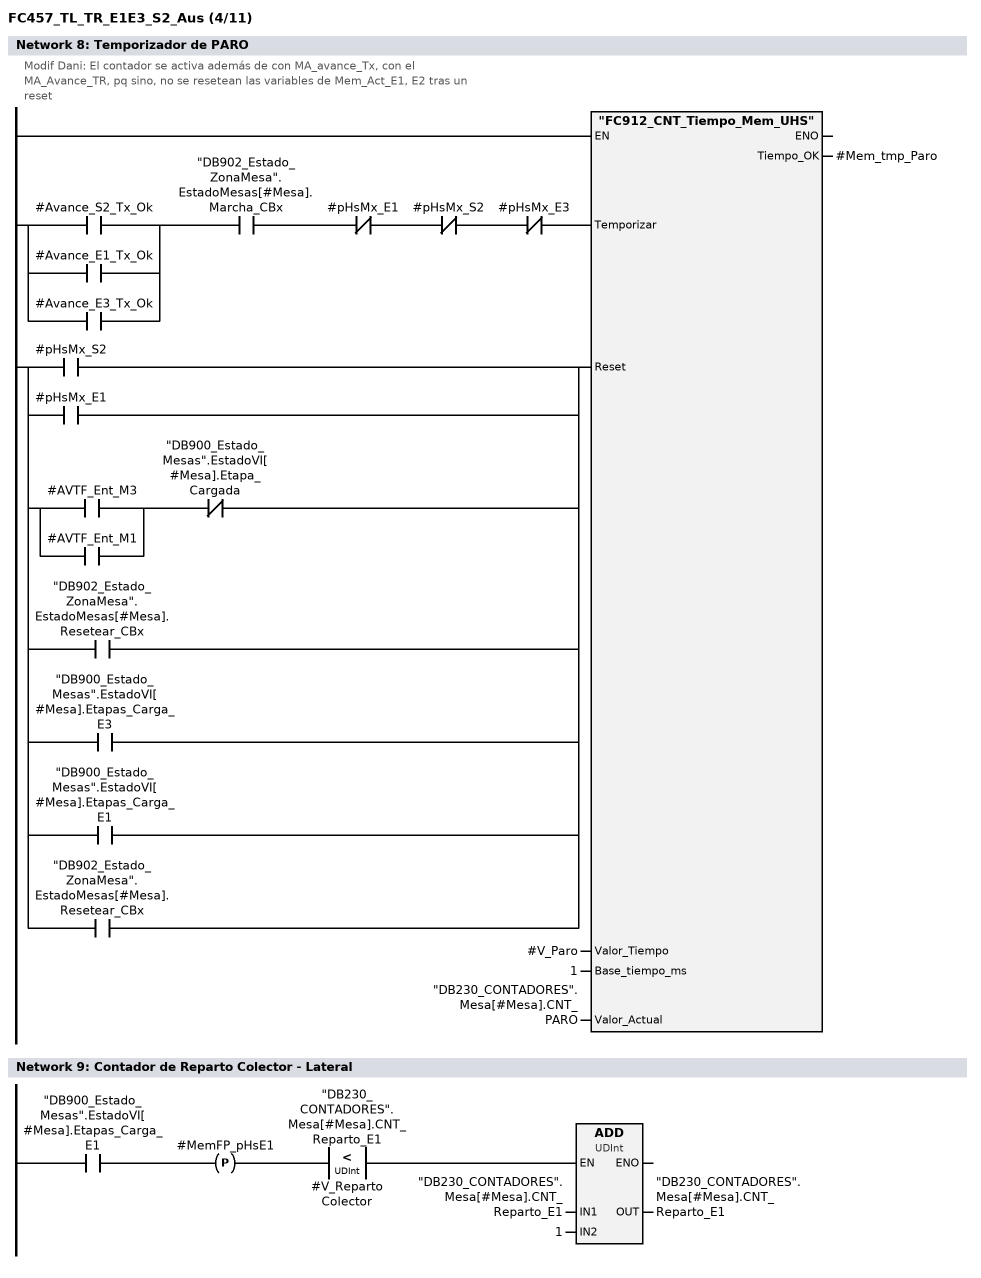
   RUNG wire#powerrail
      "FC912_CNT_Tiempo_Mem_UHS"(Temporizar := wire#w2, Reset := wire#w4, Valor_Tiempo := #V_Paro, Base_tiempo_ms := 1, Valor_Actual := "DB230_CONTADORES".Mesa[#Mesa].CNT_PARO, Tiempo_OK => #Mem_tmp_Paro)
   END_RUNG
   RUNG wire#powerrail
      Contact( #Avance_S2_Tx_Ok )
      wire#w1
      Contact( "DB902_Estado_ZonaMesa".EstadoMesas[#Mesa].Marcha_CBx )
      I_Contact( #pHsMx_E1 )
      I_Contact( #pHsMx_S2 )
      I_Contact( #pHsMx_E3 )
   END_RUNG wire#w2
   RUNG wire#powerrail
      Contact( #Avance_E1_Tx_Ok )
   END_RUNG wire#w1
   RUNG wire#powerrail
      Contact( #Avance_E3_Tx_Ok )
   END_RUNG wire#w1
   RUNG wire#powerrail
      Contact( #pHsMx_S2 )
   END_RUNG wire#w4
   RUNG wire#powerrail
      Contact( #pHsMx_E1 )
   END_RUNG wire#w4
   RUNG wire#powerrail
      Contact( #AVTF_Ent_M3 )
      wire#w3
      I_Contact( "DB900_Estado_Mesas".EstadoVI[#Mesa].Etapa_Cargada )
   END_RUNG wire#w4
   RUNG wire#powerrail
      Contact( #AVTF_Ent_M1 )
   END_RUNG wire#w3
   RUNG wire#powerrail
      Contact( "DB902_Estado_ZonaMesa".EstadoMesas[#Mesa].Resetear_CBx )
   END_RUNG wire#w4
   RUNG wire#powerrail
      Contact( "DB900_Estado_Mesas".EstadoVI[#Mesa].Etapas_Carga_E3 )
   END_RUNG wire#w4
   RUNG wire#powerrail
      Contact( "DB900_Estado_Mesas".EstadoVI[#Mesa].Etapas_Carga_E1 )
   END_RUNG wire#w4
   RUNG wire#powerrail
      Contact( "DB902_Estado_ZonaMesa".EstadoMesas[#Mesa].Resetear_CBx )
   END_RUNG wire#w4
   // the same network as SCL:
   "FC912_CNT_Tiempo_Mem_UHS"(Temporizar := (#Avance_S2_Tx_Ok OR #Avance_E1_Tx_Ok OR #Avance_E3_Tx_Ok) AND "DB902_Estado_ZonaMesa".EstadoMesas[#Mesa].Marcha_CBx AND NOT #pHsMx_E1 AND NOT #pHsMx_S2 AND NOT #pHsMx_E3,
                           Reset := #pHsMx_S2 OR #pHsMx_E1 OR ((#AVTF_Ent_M3 OR #AVTF_Ent_M1) AND NOT "DB900_Estado_Mesas".EstadoVI[#Mesa].Etapa_Cargada) OR "DB902_Estado_ZonaMesa".EstadoMesas[#Mesa].Resetear_CBx OR "DB900_Estado_Mesas".EstadoVI[#Mesa].Etapas_Carga_E3 OR "DB900_Estado_Mesas".EstadoVI[#Mesa].Etapas_Carga_E1 OR "DB902_Estado_ZonaMesa".EstadoMesas[#Mesa].Resetear_CBx,
                           Valor_Tiempo := #V_Paro,
                           Base_tiempo_ms := 1,
                           Valor_Actual := "DB230_CONTADORES".Mesa[#Mesa].CNT_PARO,
                           Tiempo_OK => #Mem_tmp_Paro);
END_REGION

REGION Network 9: Contador de Reparto Colector - Lateral
   RUNG wire#powerrail
      Contact( "DB900_Estado_Mesas".EstadoVI[#Mesa].Etapas_Carga_E1 )
      P_Trig( #MemFP_pHsE1 )
      { S7_Templates := "SrcType := UDInt" } LT_Contact(in1 := "DB230_CONTADORES".Mesa[#Mesa].CNT_Reparto_E1, in2 := #V_RepartoColector)
      { S7_Templates := "SrcType := UDInt"; S7_GenerateENO := "TRUE" } Add(in1 := "DB230_CONTADORES".Mesa[#Mesa].CNT_Reparto_E1, in2 := 1, out => "DB230_CONTADORES".Mesa[#Mesa].CNT_Reparto_E1)
   END_RUNG
   // the same network as SCL:
   #_w1 := "DB900_Estado_Mesas".EstadoVI[#Mesa].Etapas_Carga_E1 AND NOT #MemFP_pHsE1;   // rising edge
   #MemFP_pHsE1 := "DB900_Estado_Mesas".EstadoVI[#Mesa].Etapas_Carga_E1;
   IF #_w1 AND ("DB230_CONTADORES".Mesa[#Mesa].CNT_Reparto_E1 < #V_RepartoColector) THEN
       "DB230_CONTADORES".Mesa[#Mesa].CNT_Reparto_E1 := "DB230_CONTADORES".Mesa[#Mesa].CNT_Reparto_E1 + 1;
   END_IF;
END_REGION

REGION Network 10
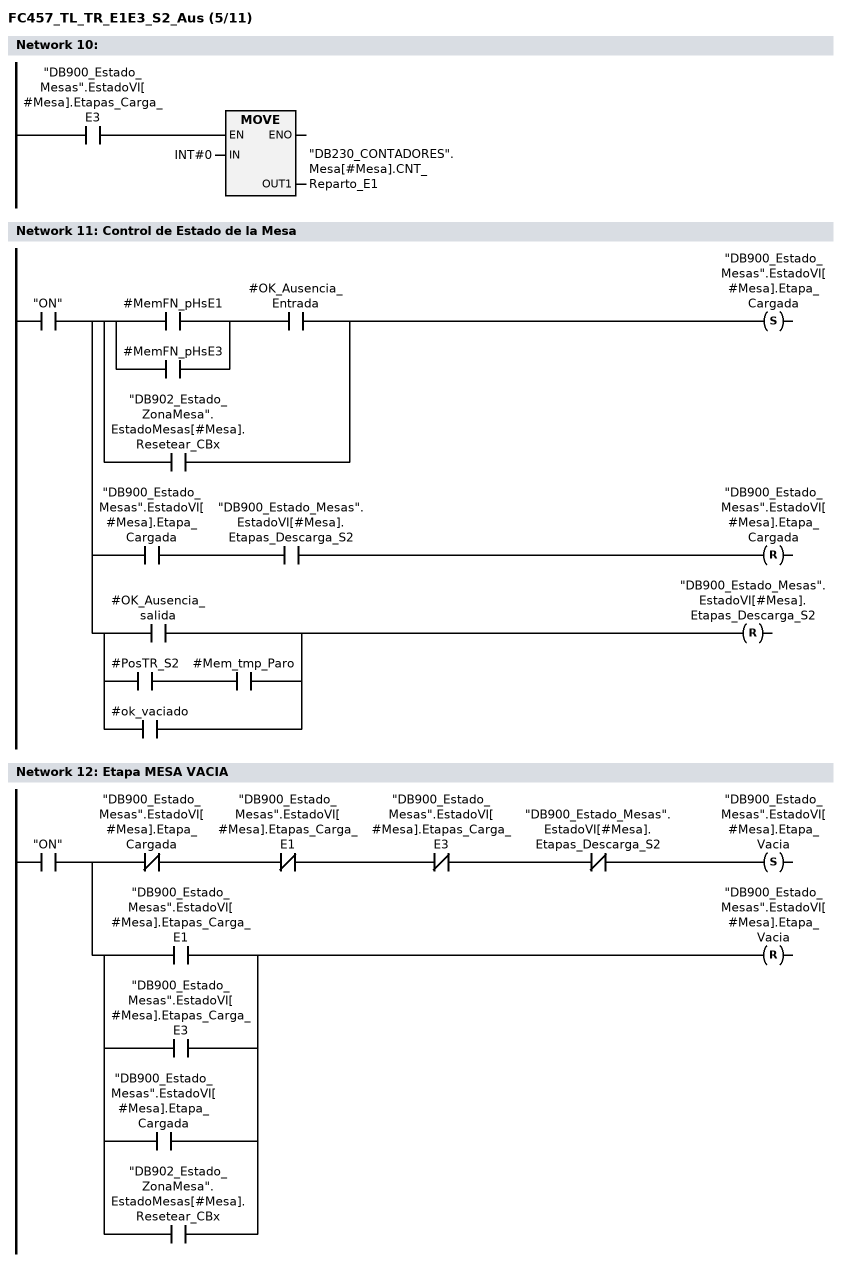
   RUNG wire#powerrail
      Contact( "DB900_Estado_Mesas".EstadoVI[#Mesa].Etapas_Carga_E3 )
      { S7_GenerateENO := "TRUE" } Move(in := INT#0, out1 => "DB230_CONTADORES".Mesa[#Mesa].CNT_Reparto_E1)
   END_RUNG
   // the same network as SCL:
   IF "DB900_Estado_Mesas".EstadoVI[#Mesa].Etapas_Carga_E3 THEN
       "DB230_CONTADORES".Mesa[#Mesa].CNT_Reparto_E1 := INT#0;
   END_IF;
END_REGION

REGION Network 11: Control de Estado de la Mesa
   RUNG wire#powerrail
      Contact( "ON" )
      wire#w1
      Contact( #MemFN_pHsE1 )
      wire#w2
      Contact( #OK_Ausencia_Entrada )
      wire#w3
      S_Coil( "DB900_Estado_Mesas".EstadoVI[#Mesa].Etapa_Cargada )
   END_RUNG
   RUNG wire#w1
      Contact( #MemFN_pHsE3 )
   END_RUNG wire#w2
   RUNG wire#w1
      Contact( "DB902_Estado_ZonaMesa".EstadoMesas[#Mesa].Resetear_CBx )
   END_RUNG wire#w3
   RUNG wire#w1
      Contact( "DB900_Estado_Mesas".EstadoVI[#Mesa].Etapa_Cargada )
      Contact( "DB900_Estado_Mesas".EstadoVI[#Mesa].Etapas_Descarga_S2 )
      R_Coil( "DB900_Estado_Mesas".EstadoVI[#Mesa].Etapa_Cargada )
   END_RUNG
   RUNG wire#w1
      Contact( #OK_Ausencia_salida )
      wire#w4
      R_Coil( "DB900_Estado_Mesas".EstadoVI[#Mesa].Etapas_Descarga_S2 )
   END_RUNG
   RUNG wire#w1
      Contact( #PosTR_S2 )
      Contact( #Mem_tmp_Paro )
   END_RUNG wire#w4
   RUNG wire#w1
      Contact( #ok_vaciado )
   END_RUNG wire#w4
   // the same network as SCL:
   IF "ON" AND (((#MemFN_pHsE1 OR #MemFN_pHsE3) AND #OK_Ausencia_Entrada) OR "DB902_Estado_ZonaMesa".EstadoMesas[#Mesa].Resetear_CBx) THEN
       "DB900_Estado_Mesas".EstadoVI[#Mesa].Etapa_Cargada := TRUE;
   END_IF;
   IF "ON" AND "DB900_Estado_Mesas".EstadoVI[#Mesa].Etapa_Cargada AND "DB900_Estado_Mesas".EstadoVI[#Mesa].Etapas_Descarga_S2 THEN
       "DB900_Estado_Mesas".EstadoVI[#Mesa].Etapa_Cargada := FALSE;
   END_IF;
   IF "ON" AND (#OK_Ausencia_salida OR (#PosTR_S2 AND #Mem_tmp_Paro) OR #ok_vaciado) THEN
       "DB900_Estado_Mesas".EstadoVI[#Mesa].Etapas_Descarga_S2 := FALSE;
   END_IF;
END_REGION

REGION Network 12: Etapa MESA VACIA
   RUNG wire#powerrail
      Contact( "ON" )
      wire#w1
      I_Contact( "DB900_Estado_Mesas".EstadoVI[#Mesa].Etapa_Cargada )
      I_Contact( "DB900_Estado_Mesas".EstadoVI[#Mesa].Etapas_Carga_E1 )
      I_Contact( "DB900_Estado_Mesas".EstadoVI[#Mesa].Etapas_Carga_E3 )
      I_Contact( "DB900_Estado_Mesas".EstadoVI[#Mesa].Etapas_Descarga_S2 )
      S_Coil( "DB900_Estado_Mesas".EstadoVI[#Mesa].Etapa_Vacia )
   END_RUNG
   RUNG wire#w1
      Contact( "DB900_Estado_Mesas".EstadoVI[#Mesa].Etapas_Carga_E1 )
      wire#w2
      R_Coil( "DB900_Estado_Mesas".EstadoVI[#Mesa].Etapa_Vacia )
   END_RUNG
   RUNG wire#w1
      Contact( "DB900_Estado_Mesas".EstadoVI[#Mesa].Etapas_Carga_E3 )
   END_RUNG wire#w2
   RUNG wire#w1
      Contact( "DB900_Estado_Mesas".EstadoVI[#Mesa].Etapa_Cargada )
   END_RUNG wire#w2
   RUNG wire#w1
      Contact( "DB902_Estado_ZonaMesa".EstadoMesas[#Mesa].Resetear_CBx )
   END_RUNG wire#w2
   // the same network as SCL:
   IF "ON" AND NOT "DB900_Estado_Mesas".EstadoVI[#Mesa].Etapa_Cargada AND NOT "DB900_Estado_Mesas".EstadoVI[#Mesa].Etapas_Carga_E1 AND NOT "DB900_Estado_Mesas".EstadoVI[#Mesa].Etapas_Carga_E3 AND NOT "DB900_Estado_Mesas".EstadoVI[#Mesa].Etapas_Descarga_S2 THEN
       "DB900_Estado_Mesas".EstadoVI[#Mesa].Etapa_Vacia := TRUE;
   END_IF;
   IF "ON" AND ("DB900_Estado_Mesas".EstadoVI[#Mesa].Etapas_Carga_E1 OR "DB900_Estado_Mesas".EstadoVI[#Mesa].Etapas_Carga_E3 OR "DB900_Estado_Mesas".EstadoVI[#Mesa].Etapa_Cargada OR "DB902_Estado_ZonaMesa".EstadoMesas[#Mesa].Resetear_CBx) THEN
       "DB900_Estado_Mesas".EstadoVI[#Mesa].Etapa_Vacia := FALSE;
   END_IF;
END_REGION

REGION Network 13
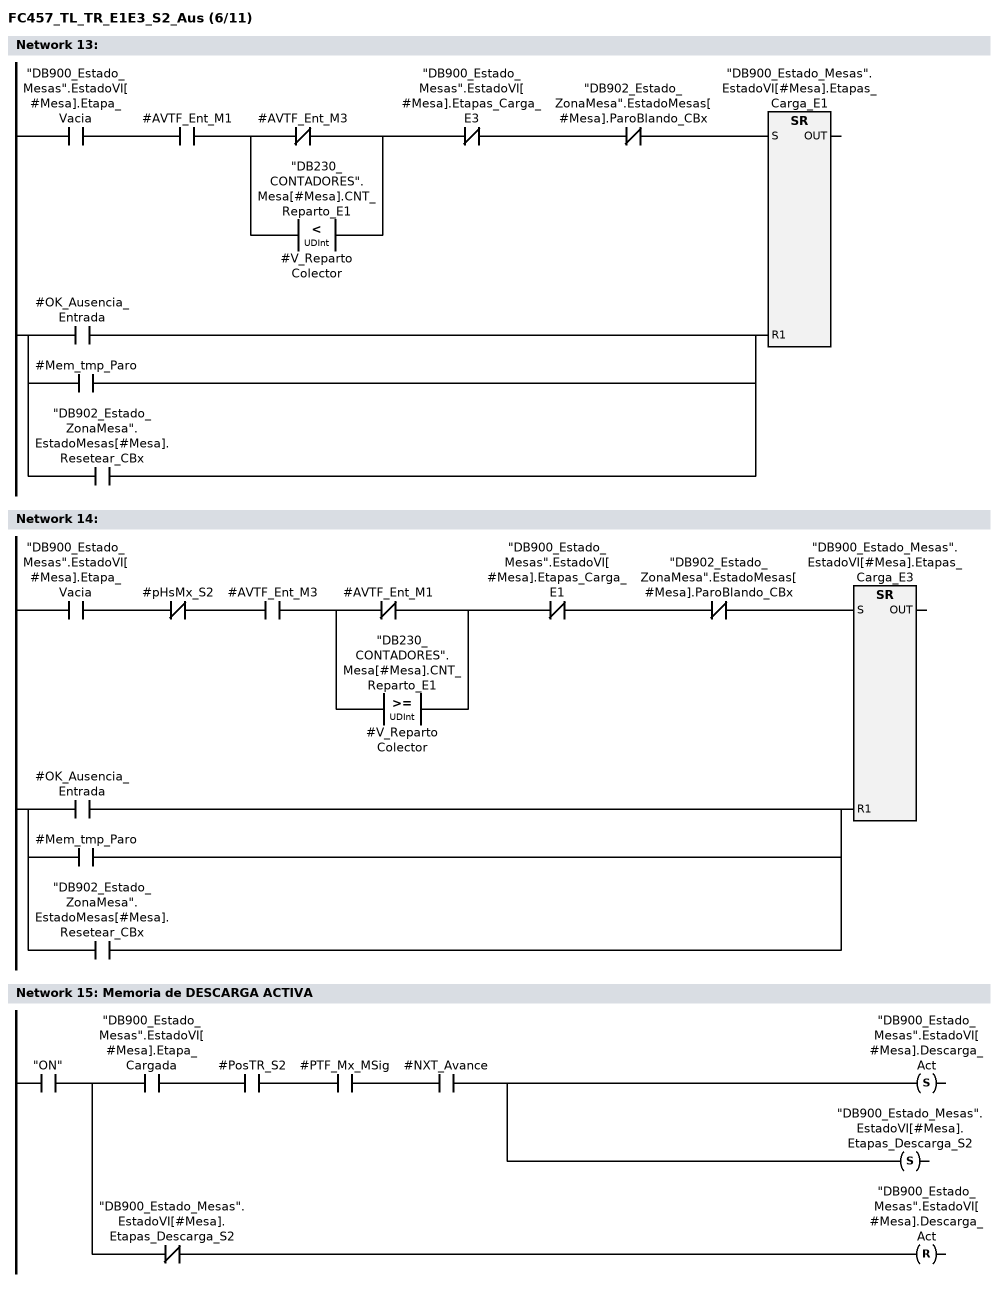
   RUNG wire#powerrail
      Contact( "DB900_Estado_Mesas".EstadoVI[#Mesa].Etapa_Vacia )
      Contact( #AVTF_Ent_M1 )
      wire#w1
      I_Contact( #AVTF_Ent_M3 )
      wire#w2
      I_Contact( "DB900_Estado_Mesas".EstadoVI[#Mesa].Etapas_Carga_E3 )
      I_Contact( "DB902_Estado_ZonaMesa".EstadoMesas[#Mesa].ParoBlando_CBx )
      S_SR(operand := "DB900_Estado_Mesas".EstadoVI[#Mesa].Etapas_Carga_E1, r1 := wire#w3)
   END_RUNG
   RUNG wire#w1
      { S7_Templates := "SrcType := UDInt" } LT_Contact(in1 := "DB230_CONTADORES".Mesa[#Mesa].CNT_Reparto_E1, in2 := #V_RepartoColector)
   END_RUNG wire#w2
   RUNG wire#powerrail
      Contact( #OK_Ausencia_Entrada )
   END_RUNG wire#w3
   RUNG wire#powerrail
      Contact( #Mem_tmp_Paro )
   END_RUNG wire#w3
   RUNG wire#powerrail
      Contact( "DB902_Estado_ZonaMesa".EstadoMesas[#Mesa].Resetear_CBx )
   END_RUNG wire#w3
   // the same network as SCL:
   #_w1 := #OK_Ausencia_Entrada OR #Mem_tmp_Paro OR "DB902_Estado_ZonaMesa".EstadoMesas[#Mesa].Resetear_CBx;
   IF "DB900_Estado_Mesas".EstadoVI[#Mesa].Etapa_Vacia AND #AVTF_Ent_M1 AND (NOT #AVTF_Ent_M3 OR ("DB230_CONTADORES".Mesa[#Mesa].CNT_Reparto_E1 < #V_RepartoColector)) AND NOT "DB900_Estado_Mesas".EstadoVI[#Mesa].Etapas_Carga_E3 AND NOT "DB902_Estado_ZonaMesa".EstadoMesas[#Mesa].ParoBlando_CBx THEN
       "DB900_Estado_Mesas".EstadoVI[#Mesa].Etapas_Carga_E1 := TRUE;   // SR flip-flop
   END_IF;
   IF #_w1 THEN "DB900_Estado_Mesas".EstadoVI[#Mesa].Etapas_Carga_E1 := FALSE; END_IF;
END_REGION

REGION Network 14
   RUNG wire#powerrail
      Contact( "DB900_Estado_Mesas".EstadoVI[#Mesa].Etapa_Vacia )
      I_Contact( #pHsMx_S2 )
      Contact( #AVTF_Ent_M3 )
      wire#w1
      I_Contact( #AVTF_Ent_M1 )
      wire#w2
      I_Contact( "DB900_Estado_Mesas".EstadoVI[#Mesa].Etapas_Carga_E1 )
      I_Contact( "DB902_Estado_ZonaMesa".EstadoMesas[#Mesa].ParoBlando_CBx )
      S_SR(operand := "DB900_Estado_Mesas".EstadoVI[#Mesa].Etapas_Carga_E3, r1 := wire#w3)
   END_RUNG
   RUNG wire#w1
      { S7_Templates := "SrcType := UDInt" } GE_Contact(in1 := "DB230_CONTADORES".Mesa[#Mesa].CNT_Reparto_E1, in2 := #V_RepartoColector)
   END_RUNG wire#w2
   RUNG wire#powerrail
      Contact( #OK_Ausencia_Entrada )
   END_RUNG wire#w3
   RUNG wire#powerrail
      Contact( #Mem_tmp_Paro )
   END_RUNG wire#w3
   RUNG wire#powerrail
      Contact( "DB902_Estado_ZonaMesa".EstadoMesas[#Mesa].Resetear_CBx )
   END_RUNG wire#w3
   // the same network as SCL:
   #_w1 := #OK_Ausencia_Entrada OR #Mem_tmp_Paro OR "DB902_Estado_ZonaMesa".EstadoMesas[#Mesa].Resetear_CBx;
   IF "DB900_Estado_Mesas".EstadoVI[#Mesa].Etapa_Vacia AND NOT #pHsMx_S2 AND #AVTF_Ent_M3 AND (NOT #AVTF_Ent_M1 OR ("DB230_CONTADORES".Mesa[#Mesa].CNT_Reparto_E1 >= #V_RepartoColector)) AND NOT "DB900_Estado_Mesas".EstadoVI[#Mesa].Etapas_Carga_E1 AND NOT "DB902_Estado_ZonaMesa".EstadoMesas[#Mesa].ParoBlando_CBx THEN
       "DB900_Estado_Mesas".EstadoVI[#Mesa].Etapas_Carga_E3 := TRUE;   // SR flip-flop
   END_IF;
   IF #_w1 THEN "DB900_Estado_Mesas".EstadoVI[#Mesa].Etapas_Carga_E3 := FALSE; END_IF;
END_REGION

REGION Network 15: Memoria de DESCARGA ACTIVA
   RUNG wire#powerrail
      Contact( "ON" )
      wire#w1
      Contact( "DB900_Estado_Mesas".EstadoVI[#Mesa].Etapa_Cargada )
      Contact( #PosTR_S2 )
      Contact( #PTF_Mx_MSig )
      Contact( #NXT_Avance )
      wire#w2
      S_Coil( "DB900_Estado_Mesas".EstadoVI[#Mesa].Descarga_Act )
   END_RUNG
   RUNG wire#w2
      S_Coil( "DB900_Estado_Mesas".EstadoVI[#Mesa].Etapas_Descarga_S2 )
   END_RUNG
   RUNG wire#w1
      I_Contact( "DB900_Estado_Mesas".EstadoVI[#Mesa].Etapas_Descarga_S2 )
      R_Coil( "DB900_Estado_Mesas".EstadoVI[#Mesa].Descarga_Act )
   END_RUNG
   // the same network as SCL:
   #_w1 := "ON" AND "DB900_Estado_Mesas".EstadoVI[#Mesa].Etapa_Cargada AND #PosTR_S2 AND #PTF_Mx_MSig AND #NXT_Avance;
   IF #_w1 THEN
       "DB900_Estado_Mesas".EstadoVI[#Mesa].Descarga_Act := TRUE;
       "DB900_Estado_Mesas".EstadoVI[#Mesa].Etapas_Descarga_S2 := TRUE;
   END_IF;
   IF "ON" AND NOT "DB900_Estado_Mesas".EstadoVI[#Mesa].Etapas_Descarga_S2 THEN
       "DB900_Estado_Mesas".EstadoVI[#Mesa].Descarga_Act := FALSE;
   END_IF;
END_REGION

REGION Network 16: Salidas Auxiliares
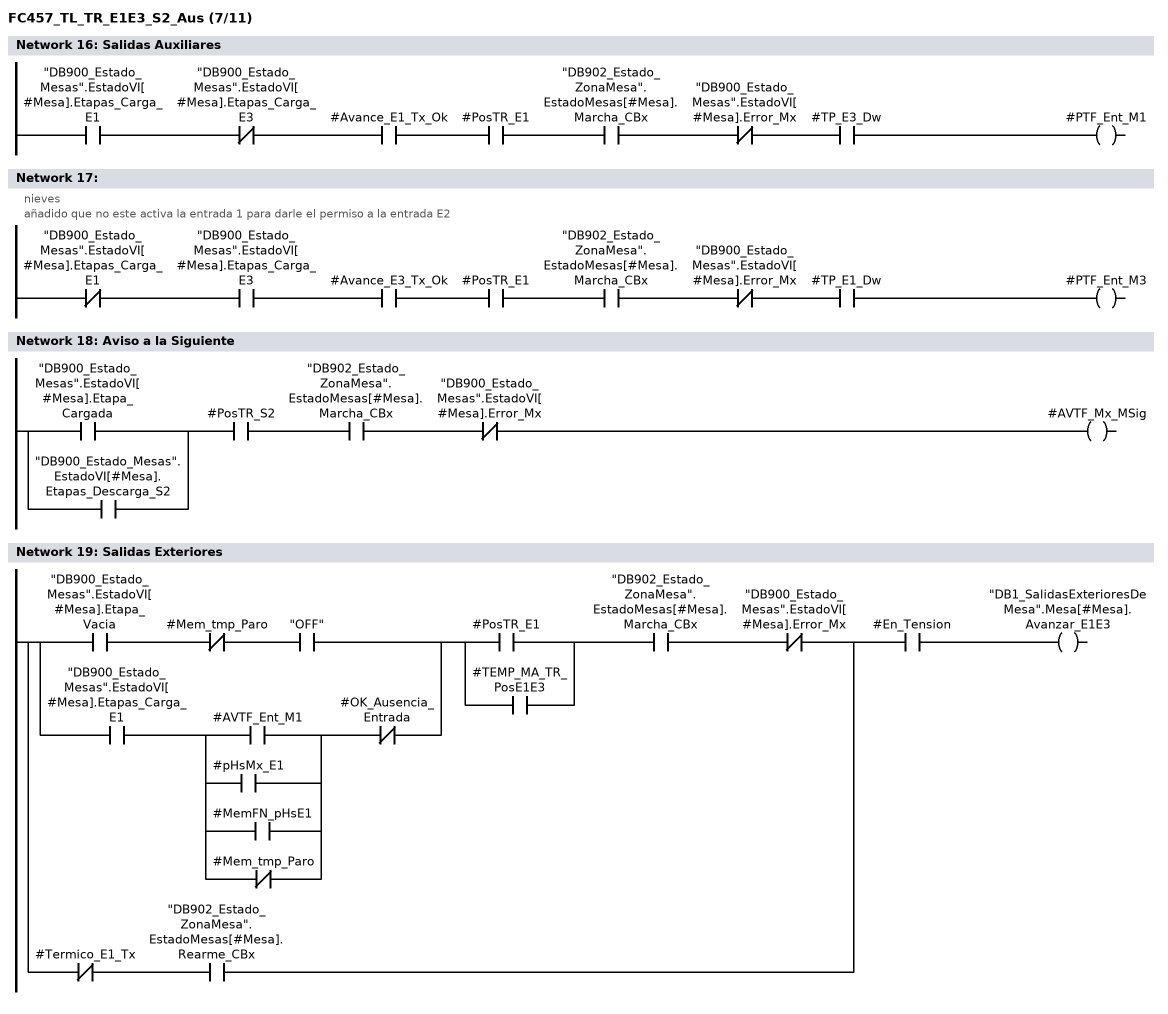
   RUNG wire#powerrail
      Contact( "DB900_Estado_Mesas".EstadoVI[#Mesa].Etapas_Carga_E1 )
      I_Contact( "DB900_Estado_Mesas".EstadoVI[#Mesa].Etapas_Carga_E3 )
      Contact( #Avance_E1_Tx_Ok )
      Contact( #PosTR_E1 )
      Contact( "DB902_Estado_ZonaMesa".EstadoMesas[#Mesa].Marcha_CBx )
      I_Contact( "DB900_Estado_Mesas".EstadoVI[#Mesa].Error_Mx )
      Contact( #TP_E3_Dw )
      Coil( #PTF_Ent_M1 )
   END_RUNG
   // the same network as SCL:
   #PTF_Ent_M1 := "DB900_Estado_Mesas".EstadoVI[#Mesa].Etapas_Carga_E1 AND NOT "DB900_Estado_Mesas".EstadoVI[#Mesa].Etapas_Carga_E3 AND #Avance_E1_Tx_Ok AND #PosTR_E1 AND "DB902_Estado_ZonaMesa".EstadoMesas[#Mesa].Marcha_CBx AND NOT "DB900_Estado_Mesas".EstadoVI[#Mesa].Error_Mx AND #TP_E3_Dw;
END_REGION

REGION Network 17
   // nieves
   // añadido que no este activa la entrada 1 para darle el permiso a la entrada E2
   RUNG wire#powerrail
      I_Contact( "DB900_Estado_Mesas".EstadoVI[#Mesa].Etapas_Carga_E1 )
      Contact( "DB900_Estado_Mesas".EstadoVI[#Mesa].Etapas_Carga_E3 )
      Contact( #Avance_E3_Tx_Ok )
      Contact( #PosTR_E1 )
      Contact( "DB902_Estado_ZonaMesa".EstadoMesas[#Mesa].Marcha_CBx )
      I_Contact( "DB900_Estado_Mesas".EstadoVI[#Mesa].Error_Mx )
      Contact( #TP_E1_Dw )
      Coil( #PTF_Ent_M3 )
   END_RUNG
   // the same network as SCL:
   #PTF_Ent_M3 := NOT "DB900_Estado_Mesas".EstadoVI[#Mesa].Etapas_Carga_E1 AND "DB900_Estado_Mesas".EstadoVI[#Mesa].Etapas_Carga_E3 AND #Avance_E3_Tx_Ok AND #PosTR_E1 AND "DB902_Estado_ZonaMesa".EstadoMesas[#Mesa].Marcha_CBx AND NOT "DB900_Estado_Mesas".EstadoVI[#Mesa].Error_Mx AND #TP_E1_Dw;
END_REGION

REGION Network 18: Aviso a la Siguiente
   RUNG wire#powerrail
      Contact( "DB900_Estado_Mesas".EstadoVI[#Mesa].Etapa_Cargada )
      wire#w1
      Contact( #PosTR_S2 )
      Contact( "DB902_Estado_ZonaMesa".EstadoMesas[#Mesa].Marcha_CBx )
      I_Contact( "DB900_Estado_Mesas".EstadoVI[#Mesa].Error_Mx )
      Coil( #AVTF_Mx_MSig )
   END_RUNG
   RUNG wire#powerrail
      Contact( "DB900_Estado_Mesas".EstadoVI[#Mesa].Etapas_Descarga_S2 )
   END_RUNG wire#w1
   // the same network as SCL:
   #AVTF_Mx_MSig := ("DB900_Estado_Mesas".EstadoVI[#Mesa].Etapa_Cargada OR "DB900_Estado_Mesas".EstadoVI[#Mesa].Etapas_Descarga_S2) AND #PosTR_S2 AND "DB902_Estado_ZonaMesa".EstadoMesas[#Mesa].Marcha_CBx AND NOT "DB900_Estado_Mesas".EstadoVI[#Mesa].Error_Mx;
END_REGION

REGION Network 19: Salidas Exteriores
   RUNG wire#powerrail
      Contact( "DB900_Estado_Mesas".EstadoVI[#Mesa].Etapa_Vacia )
      I_Contact( #Mem_tmp_Paro )
      Contact( "OFF" )
      wire#w1
      Contact( #PosTR_E1 )
      wire#w4
      Contact( "DB902_Estado_ZonaMesa".EstadoMesas[#Mesa].Marcha_CBx )
      I_Contact( "DB900_Estado_Mesas".EstadoVI[#Mesa].Error_Mx )
      wire#w5
      Contact( #En_Tension )
      Coil( "DB1_SalidasExterioresDeMesa".Mesa[#Mesa].Avanzar_E1E3 )
   END_RUNG
   RUNG wire#powerrail
      Contact( "DB900_Estado_Mesas".EstadoVI[#Mesa].Etapas_Carga_E1 )
      wire#w2
      Contact( #AVTF_Ent_M1 )
      wire#w3
      I_Contact( #OK_Ausencia_Entrada )
   END_RUNG wire#w1
   RUNG wire#w2
      Contact( #pHsMx_E1 )
   END_RUNG wire#w3
   RUNG wire#w2
      Contact( #MemFN_pHsE1 )
   END_RUNG wire#w3
   RUNG wire#w2
      I_Contact( #Mem_tmp_Paro )
   END_RUNG wire#w3
   RUNG wire#w1
      Contact( #TEMP_MA_TR_PosE1E3 )
   END_RUNG wire#w4
   RUNG wire#powerrail
      I_Contact( #Termico_E1_Tx )
      Contact( "DB902_Estado_ZonaMesa".EstadoMesas[#Mesa].Rearme_CBx )
   END_RUNG wire#w5
   // the same network as SCL:
   "DB1_SalidasExterioresDeMesa".Mesa[#Mesa].Avanzar_E1E3 := (((("DB900_Estado_Mesas".EstadoVI[#Mesa].Etapa_Vacia AND NOT #Mem_tmp_Paro AND "OFF") OR ("DB900_Estado_Mesas".EstadoVI[#Mesa].Etapas_Carga_E1 AND (#AVTF_Ent_M1 OR #pHsMx_E1 OR #MemFN_pHsE1 OR NOT #Mem_tmp_Paro) AND NOT #OK_Ausencia_Entrada)) AND (#PosTR_E1 OR #TEMP_MA_TR_PosE1E3) AND "DB902_Estado_ZonaMesa".EstadoMesas[#Mesa].Marcha_CBx AND NOT "DB900_Estado_Mesas".EstadoVI[#Mesa].Error_Mx) OR (NOT #Termico_E1_Tx AND "DB902_Estado_ZonaMesa".EstadoMesas[#Mesa].Rearme_CBx)) AND #En_Tension;
END_REGION

REGION Network 20: ---
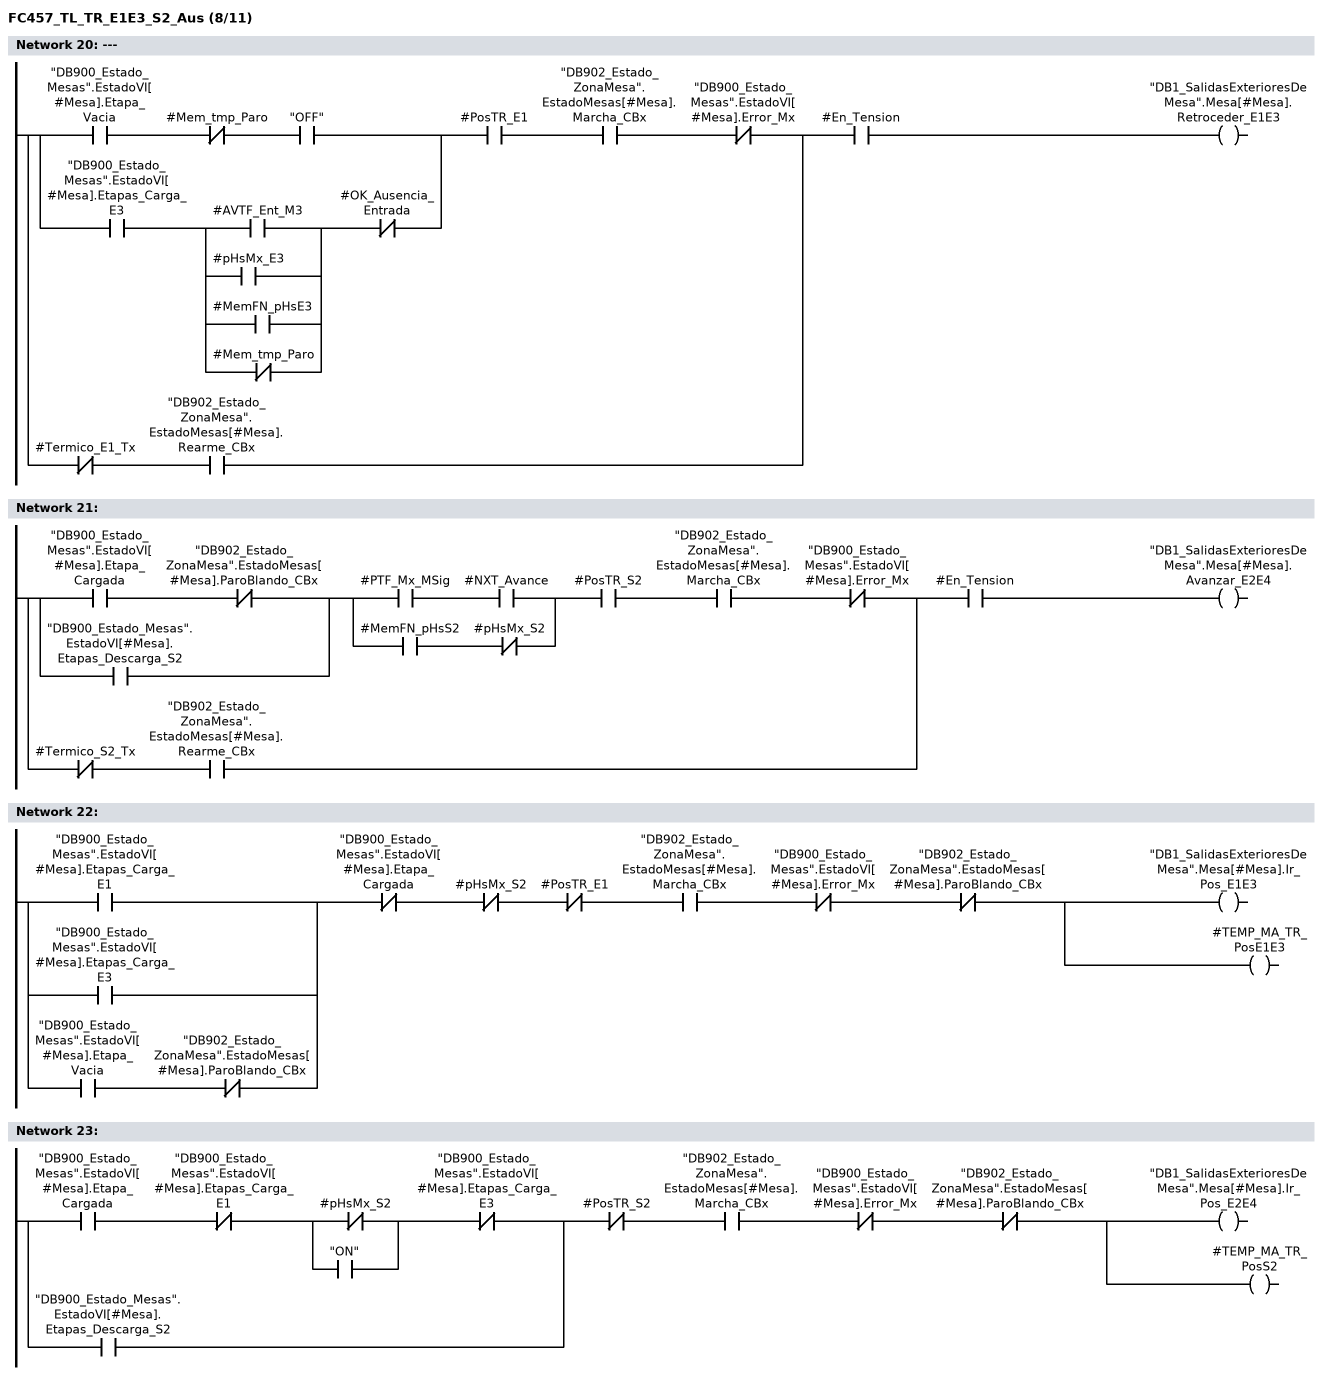
   RUNG wire#powerrail
      Contact( "DB900_Estado_Mesas".EstadoVI[#Mesa].Etapa_Vacia )
      I_Contact( #Mem_tmp_Paro )
      Contact( "OFF" )
      wire#w1
      Contact( #PosTR_E1 )
      Contact( "DB902_Estado_ZonaMesa".EstadoMesas[#Mesa].Marcha_CBx )
      I_Contact( "DB900_Estado_Mesas".EstadoVI[#Mesa].Error_Mx )
      wire#w4
      Contact( #En_Tension )
      Coil( "DB1_SalidasExterioresDeMesa".Mesa[#Mesa].Retroceder_E1E3 )
   END_RUNG
   RUNG wire#powerrail
      Contact( "DB900_Estado_Mesas".EstadoVI[#Mesa].Etapas_Carga_E3 )
      wire#w2
      Contact( #AVTF_Ent_M3 )
      wire#w3
      I_Contact( #OK_Ausencia_Entrada )
   END_RUNG wire#w1
   RUNG wire#w2
      Contact( #pHsMx_E3 )
   END_RUNG wire#w3
   RUNG wire#w2
      Contact( #MemFN_pHsE3 )
   END_RUNG wire#w3
   RUNG wire#w2
      I_Contact( #Mem_tmp_Paro )
   END_RUNG wire#w3
   RUNG wire#powerrail
      I_Contact( #Termico_E1_Tx )
      Contact( "DB902_Estado_ZonaMesa".EstadoMesas[#Mesa].Rearme_CBx )
   END_RUNG wire#w4
   // the same network as SCL:
   "DB1_SalidasExterioresDeMesa".Mesa[#Mesa].Retroceder_E1E3 := (((("DB900_Estado_Mesas".EstadoVI[#Mesa].Etapa_Vacia AND NOT #Mem_tmp_Paro AND "OFF") OR ("DB900_Estado_Mesas".EstadoVI[#Mesa].Etapas_Carga_E3 AND (#AVTF_Ent_M3 OR #pHsMx_E3 OR #MemFN_pHsE3 OR NOT #Mem_tmp_Paro) AND NOT #OK_Ausencia_Entrada)) AND #PosTR_E1 AND "DB902_Estado_ZonaMesa".EstadoMesas[#Mesa].Marcha_CBx AND NOT "DB900_Estado_Mesas".EstadoVI[#Mesa].Error_Mx) OR (NOT #Termico_E1_Tx AND "DB902_Estado_ZonaMesa".EstadoMesas[#Mesa].Rearme_CBx)) AND #En_Tension;
END_REGION

REGION Network 21
   RUNG wire#powerrail
      Contact( "DB900_Estado_Mesas".EstadoVI[#Mesa].Etapa_Cargada )
      I_Contact( "DB902_Estado_ZonaMesa".EstadoMesas[#Mesa].ParoBlando_CBx )
      wire#w1
      Contact( #PTF_Mx_MSig )
      Contact( #NXT_Avance )
      wire#w2
      Contact( #PosTR_S2 )
      Contact( "DB902_Estado_ZonaMesa".EstadoMesas[#Mesa].Marcha_CBx )
      I_Contact( "DB900_Estado_Mesas".EstadoVI[#Mesa].Error_Mx )
      wire#w3
      Contact( #En_Tension )
      Coil( "DB1_SalidasExterioresDeMesa".Mesa[#Mesa].Avanzar_E2E4 )
   END_RUNG
   RUNG wire#powerrail
      Contact( "DB900_Estado_Mesas".EstadoVI[#Mesa].Etapas_Descarga_S2 )
   END_RUNG wire#w1
   RUNG wire#w1
      Contact( #MemFN_pHsS2 )
      I_Contact( #pHsMx_S2 )
   END_RUNG wire#w2
   RUNG wire#powerrail
      I_Contact( #Termico_S2_Tx )
      Contact( "DB902_Estado_ZonaMesa".EstadoMesas[#Mesa].Rearme_CBx )
   END_RUNG wire#w3
   // the same network as SCL:
   "DB1_SalidasExterioresDeMesa".Mesa[#Mesa].Avanzar_E2E4 := (((("DB900_Estado_Mesas".EstadoVI[#Mesa].Etapa_Cargada AND NOT "DB902_Estado_ZonaMesa".EstadoMesas[#Mesa].ParoBlando_CBx) OR "DB900_Estado_Mesas".EstadoVI[#Mesa].Etapas_Descarga_S2) AND ((#PTF_Mx_MSig AND #NXT_Avance) OR (#MemFN_pHsS2 AND NOT #pHsMx_S2)) AND #PosTR_S2 AND "DB902_Estado_ZonaMesa".EstadoMesas[#Mesa].Marcha_CBx AND NOT "DB900_Estado_Mesas".EstadoVI[#Mesa].Error_Mx) OR (NOT #Termico_S2_Tx AND "DB902_Estado_ZonaMesa".EstadoMesas[#Mesa].Rearme_CBx)) AND #En_Tension;
END_REGION

REGION Network 22
   RUNG wire#powerrail
      Contact( "DB900_Estado_Mesas".EstadoVI[#Mesa].Etapas_Carga_E1 )
      wire#w1
      I_Contact( "DB900_Estado_Mesas".EstadoVI[#Mesa].Etapa_Cargada )
      I_Contact( #pHsMx_S2 )
      I_Contact( #PosTR_E1 )
      Contact( "DB902_Estado_ZonaMesa".EstadoMesas[#Mesa].Marcha_CBx )
      I_Contact( "DB900_Estado_Mesas".EstadoVI[#Mesa].Error_Mx )
      I_Contact( "DB902_Estado_ZonaMesa".EstadoMesas[#Mesa].ParoBlando_CBx )
      wire#w2
      Coil( "DB1_SalidasExterioresDeMesa".Mesa[#Mesa].Ir_Pos_E1E3 )
   END_RUNG
   RUNG wire#powerrail
      Contact( "DB900_Estado_Mesas".EstadoVI[#Mesa].Etapas_Carga_E3 )
   END_RUNG wire#w1
   RUNG wire#powerrail
      Contact( "DB900_Estado_Mesas".EstadoVI[#Mesa].Etapa_Vacia )
      I_Contact( "DB902_Estado_ZonaMesa".EstadoMesas[#Mesa].ParoBlando_CBx )
   END_RUNG wire#w1
   RUNG wire#w2
      Coil( #TEMP_MA_TR_PosE1E3 )
   END_RUNG
   // the same network as SCL:
   #_w1 := ("DB900_Estado_Mesas".EstadoVI[#Mesa].Etapas_Carga_E1 OR "DB900_Estado_Mesas".EstadoVI[#Mesa].Etapas_Carga_E3 OR ("DB900_Estado_Mesas".EstadoVI[#Mesa].Etapa_Vacia AND NOT "DB902_Estado_ZonaMesa".EstadoMesas[#Mesa].ParoBlando_CBx)) AND NOT "DB900_Estado_Mesas".EstadoVI[#Mesa].Etapa_Cargada AND NOT #pHsMx_S2 AND NOT #PosTR_E1 AND "DB902_Estado_ZonaMesa".EstadoMesas[#Mesa].Marcha_CBx AND NOT "DB900_Estado_Mesas".EstadoVI[#Mesa].Error_Mx AND NOT "DB902_Estado_ZonaMesa".EstadoMesas[#Mesa].ParoBlando_CBx;
   "DB1_SalidasExterioresDeMesa".Mesa[#Mesa].Ir_Pos_E1E3 := ("DB900_Estado_Mesas".EstadoVI[#Mesa].Etapas_Carga_E1 OR "DB900_Estado_Mesas".EstadoVI[#Mesa].Etapas_Carga_E3 OR ("DB900_Estado_Mesas".EstadoVI[#Mesa].Etapa_Vacia AND NOT "DB902_Estado_ZonaMesa".EstadoMesas[#Mesa].ParoBlando_CBx)) AND NOT "DB900_Estado_Mesas".EstadoVI[#Mesa].Etapa_Cargada AND NOT #pHsMx_S2 AND NOT #PosTR_E1 AND "DB902_Estado_ZonaMesa".EstadoMesas[#Mesa].Marcha_CBx AND NOT "DB900_Estado_Mesas".EstadoVI[#Mesa].Error_Mx AND NOT "DB902_Estado_ZonaMesa".EstadoMesas[#Mesa].ParoBlando_CBx;
   #TEMP_MA_TR_PosE1E3 := #_w1;
END_REGION

REGION Network 23
   RUNG wire#powerrail
      Contact( "DB900_Estado_Mesas".EstadoVI[#Mesa].Etapa_Cargada )
      I_Contact( "DB900_Estado_Mesas".EstadoVI[#Mesa].Etapas_Carga_E1 )
      wire#w1
      I_Contact( #pHsMx_S2 )
      wire#w2
      I_Contact( "DB900_Estado_Mesas".EstadoVI[#Mesa].Etapas_Carga_E3 )
      wire#w3
      I_Contact( #PosTR_S2 )
      Contact( "DB902_Estado_ZonaMesa".EstadoMesas[#Mesa].Marcha_CBx )
      I_Contact( "DB900_Estado_Mesas".EstadoVI[#Mesa].Error_Mx )
      I_Contact( "DB902_Estado_ZonaMesa".EstadoMesas[#Mesa].ParoBlando_CBx )
      wire#w4
      Coil( "DB1_SalidasExterioresDeMesa".Mesa[#Mesa].Ir_Pos_E2E4 )
   END_RUNG
   RUNG wire#w1
      Contact( "ON" )
   END_RUNG wire#w2
   RUNG wire#powerrail
      Contact( "DB900_Estado_Mesas".EstadoVI[#Mesa].Etapas_Descarga_S2 )
   END_RUNG wire#w3
   RUNG wire#w4
      Coil( #TEMP_MA_TR_PosS2 )
   END_RUNG
   // the same network as SCL:
   #_w1 := (("DB900_Estado_Mesas".EstadoVI[#Mesa].Etapa_Cargada AND NOT "DB900_Estado_Mesas".EstadoVI[#Mesa].Etapas_Carga_E1 AND (NOT #pHsMx_S2 OR "ON") AND NOT "DB900_Estado_Mesas".EstadoVI[#Mesa].Etapas_Carga_E3) OR "DB900_Estado_Mesas".EstadoVI[#Mesa].Etapas_Descarga_S2) AND NOT #PosTR_S2 AND "DB902_Estado_ZonaMesa".EstadoMesas[#Mesa].Marcha_CBx AND NOT "DB900_Estado_Mesas".EstadoVI[#Mesa].Error_Mx AND NOT "DB902_Estado_ZonaMesa".EstadoMesas[#Mesa].ParoBlando_CBx;
   "DB1_SalidasExterioresDeMesa".Mesa[#Mesa].Ir_Pos_E2E4 := (("DB900_Estado_Mesas".EstadoVI[#Mesa].Etapa_Cargada AND NOT "DB900_Estado_Mesas".EstadoVI[#Mesa].Etapas_Carga_E1 AND (NOT #pHsMx_S2 OR "ON") AND NOT "DB900_Estado_Mesas".EstadoVI[#Mesa].Etapas_Carga_E3) OR "DB900_Estado_Mesas".EstadoVI[#Mesa].Etapas_Descarga_S2) AND NOT #PosTR_S2 AND "DB902_Estado_ZonaMesa".EstadoMesas[#Mesa].Marcha_CBx AND NOT "DB900_Estado_Mesas".EstadoVI[#Mesa].Error_Mx AND NOT "DB902_Estado_ZonaMesa".EstadoMesas[#Mesa].ParoBlando_CBx;
   #TEMP_MA_TR_PosS2 := #_w1;
END_REGION

REGION Network 24: Subida de topes
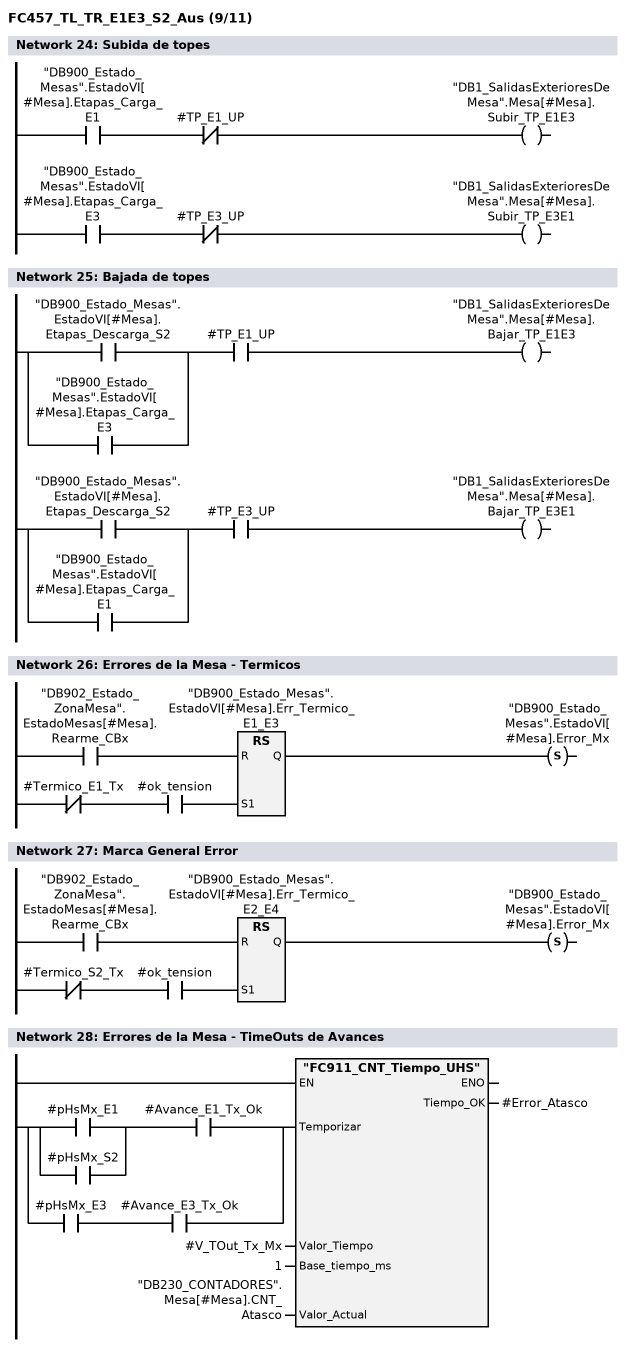
   RUNG wire#powerrail
      Contact( "DB900_Estado_Mesas".EstadoVI[#Mesa].Etapas_Carga_E1 )
      I_Contact( #TP_E1_UP )
      Coil( "DB1_SalidasExterioresDeMesa".Mesa[#Mesa].Subir_TP_E1E3 )
   END_RUNG
   RUNG wire#powerrail
      Contact( "DB900_Estado_Mesas".EstadoVI[#Mesa].Etapas_Carga_E3 )
      I_Contact( #TP_E3_UP )
      Coil( "DB1_SalidasExterioresDeMesa".Mesa[#Mesa].Subir_TP_E3E1 )
   END_RUNG
   // the same network as SCL:
   "DB1_SalidasExterioresDeMesa".Mesa[#Mesa].Subir_TP_E1E3 := "DB900_Estado_Mesas".EstadoVI[#Mesa].Etapas_Carga_E1 AND NOT #TP_E1_UP;
   "DB1_SalidasExterioresDeMesa".Mesa[#Mesa].Subir_TP_E3E1 := "DB900_Estado_Mesas".EstadoVI[#Mesa].Etapas_Carga_E3 AND NOT #TP_E3_UP;
END_REGION

REGION Network 25: Bajada de topes
   RUNG wire#powerrail
      Contact( "DB900_Estado_Mesas".EstadoVI[#Mesa].Etapas_Descarga_S2 )
      wire#w1
      Contact( #TP_E1_UP )
      Coil( "DB1_SalidasExterioresDeMesa".Mesa[#Mesa].Bajar_TP_E1E3 )
   END_RUNG
   RUNG wire#powerrail
      Contact( "DB900_Estado_Mesas".EstadoVI[#Mesa].Etapas_Carga_E3 )
   END_RUNG wire#w1
   RUNG wire#powerrail
      Contact( "DB900_Estado_Mesas".EstadoVI[#Mesa].Etapas_Descarga_S2 )
      wire#w2
      Contact( #TP_E3_UP )
      Coil( "DB1_SalidasExterioresDeMesa".Mesa[#Mesa].Bajar_TP_E3E1 )
   END_RUNG
   RUNG wire#powerrail
      Contact( "DB900_Estado_Mesas".EstadoVI[#Mesa].Etapas_Carga_E1 )
   END_RUNG wire#w2
   // the same network as SCL:
   "DB1_SalidasExterioresDeMesa".Mesa[#Mesa].Bajar_TP_E1E3 := ("DB900_Estado_Mesas".EstadoVI[#Mesa].Etapas_Descarga_S2 OR "DB900_Estado_Mesas".EstadoVI[#Mesa].Etapas_Carga_E3) AND #TP_E1_UP;
   "DB1_SalidasExterioresDeMesa".Mesa[#Mesa].Bajar_TP_E3E1 := ("DB900_Estado_Mesas".EstadoVI[#Mesa].Etapas_Descarga_S2 OR "DB900_Estado_Mesas".EstadoVI[#Mesa].Etapas_Carga_E1) AND #TP_E3_UP;
END_REGION

REGION Network 26: Errores de la Mesa - Termicos
   RUNG wire#powerrail
      Contact( "DB902_Estado_ZonaMesa".EstadoMesas[#Mesa].Rearme_CBx )
      S_RS(operand := "DB900_Estado_Mesas".EstadoVI[#Mesa].Err_Termico_E1_E3, s1 := wire#w1)
      S_Coil( "DB900_Estado_Mesas".EstadoVI[#Mesa].Error_Mx )
   END_RUNG
   RUNG wire#powerrail
      I_Contact( #Termico_E1_Tx )
      Contact( #ok_tension )
   END_RUNG wire#w1
   // the same network as SCL:
   IF "DB902_Estado_ZonaMesa".EstadoMesas[#Mesa].Rearme_CBx THEN
       "DB900_Estado_Mesas".EstadoVI[#Mesa].Err_Termico_E1_E3 := FALSE;   // RS flip-flop
   END_IF;
   IF NOT #Termico_E1_Tx AND #ok_tension THEN
       "DB900_Estado_Mesas".EstadoVI[#Mesa].Err_Termico_E1_E3 := TRUE;
   END_IF;
   IF "DB900_Estado_Mesas".EstadoVI[#Mesa].Err_Termico_E1_E3 THEN
       "DB900_Estado_Mesas".EstadoVI[#Mesa].Error_Mx := TRUE;
   END_IF;
END_REGION

REGION Network 27: Marca General Error
   RUNG wire#powerrail
      Contact( "DB902_Estado_ZonaMesa".EstadoMesas[#Mesa].Rearme_CBx )
      S_RS(operand := "DB900_Estado_Mesas".EstadoVI[#Mesa].Err_Termico_E2_E4, s1 := wire#w1)
      S_Coil( "DB900_Estado_Mesas".EstadoVI[#Mesa].Error_Mx )
   END_RUNG
   RUNG wire#powerrail
      I_Contact( #Termico_S2_Tx )
      Contact( #ok_tension )
   END_RUNG wire#w1
   // the same network as SCL:
   IF "DB902_Estado_ZonaMesa".EstadoMesas[#Mesa].Rearme_CBx THEN
       "DB900_Estado_Mesas".EstadoVI[#Mesa].Err_Termico_E2_E4 := FALSE;   // RS flip-flop
   END_IF;
   IF NOT #Termico_S2_Tx AND #ok_tension THEN
       "DB900_Estado_Mesas".EstadoVI[#Mesa].Err_Termico_E2_E4 := TRUE;
   END_IF;
   IF "DB900_Estado_Mesas".EstadoVI[#Mesa].Err_Termico_E2_E4 THEN
       "DB900_Estado_Mesas".EstadoVI[#Mesa].Error_Mx := TRUE;
   END_IF;
END_REGION

REGION Network 28: Errores de la Mesa - TimeOuts de Avances
   RUNG wire#powerrail
      "FC911_CNT_Tiempo_UHS"(Temporizar := wire#w2, Valor_Tiempo := #V_TOut_Tx_Mx, Base_tiempo_ms := 1, Valor_Actual := "DB230_CONTADORES".Mesa[#Mesa].CNT_Atasco, Tiempo_OK => #Error_Atasco)
   END_RUNG
   RUNG wire#powerrail
      Contact( #pHsMx_E1 )
      wire#w1
      Contact( #Avance_E1_Tx_Ok )
   END_RUNG wire#w2
   RUNG wire#powerrail
      Contact( #pHsMx_S2 )
   END_RUNG wire#w1
   RUNG wire#powerrail
      Contact( #pHsMx_E3 )
      Contact( #Avance_E3_Tx_Ok )
   END_RUNG wire#w2
   // the same network as SCL:
   "FC911_CNT_Tiempo_UHS"(Temporizar := ((#pHsMx_E1 OR #pHsMx_S2) AND #Avance_E1_Tx_Ok) OR (#pHsMx_E3 AND #Avance_E3_Tx_Ok),
                          Valor_Tiempo := #V_TOut_Tx_Mx,
                          Base_tiempo_ms := 1,
                          Valor_Actual := "DB230_CONTADORES".Mesa[#Mesa].CNT_Atasco,
                          Tiempo_OK => #Error_Atasco);
END_REGION

REGION Network 29
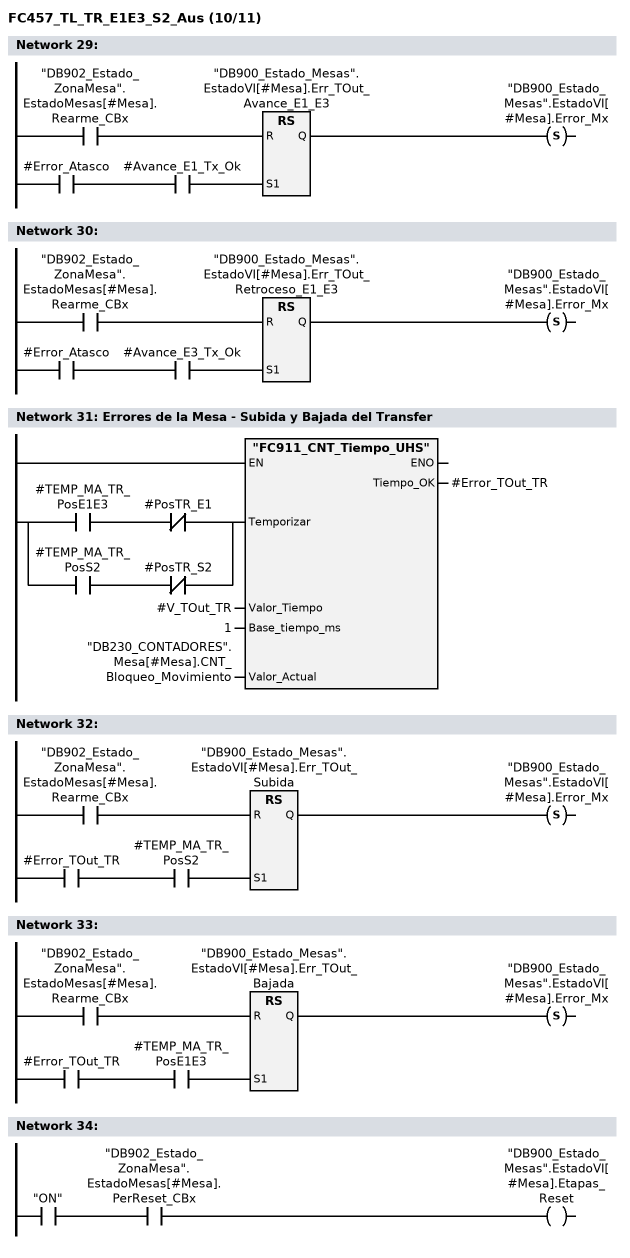
   RUNG wire#powerrail
      Contact( "DB902_Estado_ZonaMesa".EstadoMesas[#Mesa].Rearme_CBx )
      S_RS(operand := "DB900_Estado_Mesas".EstadoVI[#Mesa].Err_TOut_Avance_E1_E3, s1 := wire#w1)
      S_Coil( "DB900_Estado_Mesas".EstadoVI[#Mesa].Error_Mx )
   END_RUNG
   RUNG wire#powerrail
      Contact( #Error_Atasco )
      Contact( #Avance_E1_Tx_Ok )
   END_RUNG wire#w1
   // the same network as SCL:
   IF "DB902_Estado_ZonaMesa".EstadoMesas[#Mesa].Rearme_CBx THEN
       "DB900_Estado_Mesas".EstadoVI[#Mesa].Err_TOut_Avance_E1_E3 := FALSE;   // RS flip-flop
   END_IF;
   IF #Error_Atasco AND #Avance_E1_Tx_Ok THEN
       "DB900_Estado_Mesas".EstadoVI[#Mesa].Err_TOut_Avance_E1_E3 := TRUE;
   END_IF;
   IF "DB900_Estado_Mesas".EstadoVI[#Mesa].Err_TOut_Avance_E1_E3 THEN
       "DB900_Estado_Mesas".EstadoVI[#Mesa].Error_Mx := TRUE;
   END_IF;
END_REGION

REGION Network 30
   RUNG wire#powerrail
      Contact( "DB902_Estado_ZonaMesa".EstadoMesas[#Mesa].Rearme_CBx )
      S_RS(operand := "DB900_Estado_Mesas".EstadoVI[#Mesa].Err_TOut_Retroceso_E1_E3, s1 := wire#w1)
      S_Coil( "DB900_Estado_Mesas".EstadoVI[#Mesa].Error_Mx )
   END_RUNG
   RUNG wire#powerrail
      Contact( #Error_Atasco )
      Contact( #Avance_E3_Tx_Ok )
   END_RUNG wire#w1
   // the same network as SCL:
   IF "DB902_Estado_ZonaMesa".EstadoMesas[#Mesa].Rearme_CBx THEN
       "DB900_Estado_Mesas".EstadoVI[#Mesa].Err_TOut_Retroceso_E1_E3 := FALSE;   // RS flip-flop
   END_IF;
   IF #Error_Atasco AND #Avance_E3_Tx_Ok THEN
       "DB900_Estado_Mesas".EstadoVI[#Mesa].Err_TOut_Retroceso_E1_E3 := TRUE;
   END_IF;
   IF "DB900_Estado_Mesas".EstadoVI[#Mesa].Err_TOut_Retroceso_E1_E3 THEN
       "DB900_Estado_Mesas".EstadoVI[#Mesa].Error_Mx := TRUE;
   END_IF;
END_REGION

REGION Network 31: Errores de la Mesa - Subida y Bajada del Transfer
   RUNG wire#powerrail
      "FC911_CNT_Tiempo_UHS"(Temporizar := wire#w1, Valor_Tiempo := #V_TOut_TR, Base_tiempo_ms := 1, Valor_Actual := "DB230_CONTADORES".Mesa[#Mesa].CNT_Bloqueo_Movimiento, Tiempo_OK => #Error_TOut_TR)
   END_RUNG
   RUNG wire#powerrail
      Contact( #TEMP_MA_TR_PosE1E3 )
      I_Contact( #PosTR_E1 )
   END_RUNG wire#w1
   RUNG wire#powerrail
      Contact( #TEMP_MA_TR_PosS2 )
      I_Contact( #PosTR_S2 )
   END_RUNG wire#w1
   // the same network as SCL:
   "FC911_CNT_Tiempo_UHS"(Temporizar := (#TEMP_MA_TR_PosE1E3 AND NOT #PosTR_E1) OR (#TEMP_MA_TR_PosS2 AND NOT #PosTR_S2),
                          Valor_Tiempo := #V_TOut_TR,
                          Base_tiempo_ms := 1,
                          Valor_Actual := "DB230_CONTADORES".Mesa[#Mesa].CNT_Bloqueo_Movimiento,
                          Tiempo_OK => #Error_TOut_TR);
END_REGION

REGION Network 32
   RUNG wire#powerrail
      Contact( "DB902_Estado_ZonaMesa".EstadoMesas[#Mesa].Rearme_CBx )
      S_RS(operand := "DB900_Estado_Mesas".EstadoVI[#Mesa].Err_TOut_Subida, s1 := wire#w1)
      S_Coil( "DB900_Estado_Mesas".EstadoVI[#Mesa].Error_Mx )
   END_RUNG
   RUNG wire#powerrail
      Contact( #Error_TOut_TR )
      Contact( #TEMP_MA_TR_PosS2 )
   END_RUNG wire#w1
   // the same network as SCL:
   IF "DB902_Estado_ZonaMesa".EstadoMesas[#Mesa].Rearme_CBx THEN
       "DB900_Estado_Mesas".EstadoVI[#Mesa].Err_TOut_Subida := FALSE;   // RS flip-flop
   END_IF;
   IF #Error_TOut_TR AND #TEMP_MA_TR_PosS2 THEN
       "DB900_Estado_Mesas".EstadoVI[#Mesa].Err_TOut_Subida := TRUE;
   END_IF;
   IF "DB900_Estado_Mesas".EstadoVI[#Mesa].Err_TOut_Subida THEN
       "DB900_Estado_Mesas".EstadoVI[#Mesa].Error_Mx := TRUE;
   END_IF;
END_REGION

REGION Network 33
   RUNG wire#powerrail
      Contact( "DB902_Estado_ZonaMesa".EstadoMesas[#Mesa].Rearme_CBx )
      S_RS(operand := "DB900_Estado_Mesas".EstadoVI[#Mesa].Err_TOut_Bajada, s1 := wire#w1)
      S_Coil( "DB900_Estado_Mesas".EstadoVI[#Mesa].Error_Mx )
   END_RUNG
   RUNG wire#powerrail
      Contact( #Error_TOut_TR )
      Contact( #TEMP_MA_TR_PosE1E3 )
   END_RUNG wire#w1
   // the same network as SCL:
   IF "DB902_Estado_ZonaMesa".EstadoMesas[#Mesa].Rearme_CBx THEN
       "DB900_Estado_Mesas".EstadoVI[#Mesa].Err_TOut_Bajada := FALSE;   // RS flip-flop
   END_IF;
   IF #Error_TOut_TR AND #TEMP_MA_TR_PosE1E3 THEN
       "DB900_Estado_Mesas".EstadoVI[#Mesa].Err_TOut_Bajada := TRUE;
   END_IF;
   IF "DB900_Estado_Mesas".EstadoVI[#Mesa].Err_TOut_Bajada THEN
       "DB900_Estado_Mesas".EstadoVI[#Mesa].Error_Mx := TRUE;
   END_IF;
END_REGION

REGION Network 34
   RUNG wire#powerrail
      Contact( "ON" )
      Contact( "DB902_Estado_ZonaMesa".EstadoMesas[#Mesa].PerReset_CBx )
      Coil( "DB900_Estado_Mesas".EstadoVI[#Mesa].Etapas_Reset )
   END_RUNG
   // the same network as SCL:
   "DB900_Estado_Mesas".EstadoVI[#Mesa].Etapas_Reset := "ON" AND "DB902_Estado_ZonaMesa".EstadoMesas[#Mesa].PerReset_CBx;
END_REGION

REGION Network 35: Entradas Mesas
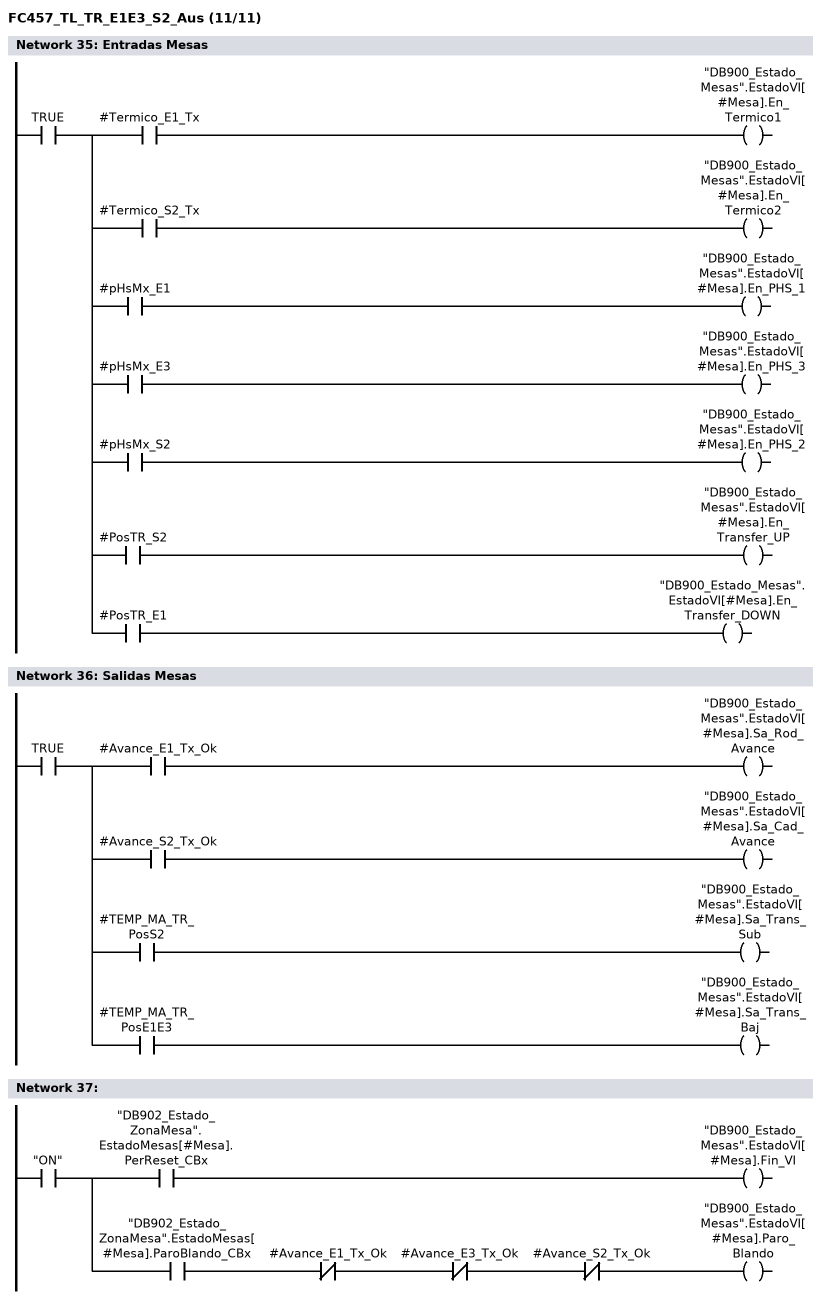
   RUNG wire#powerrail
      Contact( TRUE )
      wire#w1
      Contact( #Termico_E1_Tx )
      Coil( "DB900_Estado_Mesas".EstadoVI[#Mesa].En_Termico1 )
   END_RUNG
   RUNG wire#w1
      Contact( #Termico_S2_Tx )
      Coil( "DB900_Estado_Mesas".EstadoVI[#Mesa].En_Termico2 )
   END_RUNG
   RUNG wire#w1
      Contact( #pHsMx_E1 )
      Coil( "DB900_Estado_Mesas".EstadoVI[#Mesa].En_PHS_1 )
   END_RUNG
   RUNG wire#w1
      Contact( #pHsMx_E3 )
      Coil( "DB900_Estado_Mesas".EstadoVI[#Mesa].En_PHS_3 )
   END_RUNG
   RUNG wire#w1
      Contact( #pHsMx_S2 )
      Coil( "DB900_Estado_Mesas".EstadoVI[#Mesa].En_PHS_2 )
   END_RUNG
   RUNG wire#w1
      Contact( #PosTR_S2 )
      Coil( "DB900_Estado_Mesas".EstadoVI[#Mesa].En_Transfer_UP )
   END_RUNG
   RUNG wire#w1
      Contact( #PosTR_E1 )
      Coil( "DB900_Estado_Mesas".EstadoVI[#Mesa].En_Transfer_DOWN )
   END_RUNG
   // the same network as SCL:
   "DB900_Estado_Mesas".EstadoVI[#Mesa].En_Termico1 := TRUE AND #Termico_E1_Tx;
   "DB900_Estado_Mesas".EstadoVI[#Mesa].En_Termico2 := TRUE AND #Termico_S2_Tx;
   "DB900_Estado_Mesas".EstadoVI[#Mesa].En_PHS_1 := TRUE AND #pHsMx_E1;
   "DB900_Estado_Mesas".EstadoVI[#Mesa].En_PHS_3 := TRUE AND #pHsMx_E3;
   "DB900_Estado_Mesas".EstadoVI[#Mesa].En_PHS_2 := TRUE AND #pHsMx_S2;
   "DB900_Estado_Mesas".EstadoVI[#Mesa].En_Transfer_UP := TRUE AND #PosTR_S2;
   "DB900_Estado_Mesas".EstadoVI[#Mesa].En_Transfer_DOWN := TRUE AND #PosTR_E1;
END_REGION

REGION Network 36: Salidas Mesas
   RUNG wire#powerrail
      Contact( TRUE )
      wire#w1
      Contact( #Avance_E1_Tx_Ok )
      Coil( "DB900_Estado_Mesas".EstadoVI[#Mesa].Sa_Rod_Avance )
   END_RUNG
   RUNG wire#w1
      Contact( #Avance_S2_Tx_Ok )
      Coil( "DB900_Estado_Mesas".EstadoVI[#Mesa].Sa_Cad_Avance )
   END_RUNG
   RUNG wire#w1
      Contact( #TEMP_MA_TR_PosS2 )
      Coil( "DB900_Estado_Mesas".EstadoVI[#Mesa].Sa_Trans_Sub )
   END_RUNG
   RUNG wire#w1
      Contact( #TEMP_MA_TR_PosE1E3 )
      Coil( "DB900_Estado_Mesas".EstadoVI[#Mesa].Sa_Trans_Baj )
   END_RUNG
   // the same network as SCL:
   "DB900_Estado_Mesas".EstadoVI[#Mesa].Sa_Rod_Avance := TRUE AND #Avance_E1_Tx_Ok;
   "DB900_Estado_Mesas".EstadoVI[#Mesa].Sa_Cad_Avance := TRUE AND #Avance_S2_Tx_Ok;
   "DB900_Estado_Mesas".EstadoVI[#Mesa].Sa_Trans_Sub := TRUE AND #TEMP_MA_TR_PosS2;
   "DB900_Estado_Mesas".EstadoVI[#Mesa].Sa_Trans_Baj := TRUE AND #TEMP_MA_TR_PosE1E3;
END_REGION

REGION Network 37
   RUNG wire#powerrail
      Contact( "ON" )
      wire#w1
      Contact( "DB902_Estado_ZonaMesa".EstadoMesas[#Mesa].PerReset_CBx )
      Coil( "DB900_Estado_Mesas".EstadoVI[#Mesa].Fin_VI )
   END_RUNG
   RUNG wire#w1
      Contact( "DB902_Estado_ZonaMesa".EstadoMesas[#Mesa].ParoBlando_CBx )
      I_Contact( #Avance_E1_Tx_Ok )
      I_Contact( #Avance_E3_Tx_Ok )
      I_Contact( #Avance_S2_Tx_Ok )
      Coil( "DB900_Estado_Mesas".EstadoVI[#Mesa].Paro_Blando )
   END_RUNG
   // the same network as SCL:
   "DB900_Estado_Mesas".EstadoVI[#Mesa].Fin_VI := "ON" AND "DB902_Estado_ZonaMesa".EstadoMesas[#Mesa].PerReset_CBx;
   "DB900_Estado_Mesas".EstadoVI[#Mesa].Paro_Blando := "ON" AND "DB902_Estado_ZonaMesa".EstadoMesas[#Mesa].ParoBlando_CBx AND NOT #Avance_E1_Tx_Ok AND NOT #Avance_E3_Tx_Ok AND NOT #Avance_S2_Tx_Ok;
END_REGION
END_FUNCTION

FUNCTION "FC460_TL_Merge" : Void   // FC460, LAD
{ S7_Optimized_Access := 'FALSE' }
AUTHOR : TLigero
NAME : 20160208
VERSION : 3.3
// stored: AutoNumber false, SetENOAutomatically false
   VAR_INPUT
      Mesa : UInt;
      En_Tension : Bool;
      PhsMx : Bool;
      Avance_Tx : Bool;
      Termico_Tx : Bool;
      Simul_Mx : Bool;
      AVTF_MAnt_E1 : Bool;
      AVTF_MAnt_E2 : Bool;
      PTF_Mx_MSig : Bool;
      NXT_Avance : Bool;
      V_Paro : UDInt;
      V_TOut_Tx_Mx : UDInt;
      V_CNT_pHsMx : UDInt;
      V_Salida : UDInt;
      V_Gap : UDInt;
      V_Cajas_Equ_E1 : UDInt;
      V_Cajas_Equ_E2 : UDInt;
      V_Vaciado_E1 : UDInt;
      V_Vaciado_E2 : UDInt;
   END_VAR
   VAR_OUTPUT
      PTF_Ent_M1 : Bool;
      PTF_Ent_M2 : Bool;
      AVTF_Mx_MSig : Bool;
      NXT_Descarga_Act : Bool;
   END_VAR
   VAR_IN_OUT
      Mem_CNT_Salida : Bool;
      Mem_CNT_Tmp_Paro_Tx : Bool;
      MAUX_FP_Marcha : Bool;
      MAUX_FN_PHS : Bool;
      MAUX_PRV_Carga_OK_E1 : Bool;
      MAUX_PRV_Carga_OK_E2 : Bool;
      MAUX_FP_contador_E1 : Bool;
      MAUX_FP_contador_E2 : Bool;
      MAUX_FP_En_camino_E1 : Bool;
      MAUX_FP_En_camino_E2 : Bool;
      MAUX_key_En_E1 : Bool;
      MAUX_key_En_E2 : Bool;
      MAUX_Key_por_E1_fue_usada : Bool;
      MAUX_Key_por_E2_fue_usada : Bool;
      MAUX_Caja_En_Camino_E1 : Bool;
      MAUX_Caja_En_Camino_E2 : Bool;
   END_VAR
   VAR_TEMP
      OK_Avance : Bool;
      fp_Marcha : Bool;
      fn_phs_tx : Bool;
      fp_phs_tx : Bool;
      Mem_CNT_Centrado : Bool;
      Mem_CNT_Gap : Bool;
      Error_atasco : Bool;
      TEMP_NXT_AVTF : Bool;
      TEMP_PRV_CARGA_OK : Bool;
      VaciadoE1_OK : Bool;
      VaciadoE2_OK : Bool;
      ok_tension : Bool;
   END_VAR
   VAR_TEMP   // added for the SCL form of the ladder/FBD networks
      _w1 : Bool;
   END_VAR
BEGIN

REGION Network 1: Marca General Error
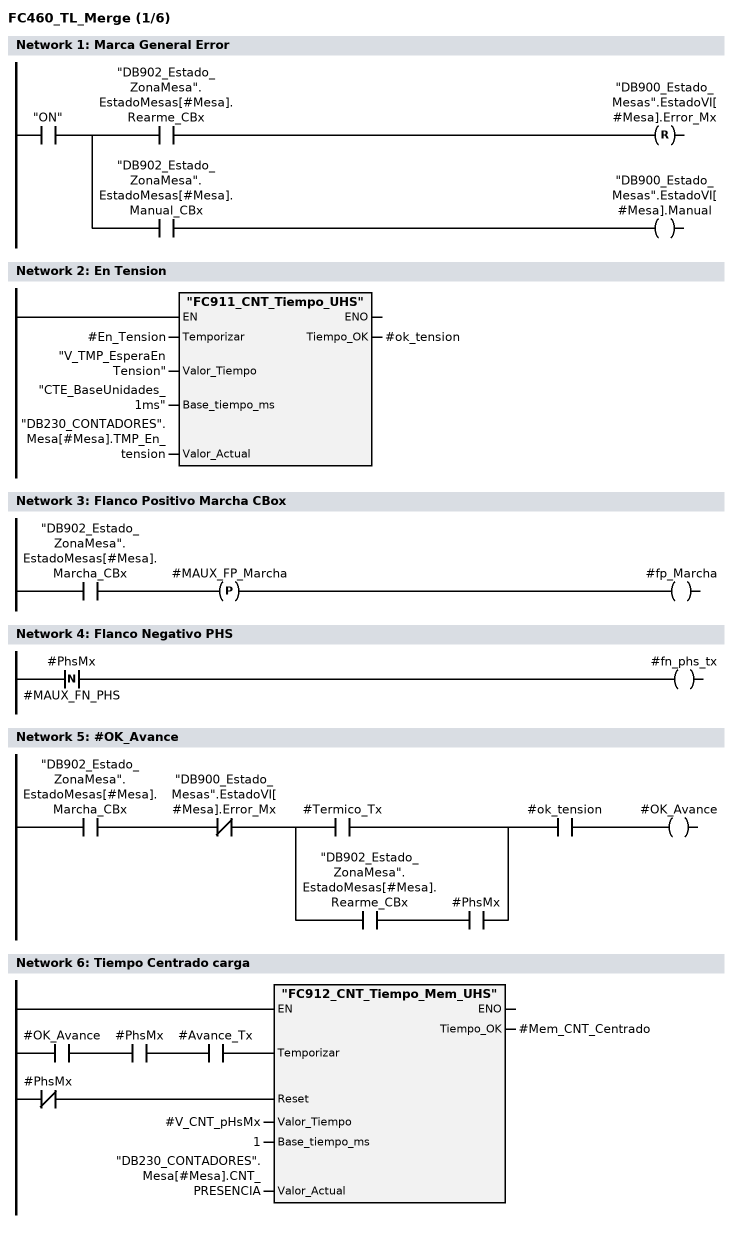
   RUNG wire#powerrail
      Contact( "ON" )
      wire#w1
      Contact( "DB902_Estado_ZonaMesa".EstadoMesas[#Mesa].Rearme_CBx )
      R_Coil( "DB900_Estado_Mesas".EstadoVI[#Mesa].Error_Mx )
   END_RUNG
   RUNG wire#w1
      Contact( "DB902_Estado_ZonaMesa".EstadoMesas[#Mesa].Manual_CBx )
      Coil( "DB900_Estado_Mesas".EstadoVI[#Mesa].Manual )
   END_RUNG
   // the same network as SCL:
   IF "ON" AND "DB902_Estado_ZonaMesa".EstadoMesas[#Mesa].Rearme_CBx THEN
       "DB900_Estado_Mesas".EstadoVI[#Mesa].Error_Mx := FALSE;
   END_IF;
   "DB900_Estado_Mesas".EstadoVI[#Mesa].Manual := "ON" AND "DB902_Estado_ZonaMesa".EstadoMesas[#Mesa].Manual_CBx;
END_REGION

REGION Network 2: En Tension
   RUNG wire#powerrail
      "FC911_CNT_Tiempo_UHS"(Temporizar := #En_Tension, Valor_Tiempo := "V_TMP_EsperaEnTension", Base_tiempo_ms := "CTE_BaseUnidades_1ms", Valor_Actual := "DB230_CONTADORES".Mesa[#Mesa].TMP_En_tension, Tiempo_OK => #ok_tension)
   END_RUNG
   // the same network as SCL:
   "FC911_CNT_Tiempo_UHS"(Temporizar := #En_Tension,
                          Valor_Tiempo := "V_TMP_EsperaEnTension",
                          Base_tiempo_ms := "CTE_BaseUnidades_1ms",
                          Valor_Actual := "DB230_CONTADORES".Mesa[#Mesa].TMP_En_tension,
                          Tiempo_OK => #ok_tension);
END_REGION

REGION Network 3: Flanco Positivo Marcha CBox
   RUNG wire#powerrail
      Contact( "DB902_Estado_ZonaMesa".EstadoMesas[#Mesa].Marcha_CBx )
      P_Trig( #MAUX_FP_Marcha )
      Coil( #fp_Marcha )
   END_RUNG
   // the same network as SCL:
   #_w1 := "DB902_Estado_ZonaMesa".EstadoMesas[#Mesa].Marcha_CBx AND NOT #MAUX_FP_Marcha;   // rising edge
   #MAUX_FP_Marcha := "DB902_Estado_ZonaMesa".EstadoMesas[#Mesa].Marcha_CBx;
   #fp_Marcha := #_w1;
END_REGION

REGION Network 4: Flanco Negativo PHS
   RUNG wire#powerrail
      N_Contact(operand := #PhsMx, bit := #MAUX_FN_PHS)
      Coil( #fn_phs_tx )
   END_RUNG
   // the same network as SCL:
   #_w1 := NOT #PhsMx AND #MAUX_FN_PHS;   // falling edge of #PhsMx
   #MAUX_FN_PHS := #PhsMx;
   #fn_phs_tx := #_w1;
END_REGION

REGION Network 5: #OK_Avance
   RUNG wire#powerrail
      Contact( "DB902_Estado_ZonaMesa".EstadoMesas[#Mesa].Marcha_CBx )
      I_Contact( "DB900_Estado_Mesas".EstadoVI[#Mesa].Error_Mx )
      wire#w1
      Contact( #Termico_Tx )
      wire#w2
      Contact( #ok_tension )
      Coil( #OK_Avance )
   END_RUNG
   RUNG wire#w1
      Contact( "DB902_Estado_ZonaMesa".EstadoMesas[#Mesa].Rearme_CBx )
      Contact( #PhsMx )
   END_RUNG wire#w2
   // the same network as SCL:
   #OK_Avance := "DB902_Estado_ZonaMesa".EstadoMesas[#Mesa].Marcha_CBx AND NOT "DB900_Estado_Mesas".EstadoVI[#Mesa].Error_Mx AND (#Termico_Tx OR ("DB902_Estado_ZonaMesa".EstadoMesas[#Mesa].Rearme_CBx AND #PhsMx)) AND #ok_tension;
END_REGION

REGION Network 6: Tiempo Centrado carga
   RUNG wire#powerrail
      "FC912_CNT_Tiempo_Mem_UHS"(Temporizar := wire#w1, Reset := wire#w2, Valor_Tiempo := #V_CNT_pHsMx, Base_tiempo_ms := 1, Valor_Actual := "DB230_CONTADORES".Mesa[#Mesa].CNT_PRESENCIA, Tiempo_OK => #Mem_CNT_Centrado)
   END_RUNG
   RUNG wire#powerrail
      Contact( #OK_Avance )
      Contact( #PhsMx )
      Contact( #Avance_Tx )
   END_RUNG wire#w1
   RUNG wire#powerrail
      I_Contact( #PhsMx )
   END_RUNG wire#w2
   // the same network as SCL:
   "FC912_CNT_Tiempo_Mem_UHS"(Temporizar := #OK_Avance AND #PhsMx AND #Avance_Tx,
                           Reset := NOT #PhsMx,
                           Valor_Tiempo := #V_CNT_pHsMx,
                           Base_tiempo_ms := 1,
                           Valor_Actual := "DB230_CONTADORES".Mesa[#Mesa].CNT_PRESENCIA,
                           Tiempo_OK => #Mem_CNT_Centrado);
END_REGION

REGION Network 7: Tiempo Centrado carga
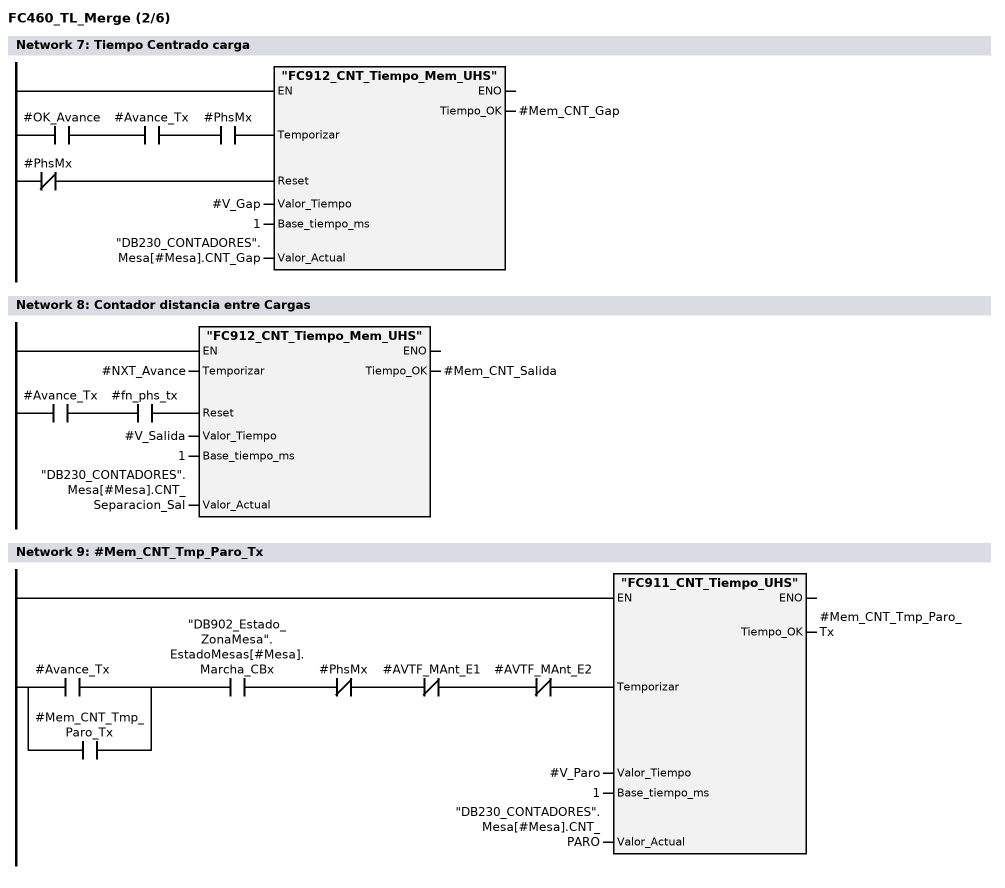
   RUNG wire#powerrail
      "FC912_CNT_Tiempo_Mem_UHS"(Temporizar := wire#w1, Reset := wire#w2, Valor_Tiempo := #V_Gap, Base_tiempo_ms := 1, Valor_Actual := "DB230_CONTADORES".Mesa[#Mesa].CNT_Gap, Tiempo_OK => #Mem_CNT_Gap)
   END_RUNG
   RUNG wire#powerrail
      Contact( #OK_Avance )
      Contact( #Avance_Tx )
      Contact( #PhsMx )
   END_RUNG wire#w1
   RUNG wire#powerrail
      I_Contact( #PhsMx )
   END_RUNG wire#w2
   // the same network as SCL:
   "FC912_CNT_Tiempo_Mem_UHS"(Temporizar := #OK_Avance AND #Avance_Tx AND #PhsMx,
                           Reset := NOT #PhsMx,
                           Valor_Tiempo := #V_Gap,
                           Base_tiempo_ms := 1,
                           Valor_Actual := "DB230_CONTADORES".Mesa[#Mesa].CNT_Gap,
                           Tiempo_OK => #Mem_CNT_Gap);
END_REGION

REGION Network 8: Contador distancia entre Cargas
   RUNG wire#powerrail
      "FC912_CNT_Tiempo_Mem_UHS"(Reset := wire#w1, Temporizar := #NXT_Avance, Valor_Tiempo := #V_Salida, Base_tiempo_ms := 1, Valor_Actual := "DB230_CONTADORES".Mesa[#Mesa].CNT_Separacion_Sal, Tiempo_OK => #Mem_CNT_Salida)
   END_RUNG
   RUNG wire#powerrail
      Contact( #Avance_Tx )
      Contact( #fn_phs_tx )
   END_RUNG wire#w1
   // the same network as SCL:
   "FC912_CNT_Tiempo_Mem_UHS"(Temporizar := #NXT_Avance,
                           Reset := #Avance_Tx AND #fn_phs_tx,
                           Valor_Tiempo := #V_Salida,
                           Base_tiempo_ms := 1,
                           Valor_Actual := "DB230_CONTADORES".Mesa[#Mesa].CNT_Separacion_Sal,
                           Tiempo_OK => #Mem_CNT_Salida);
END_REGION

REGION Network 9: #Mem_CNT_Tmp_Paro_Tx
   RUNG wire#powerrail
      "FC911_CNT_Tiempo_UHS"(Temporizar := wire#w2, Valor_Tiempo := #V_Paro, Base_tiempo_ms := 1, Valor_Actual := "DB230_CONTADORES".Mesa[#Mesa].CNT_PARO, Tiempo_OK => #Mem_CNT_Tmp_Paro_Tx)
   END_RUNG
   RUNG wire#powerrail
      Contact( #Avance_Tx )
      wire#w1
      Contact( "DB902_Estado_ZonaMesa".EstadoMesas[#Mesa].Marcha_CBx )
      I_Contact( #PhsMx )
      I_Contact( #AVTF_MAnt_E1 )
      I_Contact( #AVTF_MAnt_E2 )
   END_RUNG wire#w2
   RUNG wire#powerrail
      Contact( #Mem_CNT_Tmp_Paro_Tx )
   END_RUNG wire#w1
   // the same network as SCL:
   "FC911_CNT_Tiempo_UHS"(Temporizar := (#Avance_Tx OR #Mem_CNT_Tmp_Paro_Tx) AND "DB902_Estado_ZonaMesa".EstadoMesas[#Mesa].Marcha_CBx AND NOT #PhsMx AND NOT #AVTF_MAnt_E1 AND NOT #AVTF_MAnt_E2,
                          Valor_Tiempo := #V_Paro,
                          Base_tiempo_ms := 1,
                          Valor_Actual := "DB230_CONTADORES".Mesa[#Mesa].CNT_PARO,
                          Tiempo_OK => #Mem_CNT_Tmp_Paro_Tx);
END_REGION

REGION Network 10: #MA_AV_13_T_MX
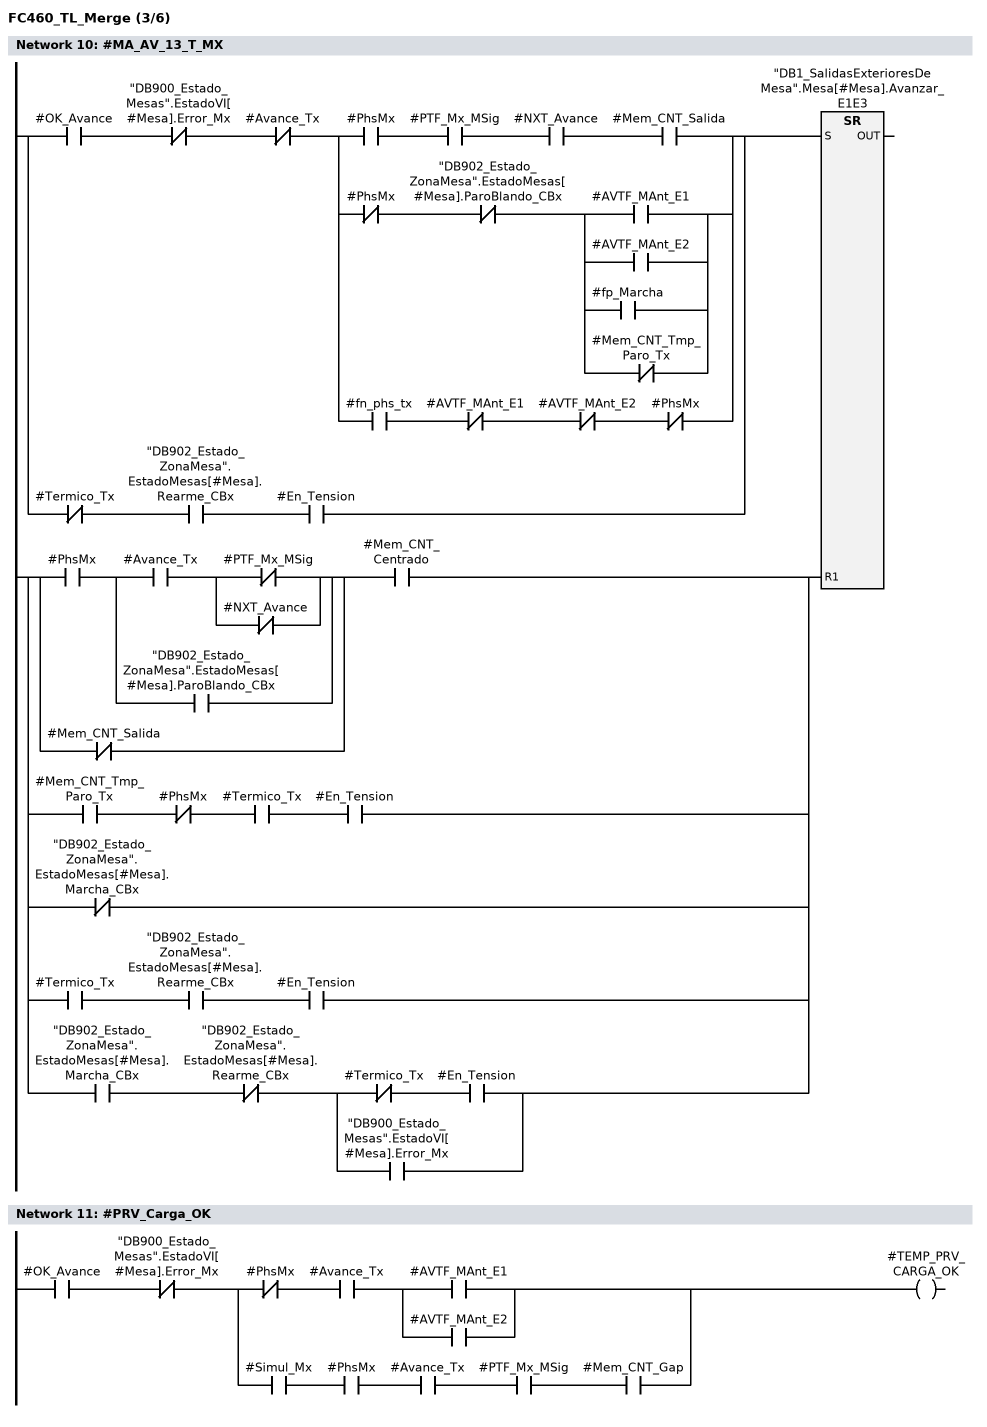
   RUNG wire#powerrail
      Contact( #OK_Avance )
      I_Contact( "DB900_Estado_Mesas".EstadoVI[#Mesa].Error_Mx )
      I_Contact( #Avance_Tx )
      wire#w1
      Contact( #PhsMx )
      Contact( #PTF_Mx_MSig )
      Contact( #NXT_Avance )
      Contact( #Mem_CNT_Salida )
      wire#w2
      S_SR(operand := "DB1_SalidasExterioresDeMesa".Mesa[#Mesa].Avanzar_E1E3, r1 := wire#w8)
   END_RUNG
   RUNG wire#w1
      I_Contact( #PhsMx )
      I_Contact( "DB902_Estado_ZonaMesa".EstadoMesas[#Mesa].ParoBlando_CBx )
      wire#w3
      Contact( #AVTF_MAnt_E1 )
   END_RUNG wire#w2
   RUNG wire#w3
      Contact( #AVTF_MAnt_E2 )
   END_RUNG wire#w2
   RUNG wire#w3
      Contact( #fp_Marcha )
   END_RUNG wire#w2
   RUNG wire#w3
      I_Contact( #Mem_CNT_Tmp_Paro_Tx )
   END_RUNG wire#w2
   RUNG wire#w1
      Contact( #fn_phs_tx )
      I_Contact( #AVTF_MAnt_E1 )
      I_Contact( #AVTF_MAnt_E2 )
      I_Contact( #PhsMx )
   END_RUNG wire#w2
   RUNG wire#powerrail
      I_Contact( #Termico_Tx )
      Contact( "DB902_Estado_ZonaMesa".EstadoMesas[#Mesa].Rearme_CBx )
      Contact( #En_Tension )
   END_RUNG wire#w2
   RUNG wire#powerrail
      Contact( #PhsMx )
      wire#w4
      Contact( #Avance_Tx )
      wire#w5
      I_Contact( #PTF_Mx_MSig )
      wire#w6
      Contact( #Mem_CNT_Centrado )
   END_RUNG wire#w8
   RUNG wire#w5
      I_Contact( #NXT_Avance )
   END_RUNG wire#w6
   RUNG wire#w4
      Contact( "DB902_Estado_ZonaMesa".EstadoMesas[#Mesa].ParoBlando_CBx )
   END_RUNG wire#w6
   RUNG wire#powerrail
      I_Contact( #Mem_CNT_Salida )
   END_RUNG wire#w6
   RUNG wire#powerrail
      Contact( #Mem_CNT_Tmp_Paro_Tx )
      I_Contact( #PhsMx )
      Contact( #Termico_Tx )
      Contact( #En_Tension )
   END_RUNG wire#w8
   RUNG wire#powerrail
      I_Contact( "DB902_Estado_ZonaMesa".EstadoMesas[#Mesa].Marcha_CBx )
   END_RUNG wire#w8
   RUNG wire#powerrail
      Contact( #Termico_Tx )
      Contact( "DB902_Estado_ZonaMesa".EstadoMesas[#Mesa].Rearme_CBx )
      Contact( #En_Tension )
   END_RUNG wire#w8
   RUNG wire#powerrail
      Contact( "DB902_Estado_ZonaMesa".EstadoMesas[#Mesa].Marcha_CBx )
      I_Contact( "DB902_Estado_ZonaMesa".EstadoMesas[#Mesa].Rearme_CBx )
      wire#w7
      I_Contact( #Termico_Tx )
      Contact( #En_Tension )
   END_RUNG wire#w8
   RUNG wire#w7
      Contact( "DB900_Estado_Mesas".EstadoVI[#Mesa].Error_Mx )
   END_RUNG wire#w8
   // the same network as SCL:
   #_w1 := (((#PhsMx AND ((#Avance_Tx AND (NOT #PTF_Mx_MSig OR NOT #NXT_Avance)) OR "DB902_Estado_ZonaMesa".EstadoMesas[#Mesa].ParoBlando_CBx)) OR NOT #Mem_CNT_Salida) AND #Mem_CNT_Centrado) OR (#Mem_CNT_Tmp_Paro_Tx AND NOT #PhsMx AND #Termico_Tx AND #En_Tension) OR NOT "DB902_Estado_ZonaMesa".EstadoMesas[#Mesa].Marcha_CBx OR (#Termico_Tx AND "DB902_Estado_ZonaMesa".EstadoMesas[#Mesa].Rearme_CBx AND #En_Tension) OR ("DB902_Estado_ZonaMesa".EstadoMesas[#Mesa].Marcha_CBx AND NOT "DB902_Estado_ZonaMesa".EstadoMesas[#Mesa].Rearme_CBx AND ((NOT #Termico_Tx AND #En_Tension) OR "DB900_Estado_Mesas".EstadoVI[#Mesa].Error_Mx));
   IF (#OK_Avance AND NOT "DB900_Estado_Mesas".EstadoVI[#Mesa].Error_Mx AND NOT #Avance_Tx AND ((#PhsMx AND #PTF_Mx_MSig AND #NXT_Avance AND #Mem_CNT_Salida) OR (NOT #PhsMx AND NOT "DB902_Estado_ZonaMesa".EstadoMesas[#Mesa].ParoBlando_CBx AND (#AVTF_MAnt_E1 OR #AVTF_MAnt_E2 OR #fp_Marcha OR NOT #Mem_CNT_Tmp_Paro_Tx)) OR (#fn_phs_tx AND NOT #AVTF_MAnt_E1 AND NOT #AVTF_MAnt_E2 AND NOT #PhsMx))) OR (NOT #Termico_Tx AND "DB902_Estado_ZonaMesa".EstadoMesas[#Mesa].Rearme_CBx AND #En_Tension) THEN
       "DB1_SalidasExterioresDeMesa".Mesa[#Mesa].Avanzar_E1E3 := TRUE;   // SR flip-flop
   END_IF;
   IF #_w1 THEN "DB1_SalidasExterioresDeMesa".Mesa[#Mesa].Avanzar_E1E3 := FALSE; END_IF;
END_REGION

REGION Network 11: #PRV_Carga_OK
   RUNG wire#powerrail
      Contact( #OK_Avance )
      I_Contact( "DB900_Estado_Mesas".EstadoVI[#Mesa].Error_Mx )
      wire#w1
      I_Contact( #PhsMx )
      Contact( #Avance_Tx )
      wire#w2
      Contact( #AVTF_MAnt_E1 )
      wire#w3
      Coil( #TEMP_PRV_CARGA_OK )
   END_RUNG
   RUNG wire#w2
      Contact( #AVTF_MAnt_E2 )
   END_RUNG wire#w3
   RUNG wire#w1
      Contact( #Simul_Mx )
      Contact( #PhsMx )
      Contact( #Avance_Tx )
      Contact( #PTF_Mx_MSig )
      Contact( #Mem_CNT_Gap )
   END_RUNG wire#w3
   // the same network as SCL:
   #TEMP_PRV_CARGA_OK := #OK_Avance AND NOT "DB900_Estado_Mesas".EstadoVI[#Mesa].Error_Mx AND ((NOT #PhsMx AND #Avance_Tx AND (#AVTF_MAnt_E1 OR #AVTF_MAnt_E2)) OR (#Simul_Mx AND #PhsMx AND #Avance_Tx AND #PTF_Mx_MSig AND #Mem_CNT_Gap));
END_REGION

REGION Network 12: #NXT_AVTF
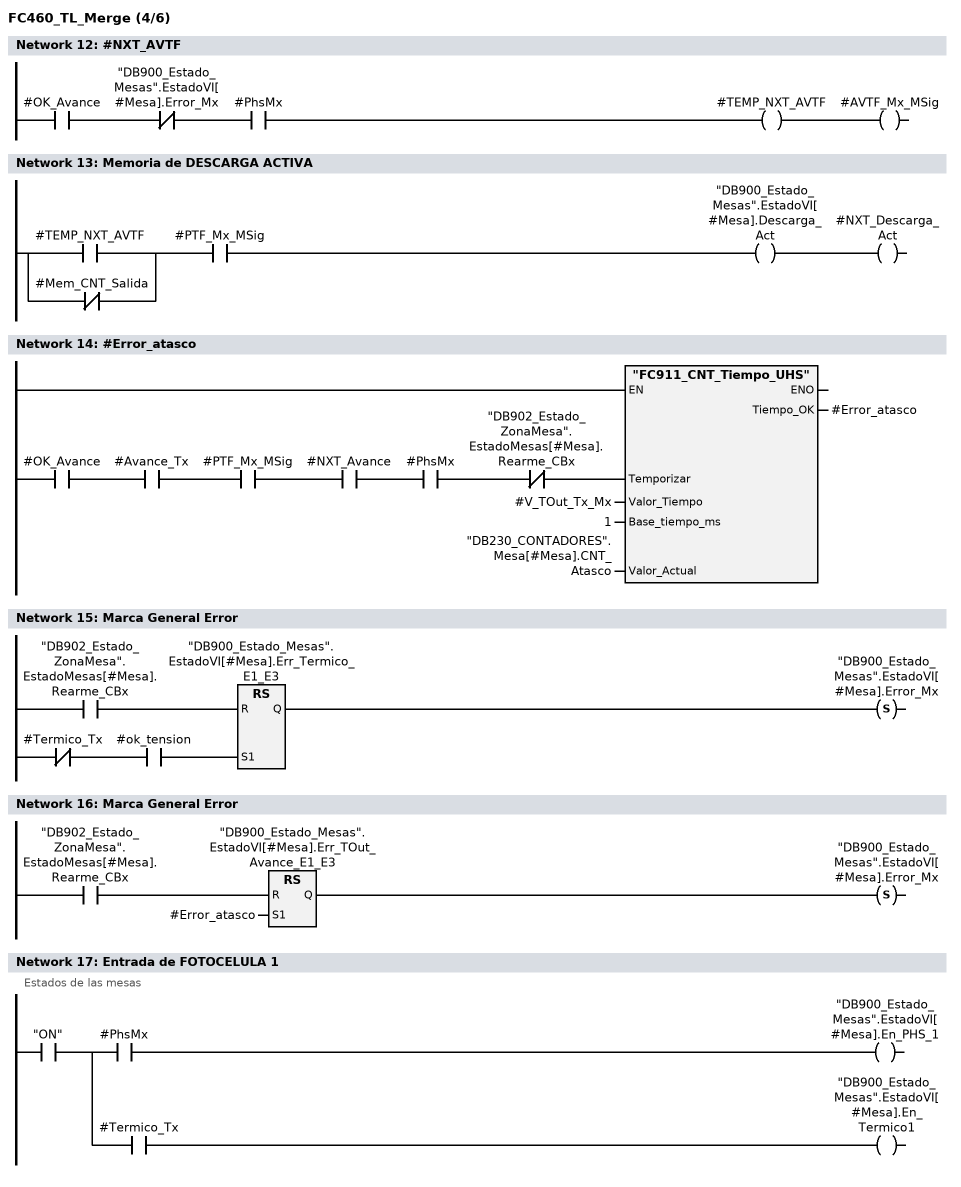
   RUNG wire#powerrail
      Contact( #OK_Avance )
      I_Contact( "DB900_Estado_Mesas".EstadoVI[#Mesa].Error_Mx )
      Contact( #PhsMx )
      Coil( #TEMP_NXT_AVTF )
      Coil( #AVTF_Mx_MSig )
   END_RUNG
   // the same network as SCL:
   #TEMP_NXT_AVTF := #OK_Avance AND NOT "DB900_Estado_Mesas".EstadoVI[#Mesa].Error_Mx AND #PhsMx;
   #AVTF_Mx_MSig := #TEMP_NXT_AVTF;
END_REGION

REGION Network 13: Memoria de DESCARGA ACTIVA
   RUNG wire#powerrail
      Contact( #TEMP_NXT_AVTF )
      wire#w1
      Contact( #PTF_Mx_MSig )
      Coil( "DB900_Estado_Mesas".EstadoVI[#Mesa].Descarga_Act )
      Coil( #NXT_Descarga_Act )
   END_RUNG
   RUNG wire#powerrail
      I_Contact( #Mem_CNT_Salida )
   END_RUNG wire#w1
   // the same network as SCL:
   "DB900_Estado_Mesas".EstadoVI[#Mesa].Descarga_Act := (#TEMP_NXT_AVTF OR NOT #Mem_CNT_Salida) AND #PTF_Mx_MSig;
   #NXT_Descarga_Act := (#TEMP_NXT_AVTF OR NOT #Mem_CNT_Salida) AND #PTF_Mx_MSig;
END_REGION

REGION Network 14: #Error_atasco
   RUNG wire#powerrail
      "FC911_CNT_Tiempo_UHS"(Temporizar := wire#w1, Valor_Tiempo := #V_TOut_Tx_Mx, Base_tiempo_ms := 1, Valor_Actual := "DB230_CONTADORES".Mesa[#Mesa].CNT_Atasco, Tiempo_OK => #Error_atasco)
   END_RUNG
   RUNG wire#powerrail
      Contact( #OK_Avance )
      Contact( #Avance_Tx )
      Contact( #PTF_Mx_MSig )
      Contact( #NXT_Avance )
      Contact( #PhsMx )
      I_Contact( "DB902_Estado_ZonaMesa".EstadoMesas[#Mesa].Rearme_CBx )
   END_RUNG wire#w1
   // the same network as SCL:
   "FC911_CNT_Tiempo_UHS"(Temporizar := #OK_Avance AND #Avance_Tx AND #PTF_Mx_MSig AND #NXT_Avance AND #PhsMx AND NOT "DB902_Estado_ZonaMesa".EstadoMesas[#Mesa].Rearme_CBx,
                          Valor_Tiempo := #V_TOut_Tx_Mx,
                          Base_tiempo_ms := 1,
                          Valor_Actual := "DB230_CONTADORES".Mesa[#Mesa].CNT_Atasco,
                          Tiempo_OK => #Error_atasco);
END_REGION

REGION Network 15: Marca General Error
   RUNG wire#powerrail
      Contact( "DB902_Estado_ZonaMesa".EstadoMesas[#Mesa].Rearme_CBx )
      S_RS(operand := "DB900_Estado_Mesas".EstadoVI[#Mesa].Err_Termico_E1_E3, s1 := wire#w1)
      S_Coil( "DB900_Estado_Mesas".EstadoVI[#Mesa].Error_Mx )
   END_RUNG
   RUNG wire#powerrail
      I_Contact( #Termico_Tx )
      Contact( #ok_tension )
   END_RUNG wire#w1
   // the same network as SCL:
   IF "DB902_Estado_ZonaMesa".EstadoMesas[#Mesa].Rearme_CBx THEN
       "DB900_Estado_Mesas".EstadoVI[#Mesa].Err_Termico_E1_E3 := FALSE;   // RS flip-flop
   END_IF;
   IF NOT #Termico_Tx AND #ok_tension THEN
       "DB900_Estado_Mesas".EstadoVI[#Mesa].Err_Termico_E1_E3 := TRUE;
   END_IF;
   IF "DB900_Estado_Mesas".EstadoVI[#Mesa].Err_Termico_E1_E3 THEN
       "DB900_Estado_Mesas".EstadoVI[#Mesa].Error_Mx := TRUE;
   END_IF;
END_REGION

REGION Network 16: Marca General Error
   RUNG wire#powerrail
      Contact( "DB902_Estado_ZonaMesa".EstadoMesas[#Mesa].Rearme_CBx )
      S_RS(operand := "DB900_Estado_Mesas".EstadoVI[#Mesa].Err_TOut_Avance_E1_E3, s1 := #Error_atasco)
      S_Coil( "DB900_Estado_Mesas".EstadoVI[#Mesa].Error_Mx )
   END_RUNG
   // the same network as SCL:
   IF "DB902_Estado_ZonaMesa".EstadoMesas[#Mesa].Rearme_CBx THEN
       "DB900_Estado_Mesas".EstadoVI[#Mesa].Err_TOut_Avance_E1_E3 := FALSE;   // RS flip-flop
   END_IF;
   IF #Error_atasco THEN "DB900_Estado_Mesas".EstadoVI[#Mesa].Err_TOut_Avance_E1_E3 := TRUE; END_IF;
   IF "DB900_Estado_Mesas".EstadoVI[#Mesa].Err_TOut_Avance_E1_E3 THEN
       "DB900_Estado_Mesas".EstadoVI[#Mesa].Error_Mx := TRUE;
   END_IF;
END_REGION

REGION Network 17: Entrada de FOTOCELULA 1
   // Estados de las mesas
   RUNG wire#powerrail
      Contact( "ON" )
      wire#w1
      Contact( #PhsMx )
      Coil( "DB900_Estado_Mesas".EstadoVI[#Mesa].En_PHS_1 )
   END_RUNG
   RUNG wire#w1
      Contact( #Termico_Tx )
      Coil( "DB900_Estado_Mesas".EstadoVI[#Mesa].En_Termico1 )
   END_RUNG
   // the same network as SCL:
   "DB900_Estado_Mesas".EstadoVI[#Mesa].En_PHS_1 := "ON" AND #PhsMx;
   "DB900_Estado_Mesas".EstadoVI[#Mesa].En_Termico1 := "ON" AND #Termico_Tx;
END_REGION

REGION Network 18: ESTADOS MESA 1
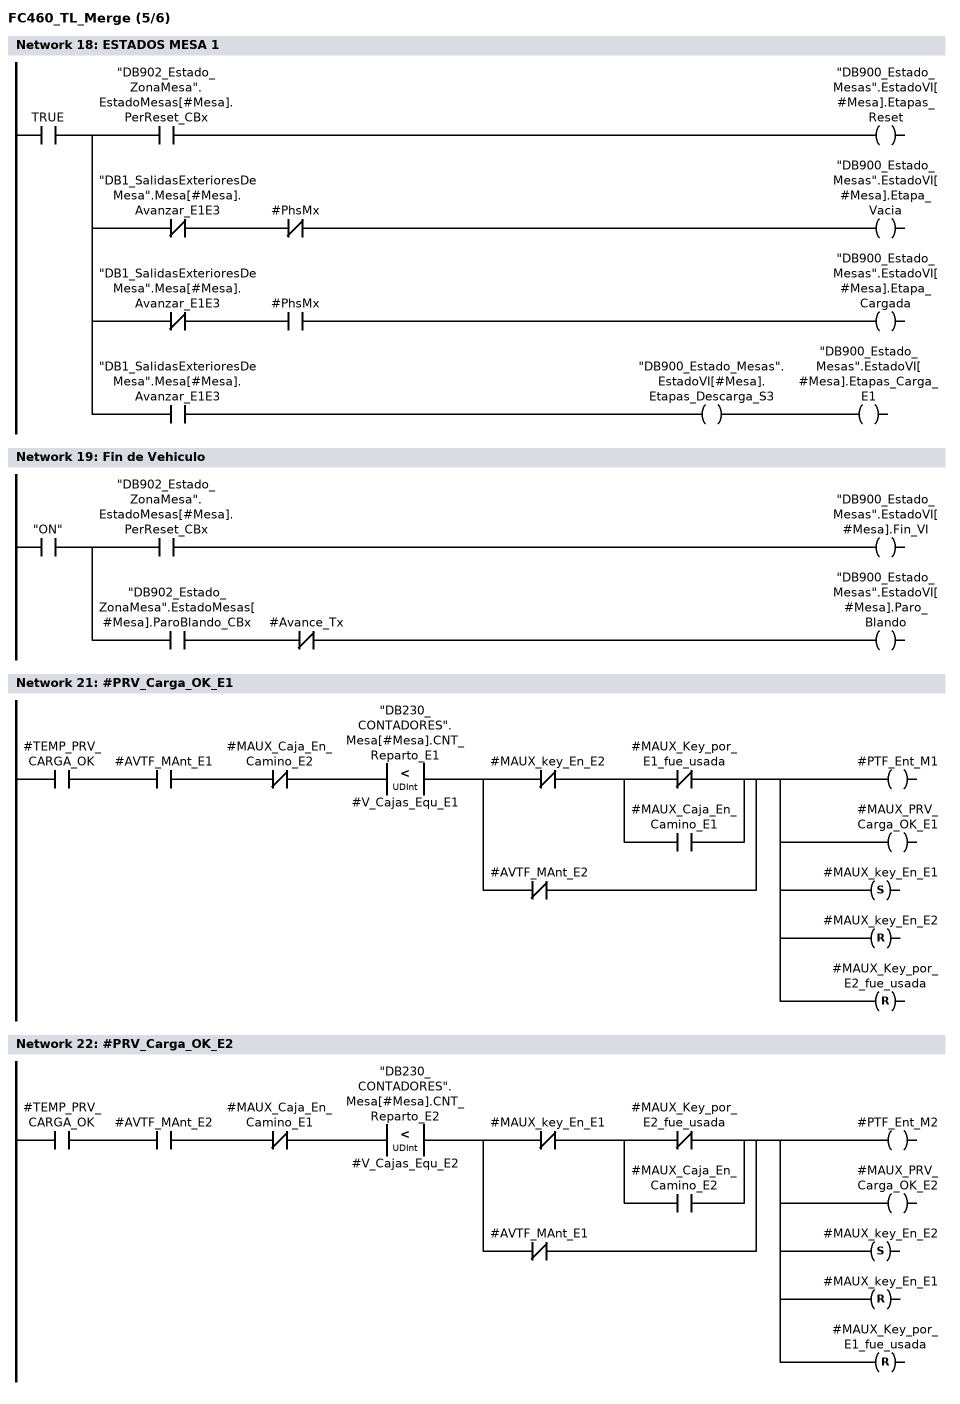
   RUNG wire#powerrail
      Contact( TRUE )
      wire#w1
      Contact( "DB902_Estado_ZonaMesa".EstadoMesas[#Mesa].PerReset_CBx )
      Coil( "DB900_Estado_Mesas".EstadoVI[#Mesa].Etapas_Reset )
   END_RUNG
   RUNG wire#w1
      I_Contact( "DB1_SalidasExterioresDeMesa".Mesa[#Mesa].Avanzar_E1E3 )
      I_Contact( #PhsMx )
      Coil( "DB900_Estado_Mesas".EstadoVI[#Mesa].Etapa_Vacia )
   END_RUNG
   RUNG wire#w1
      I_Contact( "DB1_SalidasExterioresDeMesa".Mesa[#Mesa].Avanzar_E1E3 )
      Contact( #PhsMx )
      Coil( "DB900_Estado_Mesas".EstadoVI[#Mesa].Etapa_Cargada )
   END_RUNG
   RUNG wire#w1
      Contact( "DB1_SalidasExterioresDeMesa".Mesa[#Mesa].Avanzar_E1E3 )
      Coil( "DB900_Estado_Mesas".EstadoVI[#Mesa].Etapas_Descarga_S3 )
      Coil( "DB900_Estado_Mesas".EstadoVI[#Mesa].Etapas_Carga_E1 )
   END_RUNG
   // the same network as SCL:
   "DB900_Estado_Mesas".EstadoVI[#Mesa].Etapas_Reset := TRUE AND "DB902_Estado_ZonaMesa".EstadoMesas[#Mesa].PerReset_CBx;
   "DB900_Estado_Mesas".EstadoVI[#Mesa].Etapa_Vacia := TRUE AND NOT "DB1_SalidasExterioresDeMesa".Mesa[#Mesa].Avanzar_E1E3 AND NOT #PhsMx;
   "DB900_Estado_Mesas".EstadoVI[#Mesa].Etapa_Cargada := TRUE AND NOT "DB1_SalidasExterioresDeMesa".Mesa[#Mesa].Avanzar_E1E3 AND #PhsMx;
   #_w1 := TRUE AND "DB1_SalidasExterioresDeMesa".Mesa[#Mesa].Avanzar_E1E3;
   "DB900_Estado_Mesas".EstadoVI[#Mesa].Etapas_Descarga_S3 := #_w1;
   "DB900_Estado_Mesas".EstadoVI[#Mesa].Etapas_Carga_E1 := #_w1;
END_REGION

REGION Network 19: Fin de Vehiculo
   RUNG wire#powerrail
      Contact( "ON" )
      wire#w1
      Contact( "DB902_Estado_ZonaMesa".EstadoMesas[#Mesa].PerReset_CBx )
      Coil( "DB900_Estado_Mesas".EstadoVI[#Mesa].Fin_VI )
   END_RUNG
   RUNG wire#w1
      Contact( "DB902_Estado_ZonaMesa".EstadoMesas[#Mesa].ParoBlando_CBx )
      I_Contact( #Avance_Tx )
      Coil( "DB900_Estado_Mesas".EstadoVI[#Mesa].Paro_Blando )
   END_RUNG
   // the same network as SCL:
   "DB900_Estado_Mesas".EstadoVI[#Mesa].Fin_VI := "ON" AND "DB902_Estado_ZonaMesa".EstadoMesas[#Mesa].PerReset_CBx;
   "DB900_Estado_Mesas".EstadoVI[#Mesa].Paro_Blando := "ON" AND "DB902_Estado_ZonaMesa".EstadoMesas[#Mesa].ParoBlando_CBx AND NOT #Avance_Tx;
END_REGION

REGION Network 20: Gestion de cruce
END_REGION

REGION Network 21: #PRV_Carga_OK_E1
   RUNG wire#powerrail
      Contact( #TEMP_PRV_CARGA_OK )
      Contact( #AVTF_MAnt_E1 )
      I_Contact( #MAUX_Caja_En_Camino_E2 )
      { S7_Templates := "SrcType := UDInt" } LT_Contact(in1 := "DB230_CONTADORES".Mesa[#Mesa].CNT_Reparto_E1, in2 := #V_Cajas_Equ_E1)
      wire#w1
      I_Contact( #MAUX_key_En_E2 )
      wire#w2
      I_Contact( #MAUX_Key_por_E1_fue_usada )
      wire#w3
      Coil( #PTF_Ent_M1 )
   END_RUNG
   RUNG wire#w2
      Contact( #MAUX_Caja_En_Camino_E1 )
   END_RUNG wire#w3
   RUNG wire#w1
      I_Contact( #AVTF_MAnt_E2 )
   END_RUNG wire#w3
   RUNG wire#w3
      Coil( #MAUX_PRV_Carga_OK_E1 )
   END_RUNG
   RUNG wire#w3
      S_Coil( #MAUX_key_En_E1 )
   END_RUNG
   RUNG wire#w3
      R_Coil( #MAUX_key_En_E2 )
   END_RUNG
   RUNG wire#w3
      R_Coil( #MAUX_Key_por_E2_fue_usada )
   END_RUNG
   // the same network as SCL:
   #PTF_Ent_M1 := #TEMP_PRV_CARGA_OK AND #AVTF_MAnt_E1 AND NOT #MAUX_Caja_En_Camino_E2 AND ("DB230_CONTADORES".Mesa[#Mesa].CNT_Reparto_E1 < #V_Cajas_Equ_E1) AND ((NOT #MAUX_key_En_E2 AND (NOT #MAUX_Key_por_E1_fue_usada OR #MAUX_Caja_En_Camino_E1)) OR NOT #AVTF_MAnt_E2);
   #MAUX_PRV_Carga_OK_E1 := #PTF_Ent_M1;
   IF #PTF_Ent_M1 THEN
       #MAUX_key_En_E1 := TRUE;
       #MAUX_key_En_E2 := FALSE;
       #MAUX_Key_por_E2_fue_usada := FALSE;
   END_IF;
END_REGION

REGION Network 22: #PRV_Carga_OK_E2
   RUNG wire#powerrail
      Contact( #TEMP_PRV_CARGA_OK )
      Contact( #AVTF_MAnt_E2 )
      I_Contact( #MAUX_Caja_En_Camino_E1 )
      { S7_Templates := "SrcType := UDInt" } LT_Contact(in1 := "DB230_CONTADORES".Mesa[#Mesa].CNT_Reparto_E2, in2 := #V_Cajas_Equ_E2)
      wire#w1
      I_Contact( #MAUX_key_En_E1 )
      wire#w2
      I_Contact( #MAUX_Key_por_E2_fue_usada )
      wire#w3
      Coil( #PTF_Ent_M2 )
   END_RUNG
   RUNG wire#w2
      Contact( #MAUX_Caja_En_Camino_E2 )
   END_RUNG wire#w3
   RUNG wire#w1
      I_Contact( #AVTF_MAnt_E1 )
   END_RUNG wire#w3
   RUNG wire#w3
      Coil( #MAUX_PRV_Carga_OK_E2 )
   END_RUNG
   RUNG wire#w3
      S_Coil( #MAUX_key_En_E2 )
   END_RUNG
   RUNG wire#w3
      R_Coil( #MAUX_key_En_E1 )
   END_RUNG
   RUNG wire#w3
      R_Coil( #MAUX_Key_por_E1_fue_usada )
   END_RUNG
   // the same network as SCL:
   #PTF_Ent_M2 := #TEMP_PRV_CARGA_OK AND #AVTF_MAnt_E2 AND NOT #MAUX_Caja_En_Camino_E1 AND ("DB230_CONTADORES".Mesa[#Mesa].CNT_Reparto_E2 < #V_Cajas_Equ_E2) AND ((NOT #MAUX_key_En_E1 AND (NOT #MAUX_Key_por_E2_fue_usada OR #MAUX_Caja_En_Camino_E2)) OR NOT #AVTF_MAnt_E1);
   #MAUX_PRV_Carga_OK_E2 := #PTF_Ent_M2;
   IF #PTF_Ent_M2 THEN
       #MAUX_key_En_E2 := TRUE;
       #MAUX_key_En_E1 := FALSE;
       #MAUX_Key_por_E1_fue_usada := FALSE;
   END_IF;
END_REGION

NETWORK
TITLE = Contador de cajas permitidas por E1
      A     #MAUX_PRV_Carga_OK_E1;
      FN    #MAUX_FP_contador_E1;
      JCN   cont1;

      L     "DB230_CONTADORES".Mesa[#Mesa].CNT_Reparto_E1;
      L     1;
      +I;
      T     "DB230_CONTADORES".Mesa[#Mesa].CNT_Reparto_E1;
//si no hay aviso de transferencia por E2, entonces se deja entrar otra vez por E1. Aunque ya se haya cumplido el
//contador. y si eso sucede, se tiene que resetear el key usada, de lo contrario, no dejariamos entrar de nnuevo
      R     #MAUX_Key_por_E1_fue_usada;

cont1:NOP   0;

      A     #MAUX_PRV_Carga_OK_E2;
      FN    #MAUX_FP_contador_E2;
      JCN   cont2;

      L     "DB230_CONTADORES".Mesa[#Mesa].CNT_Reparto_E2;
      L     1;
      +I;
      T     "DB230_CONTADORES".Mesa[#Mesa].CNT_Reparto_E2;
//si no hay aviso de transferencia por E2, entonces se deja entrar otra vez por E1. Aunque ya se haya cumplido el
//contador. y si eso sucede, se tiene que resetear el key usada, de lo contrario, no dejariamos entrar de nnuevo
      R     #MAUX_Key_por_E2_fue_usada;



cont2:NOP   0;

//llegando al maximo tenemos que resetear el valor
      L     "DB230_CONTADORES".Mesa[#Mesa].CNT_Reparto_E1;
      L     #V_Cajas_Equ_E1;
      >=I;
      JCN   borr1;
      L     0;
      T     "DB230_CONTADORES".Mesa[#Mesa].CNT_Reparto_E1;

      R     #MAUX_key_En_E1;
      S     #MAUX_Key_por_E1_fue_usada;
borr1:NOP   0;

//llegando al maximo tenemos que resetear el valor
      L     "DB230_CONTADORES".Mesa[#Mesa].CNT_Reparto_E2;
      L     #V_Cajas_Equ_E2;
      >=I;
      JCN   borr2;
      L     0;
      T     "DB230_CONTADORES".Mesa[#Mesa].CNT_Reparto_E2;

      R     #MAUX_key_En_E2;
      S     #MAUX_Key_por_E2_fue_usada;
borr2:NOP   0;





REGION Network 24: Caja en caminno por E1. Nada puede entrar por E2
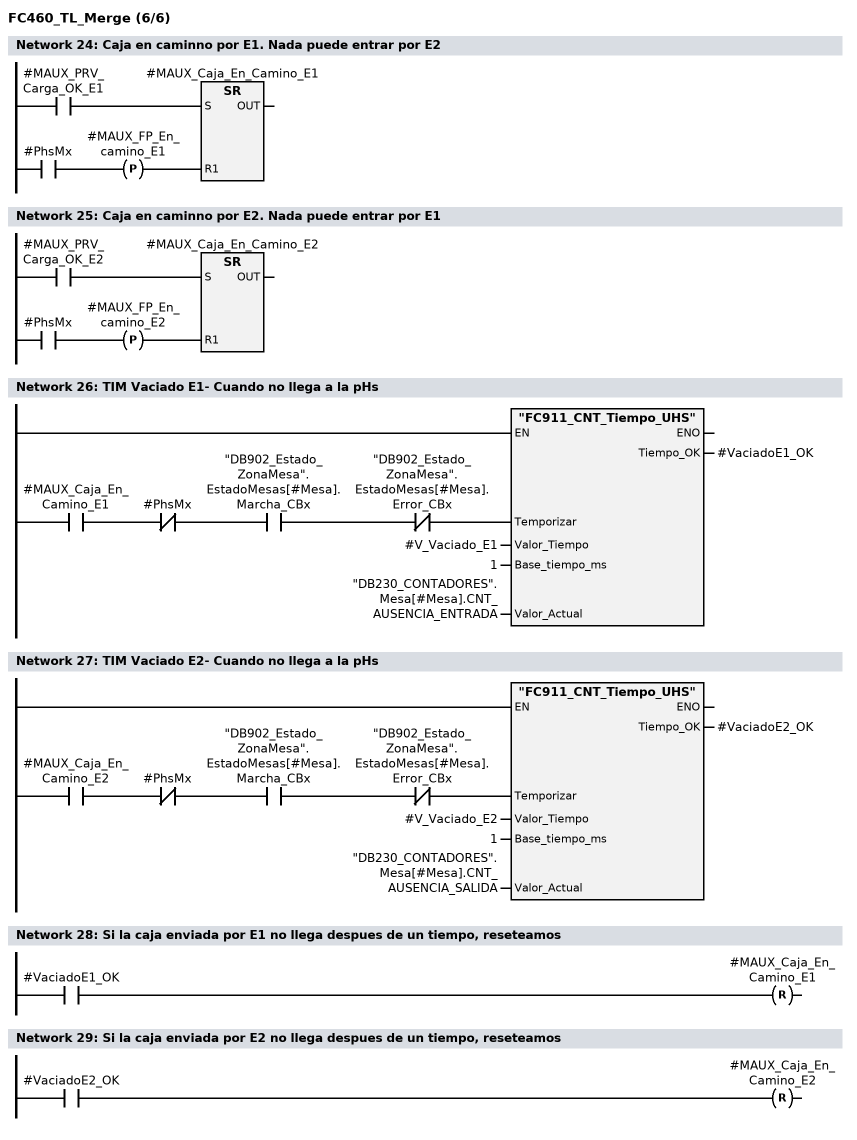
   RUNG wire#powerrail
      Contact( #MAUX_PRV_Carga_OK_E1 )
      S_SR(operand := #MAUX_Caja_En_Camino_E1, r1 := wire#w1)
   END_RUNG
   RUNG wire#powerrail
      Contact( #PhsMx )
      P_Trig( #MAUX_FP_En_camino_E1 )
   END_RUNG wire#w1
   // the same network as SCL:
   #_w1 := #PhsMx AND NOT #MAUX_FP_En_camino_E1;   // rising edge
   #MAUX_FP_En_camino_E1 := #PhsMx;
   IF #MAUX_PRV_Carga_OK_E1 THEN
       #MAUX_Caja_En_Camino_E1 := TRUE;   // SR flip-flop
   END_IF;
   IF #_w1 THEN #MAUX_Caja_En_Camino_E1 := FALSE; END_IF;
END_REGION

REGION Network 25: Caja en caminno por E2. Nada puede entrar por E1
   RUNG wire#powerrail
      Contact( #MAUX_PRV_Carga_OK_E2 )
      S_SR(operand := #MAUX_Caja_En_Camino_E2, r1 := wire#w1)
   END_RUNG
   RUNG wire#powerrail
      Contact( #PhsMx )
      P_Trig( #MAUX_FP_En_camino_E2 )
   END_RUNG wire#w1
   // the same network as SCL:
   #_w1 := #PhsMx AND NOT #MAUX_FP_En_camino_E2;   // rising edge
   #MAUX_FP_En_camino_E2 := #PhsMx;
   IF #MAUX_PRV_Carga_OK_E2 THEN
       #MAUX_Caja_En_Camino_E2 := TRUE;   // SR flip-flop
   END_IF;
   IF #_w1 THEN #MAUX_Caja_En_Camino_E2 := FALSE; END_IF;
END_REGION

REGION Network 26: TIM Vaciado E1- Cuando no llega a la pHs
   RUNG wire#powerrail
      "FC911_CNT_Tiempo_UHS"(Temporizar := wire#w1, Valor_Tiempo := #V_Vaciado_E1, Base_tiempo_ms := 1, Valor_Actual := "DB230_CONTADORES".Mesa[#Mesa].CNT_AUSENCIA_ENTRADA, Tiempo_OK => #VaciadoE1_OK)
   END_RUNG
   RUNG wire#powerrail
      Contact( #MAUX_Caja_En_Camino_E1 )
      I_Contact( #PhsMx )
      Contact( "DB902_Estado_ZonaMesa".EstadoMesas[#Mesa].Marcha_CBx )
      I_Contact( "DB902_Estado_ZonaMesa".EstadoMesas[#Mesa].Error_CBx )
   END_RUNG wire#w1
   // the same network as SCL:
   "FC911_CNT_Tiempo_UHS"(Temporizar := #MAUX_Caja_En_Camino_E1 AND NOT #PhsMx AND "DB902_Estado_ZonaMesa".EstadoMesas[#Mesa].Marcha_CBx AND NOT "DB902_Estado_ZonaMesa".EstadoMesas[#Mesa].Error_CBx,
                          Valor_Tiempo := #V_Vaciado_E1,
                          Base_tiempo_ms := 1,
                          Valor_Actual := "DB230_CONTADORES".Mesa[#Mesa].CNT_AUSENCIA_ENTRADA,
                          Tiempo_OK => #VaciadoE1_OK);
END_REGION

REGION Network 27: TIM Vaciado E2- Cuando no llega a la pHs
   RUNG wire#powerrail
      "FC911_CNT_Tiempo_UHS"(Temporizar := wire#w1, Valor_Tiempo := #V_Vaciado_E2, Base_tiempo_ms := 1, Valor_Actual := "DB230_CONTADORES".Mesa[#Mesa].CNT_AUSENCIA_SALIDA, Tiempo_OK => #VaciadoE2_OK)
   END_RUNG
   RUNG wire#powerrail
      Contact( #MAUX_Caja_En_Camino_E2 )
      I_Contact( #PhsMx )
      Contact( "DB902_Estado_ZonaMesa".EstadoMesas[#Mesa].Marcha_CBx )
      I_Contact( "DB902_Estado_ZonaMesa".EstadoMesas[#Mesa].Error_CBx )
   END_RUNG wire#w1
   // the same network as SCL:
   "FC911_CNT_Tiempo_UHS"(Temporizar := #MAUX_Caja_En_Camino_E2 AND NOT #PhsMx AND "DB902_Estado_ZonaMesa".EstadoMesas[#Mesa].Marcha_CBx AND NOT "DB902_Estado_ZonaMesa".EstadoMesas[#Mesa].Error_CBx,
                          Valor_Tiempo := #V_Vaciado_E2,
                          Base_tiempo_ms := 1,
                          Valor_Actual := "DB230_CONTADORES".Mesa[#Mesa].CNT_AUSENCIA_SALIDA,
                          Tiempo_OK => #VaciadoE2_OK);
END_REGION

REGION Network 28: Si la caja enviada por E1 no llega despues de un tiempo, reseteamos
   RUNG wire#powerrail
      Contact( #VaciadoE1_OK )
      R_Coil( #MAUX_Caja_En_Camino_E1 )
   END_RUNG
   // the same network as SCL:
   IF #VaciadoE1_OK THEN #MAUX_Caja_En_Camino_E1 := FALSE; END_IF;
END_REGION

REGION Network 29: Si la caja enviada por E2 no llega despues de un tiempo, reseteamos
   RUNG wire#powerrail
      Contact( #VaciadoE2_OK )
      R_Coil( #MAUX_Caja_En_Camino_E2 )
   END_RUNG
   // the same network as SCL:
   IF #VaciadoE2_OK THEN #MAUX_Caja_En_Camino_E2 := FALSE; END_IF;
END_REGION
END_FUNCTION

FUNCTION "FC465_Elevador_Continuo_Building" : Void   // FC465, LAD
TITLE = ELEVADOR CONTINUO
{ S7_Optimized_Access := 'FALSE' }
VERSION : 1.0
// Control para un elevador continuo con una única entrada y una única salida. si requiere de más salidas es necesario aplicar otro control para el movimiento y para el transportador abatible
// stored: AutoNumber false, SetENOAutomatically false
   VAR_INPUT
      NumeroMesa : UInt;
      NumeroMesaEntrada : UInt;
      NumeroMesaSalida : UInt;
      Termico_TEnt : Bool;
      Termico_TSal : Bool;
      Termico_Elev : Bool;
      pHs_Ent : Bool;
      Prot_Ent : Bool;
      pHs_Sal : Bool;
      Prot_Sal : Bool;
      Det_Sincr_Entrada : Bool;
      Det_Salida_Paro : Bool;
      Det_Salida_Emerg : Bool;
      AVTF_Ant : Bool;
      PTF_Sig : Bool;
      V_Permiso_Entrada : UDInt;
      V_Presencia_Entrada : UDInt;
      V_Paro_Elev : UDInt;
      V_Paro_Sal_ms : UDInt;
   END_VAR
   VAR_IN_OUT
      MAux_FP_Sincr : Bool;
      MAux_FN_Entrada : Bool;
      MAux_FP_Salida : Bool;
      Mem_TmpParoSal : Bool;
      Mem_Paro_Elev : Bool;
      out_Elevacion : Bool;
      out_Avance_Ent : Bool;
      out_Avance_Sal : Bool;
      out_AVTF_Sig : Bool;
      out_Carga_OK_Ant : Bool;
      Mem_TmpPermEntrada : Bool;
      Mem_TmpCentradoEntrada : Bool;
      Mem_TmpParoElev : Bool;
   END_VAR
   VAR_TEMP   // added for the SCL form of the ladder/FBD networks
      _w1 : Bool;
      _w2 : Bool;
   END_VAR
BEGIN

REGION Network 1: Marca General Error
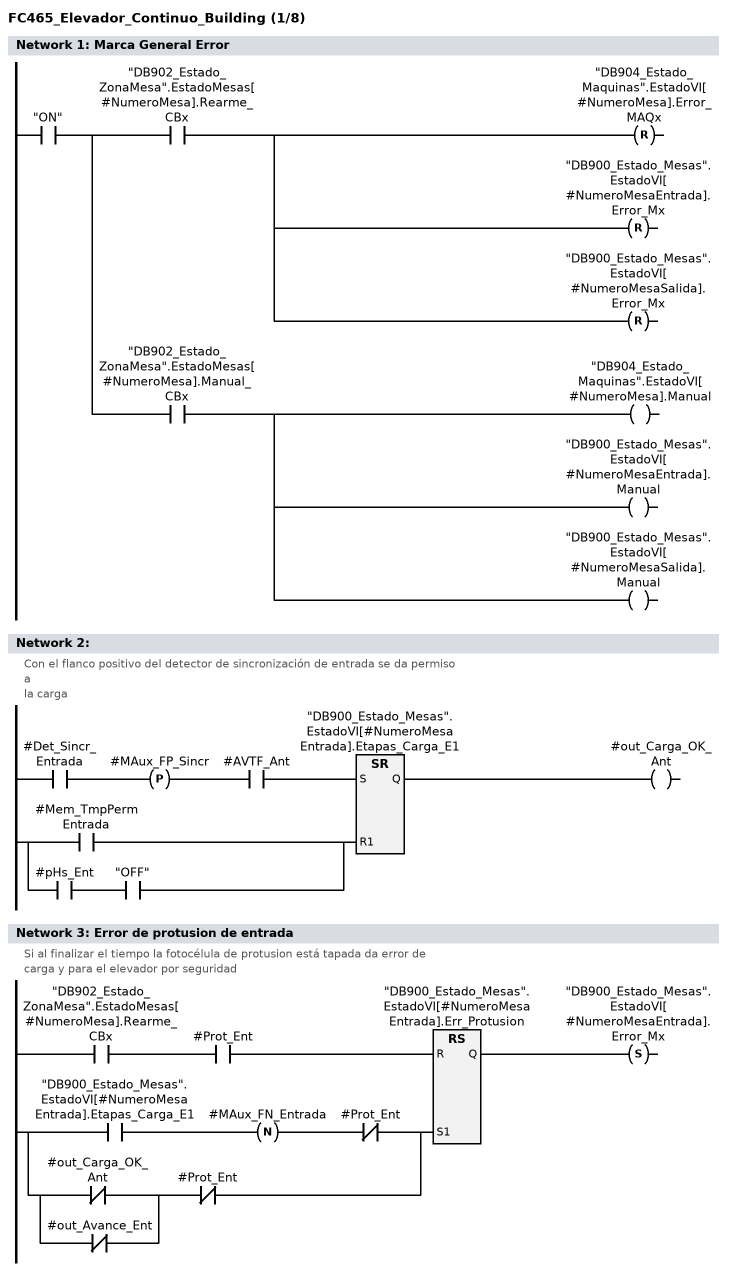
   RUNG wire#powerrail
      Contact( "ON" )
      wire#w1
      Contact( "DB902_Estado_ZonaMesa".EstadoMesas[#NumeroMesa].Rearme_CBx )
      wire#w2
      R_Coil( "DB904_Estado_Maquinas".EstadoVI[#NumeroMesa].Error_MAQx )
   END_RUNG
   RUNG wire#w2
      R_Coil( "DB900_Estado_Mesas".EstadoVI[#NumeroMesaEntrada].Error_Mx )
   END_RUNG
   RUNG wire#w2
      R_Coil( "DB900_Estado_Mesas".EstadoVI[#NumeroMesaSalida].Error_Mx )
   END_RUNG
   RUNG wire#w1
      Contact( "DB902_Estado_ZonaMesa".EstadoMesas[#NumeroMesa].Manual_CBx )
      wire#w3
      Coil( "DB904_Estado_Maquinas".EstadoVI[#NumeroMesa].Manual )
   END_RUNG
   RUNG wire#w3
      Coil( "DB900_Estado_Mesas".EstadoVI[#NumeroMesaEntrada].Manual )
   END_RUNG
   RUNG wire#w3
      Coil( "DB900_Estado_Mesas".EstadoVI[#NumeroMesaSalida].Manual )
   END_RUNG
   // the same network as SCL:
   #_w1 := "ON" AND "DB902_Estado_ZonaMesa".EstadoMesas[#NumeroMesa].Rearme_CBx;
   IF #_w1 THEN
       "DB904_Estado_Maquinas".EstadoVI[#NumeroMesa].Error_MAQx := FALSE;
       "DB900_Estado_Mesas".EstadoVI[#NumeroMesaEntrada].Error_Mx := FALSE;
       "DB900_Estado_Mesas".EstadoVI[#NumeroMesaSalida].Error_Mx := FALSE;
   END_IF;
   #_w2 := "ON" AND "DB902_Estado_ZonaMesa".EstadoMesas[#NumeroMesa].Manual_CBx;
   "DB904_Estado_Maquinas".EstadoVI[#NumeroMesa].Manual := "ON" AND "DB902_Estado_ZonaMesa".EstadoMesas[#NumeroMesa].Manual_CBx;
   "DB900_Estado_Mesas".EstadoVI[#NumeroMesaEntrada].Manual := #_w2;
   "DB900_Estado_Mesas".EstadoVI[#NumeroMesaSalida].Manual := #_w2;
END_REGION

REGION Network 2
   // Con el flanco positivo del detector de sincronización de entrada se da permiso 
   // a 
   // la carga
   RUNG wire#powerrail
      Contact( #Det_Sincr_Entrada )
      P_Trig( #MAux_FP_Sincr )
      Contact( #AVTF_Ant )
      S_SR(operand := "DB900_Estado_Mesas".EstadoVI[#NumeroMesaEntrada].Etapas_Carga_E1, r1 := wire#w1)
      Coil( #out_Carga_OK_Ant )
   END_RUNG
   RUNG wire#powerrail
      Contact( #Mem_TmpPermEntrada )
   END_RUNG wire#w1
   RUNG wire#powerrail
      Contact( #pHs_Ent )
      Contact( "OFF" )
   END_RUNG wire#w1
   // the same network as SCL:
   #_w1 := #Det_Sincr_Entrada AND NOT #MAux_FP_Sincr;   // rising edge
   #MAux_FP_Sincr := #Det_Sincr_Entrada;
   IF #_w1 AND #AVTF_Ant THEN
       "DB900_Estado_Mesas".EstadoVI[#NumeroMesaEntrada].Etapas_Carga_E1 := TRUE;   // SR flip-flop
   END_IF;
   IF #Mem_TmpPermEntrada OR (#pHs_Ent AND "OFF") THEN
       "DB900_Estado_Mesas".EstadoVI[#NumeroMesaEntrada].Etapas_Carga_E1 := FALSE;
   END_IF;
   #out_Carga_OK_Ant := "DB900_Estado_Mesas".EstadoVI[#NumeroMesaEntrada].Etapas_Carga_E1;
END_REGION

REGION Network 3: Error de protusion de entrada
   // Si al finalizar el tiempo la fotocélula de protusion está tapada da error de 
   // carga y para el elevador por seguridad
   RUNG wire#powerrail
      Contact( "DB902_Estado_ZonaMesa".EstadoMesas[#NumeroMesa].Rearme_CBx )
      Contact( #Prot_Ent )
      S_RS(operand := "DB900_Estado_Mesas".EstadoVI[#NumeroMesaEntrada].Err_Protusion, s1 := wire#w2)
      S_Coil( "DB900_Estado_Mesas".EstadoVI[#NumeroMesaEntrada].Error_Mx )
   END_RUNG
   RUNG wire#powerrail
      Contact( "DB900_Estado_Mesas".EstadoVI[#NumeroMesaEntrada].Etapas_Carga_E1 )
      N_Trig( #MAux_FN_Entrada )
      I_Contact( #Prot_Ent )
   END_RUNG wire#w2
   RUNG wire#powerrail
      I_Contact( #out_Carga_OK_Ant )
      wire#w1
      I_Contact( #Prot_Ent )
   END_RUNG wire#w2
   RUNG wire#powerrail
      I_Contact( #out_Avance_Ent )
   END_RUNG wire#w1
   // the same network as SCL:
   #_w1 := NOT "DB900_Estado_Mesas".EstadoVI[#NumeroMesaEntrada].Etapas_Carga_E1 AND #MAux_FN_Entrada;   // falling edge
   #MAux_FN_Entrada := "DB900_Estado_Mesas".EstadoVI[#NumeroMesaEntrada].Etapas_Carga_E1;
   IF "DB902_Estado_ZonaMesa".EstadoMesas[#NumeroMesa].Rearme_CBx AND #Prot_Ent THEN
       "DB900_Estado_Mesas".EstadoVI[#NumeroMesaEntrada].Err_Protusion := FALSE;   // RS flip-flop
   END_IF;
   IF (#_w1 AND NOT #Prot_Ent) OR ((NOT #out_Carga_OK_Ant OR NOT #out_Avance_Ent) AND NOT #Prot_Ent) THEN
       "DB900_Estado_Mesas".EstadoVI[#NumeroMesaEntrada].Err_Protusion := TRUE;
   END_IF;
   IF "DB900_Estado_Mesas".EstadoVI[#NumeroMesaEntrada].Err_Protusion THEN
       "DB900_Estado_Mesas".EstadoVI[#NumeroMesaEntrada].Error_Mx := TRUE;
   END_IF;
END_REGION

REGION Network 4: Error protusion de salida
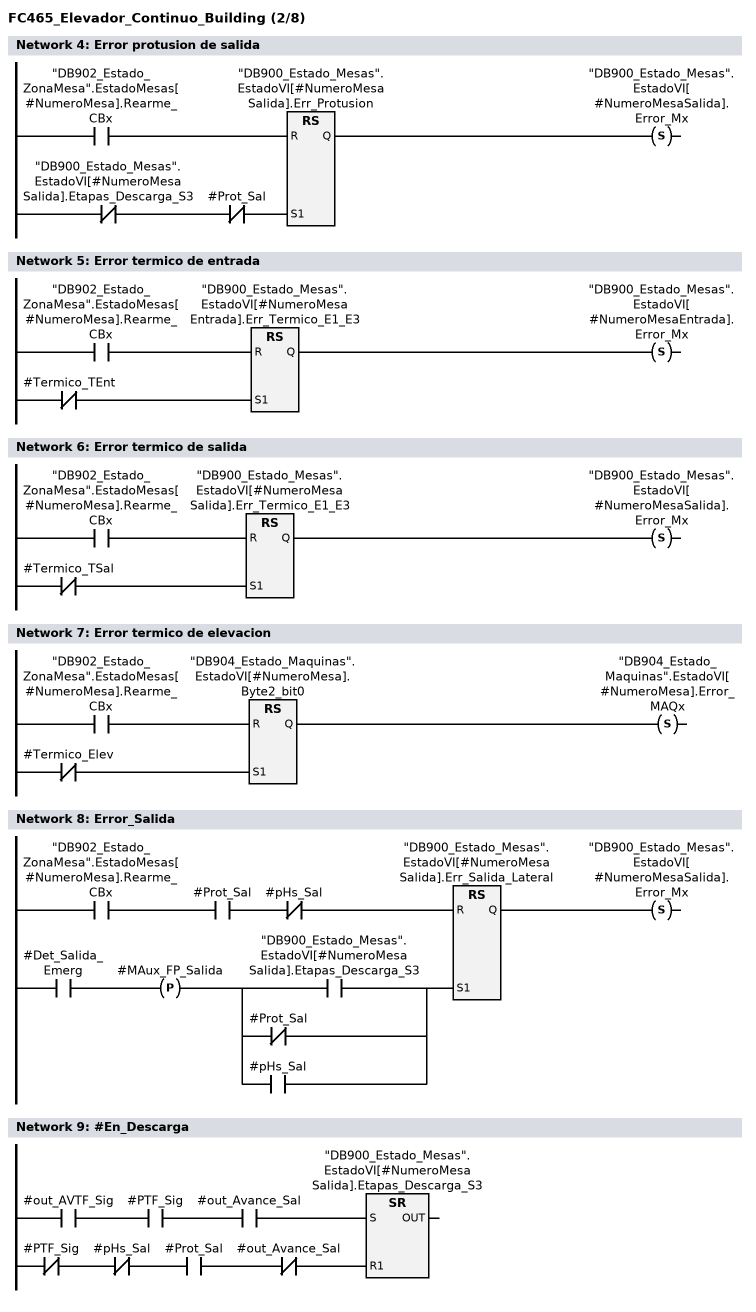
   RUNG wire#powerrail
      Contact( "DB902_Estado_ZonaMesa".EstadoMesas[#NumeroMesa].Rearme_CBx )
      S_RS(operand := "DB900_Estado_Mesas".EstadoVI[#NumeroMesaSalida].Err_Protusion, s1 := wire#w1)
      S_Coil( "DB900_Estado_Mesas".EstadoVI[#NumeroMesaSalida].Error_Mx )
   END_RUNG
   RUNG wire#powerrail
      I_Contact( "DB900_Estado_Mesas".EstadoVI[#NumeroMesaSalida].Etapas_Descarga_S3 )
      I_Contact( #Prot_Sal )
   END_RUNG wire#w1
   // the same network as SCL:
   #_w1 := NOT "DB900_Estado_Mesas".EstadoVI[#NumeroMesaSalida].Etapas_Descarga_S3 AND NOT #Prot_Sal;
   IF "DB902_Estado_ZonaMesa".EstadoMesas[#NumeroMesa].Rearme_CBx THEN
       "DB900_Estado_Mesas".EstadoVI[#NumeroMesaSalida].Err_Protusion := FALSE;   // RS flip-flop
   END_IF;
   IF #_w1 THEN "DB900_Estado_Mesas".EstadoVI[#NumeroMesaSalida].Err_Protusion := TRUE; END_IF;
   IF "DB900_Estado_Mesas".EstadoVI[#NumeroMesaSalida].Err_Protusion THEN
       "DB900_Estado_Mesas".EstadoVI[#NumeroMesaSalida].Error_Mx := TRUE;
   END_IF;
END_REGION

REGION Network 5: Error termico de entrada
   RUNG wire#powerrail
      Contact( "DB902_Estado_ZonaMesa".EstadoMesas[#NumeroMesa].Rearme_CBx )
      S_RS(operand := "DB900_Estado_Mesas".EstadoVI[#NumeroMesaEntrada].Err_Termico_E1_E3, s1 := wire#w1)
      S_Coil( "DB900_Estado_Mesas".EstadoVI[#NumeroMesaEntrada].Error_Mx )
   END_RUNG
   RUNG wire#powerrail
      I_Contact( #Termico_TEnt )
   END_RUNG wire#w1
   // the same network as SCL:
   IF "DB902_Estado_ZonaMesa".EstadoMesas[#NumeroMesa].Rearme_CBx THEN
       "DB900_Estado_Mesas".EstadoVI[#NumeroMesaEntrada].Err_Termico_E1_E3 := FALSE;   // RS flip-flop
   END_IF;
   IF NOT #Termico_TEnt THEN
       "DB900_Estado_Mesas".EstadoVI[#NumeroMesaEntrada].Err_Termico_E1_E3 := TRUE;
   END_IF;
   IF "DB900_Estado_Mesas".EstadoVI[#NumeroMesaEntrada].Err_Termico_E1_E3 THEN
       "DB900_Estado_Mesas".EstadoVI[#NumeroMesaEntrada].Error_Mx := TRUE;
   END_IF;
END_REGION

REGION Network 6: Error termico de salida
   RUNG wire#powerrail
      Contact( "DB902_Estado_ZonaMesa".EstadoMesas[#NumeroMesa].Rearme_CBx )
      S_RS(operand := "DB900_Estado_Mesas".EstadoVI[#NumeroMesaSalida].Err_Termico_E1_E3, s1 := wire#w1)
      S_Coil( "DB900_Estado_Mesas".EstadoVI[#NumeroMesaSalida].Error_Mx )
   END_RUNG
   RUNG wire#powerrail
      I_Contact( #Termico_TSal )
   END_RUNG wire#w1
   // the same network as SCL:
   IF "DB902_Estado_ZonaMesa".EstadoMesas[#NumeroMesa].Rearme_CBx THEN
       "DB900_Estado_Mesas".EstadoVI[#NumeroMesaSalida].Err_Termico_E1_E3 := FALSE;   // RS flip-flop
   END_IF;
   IF NOT #Termico_TSal THEN
       "DB900_Estado_Mesas".EstadoVI[#NumeroMesaSalida].Err_Termico_E1_E3 := TRUE;
   END_IF;
   IF "DB900_Estado_Mesas".EstadoVI[#NumeroMesaSalida].Err_Termico_E1_E3 THEN
       "DB900_Estado_Mesas".EstadoVI[#NumeroMesaSalida].Error_Mx := TRUE;
   END_IF;
END_REGION

REGION Network 7: Error termico de elevacion
   RUNG wire#powerrail
      Contact( "DB902_Estado_ZonaMesa".EstadoMesas[#NumeroMesa].Rearme_CBx )
      S_RS(operand := "DB904_Estado_Maquinas".EstadoVI[#NumeroMesa].Byte2_bit0, s1 := wire#w1)
      S_Coil( "DB904_Estado_Maquinas".EstadoVI[#NumeroMesa].Error_MAQx )
   END_RUNG
   RUNG wire#powerrail
      I_Contact( #Termico_Elev )
   END_RUNG wire#w1
   // the same network as SCL:
   IF "DB902_Estado_ZonaMesa".EstadoMesas[#NumeroMesa].Rearme_CBx THEN
       "DB904_Estado_Maquinas".EstadoVI[#NumeroMesa].Byte2_bit0 := FALSE;   // RS flip-flop
   END_IF;
   IF NOT #Termico_Elev THEN "DB904_Estado_Maquinas".EstadoVI[#NumeroMesa].Byte2_bit0 := TRUE; END_IF;
   IF "DB904_Estado_Maquinas".EstadoVI[#NumeroMesa].Byte2_bit0 THEN
       "DB904_Estado_Maquinas".EstadoVI[#NumeroMesa].Error_MAQx := TRUE;
   END_IF;
END_REGION

REGION Network 8: Error_Salida
   RUNG wire#powerrail
      Contact( "DB902_Estado_ZonaMesa".EstadoMesas[#NumeroMesa].Rearme_CBx )
      Contact( #Prot_Sal )
      I_Contact( #pHs_Sal )
      S_RS(operand := "DB900_Estado_Mesas".EstadoVI[#NumeroMesaSalida].Err_Salida_Lateral, s1 := wire#w2)
      S_Coil( "DB900_Estado_Mesas".EstadoVI[#NumeroMesaSalida].Error_Mx )
   END_RUNG
   RUNG wire#powerrail
      Contact( #Det_Salida_Emerg )
      P_Trig( #MAux_FP_Salida )
      wire#w1
      Contact( "DB900_Estado_Mesas".EstadoVI[#NumeroMesaSalida].Etapas_Descarga_S3 )
   END_RUNG wire#w2
   RUNG wire#w1
      I_Contact( #Prot_Sal )
   END_RUNG wire#w2
   RUNG wire#w1
      Contact( #pHs_Sal )
   END_RUNG wire#w2
   // the same network as SCL:
   #_w1 := #Det_Salida_Emerg AND NOT #MAux_FP_Salida;   // rising edge
   #MAux_FP_Salida := #Det_Salida_Emerg;
   #_w2 := #_w1 AND ("DB900_Estado_Mesas".EstadoVI[#NumeroMesaSalida].Etapas_Descarga_S3 OR NOT #Prot_Sal OR #pHs_Sal);
   IF "DB902_Estado_ZonaMesa".EstadoMesas[#NumeroMesa].Rearme_CBx AND #Prot_Sal AND NOT #pHs_Sal THEN
       "DB900_Estado_Mesas".EstadoVI[#NumeroMesaSalida].Err_Salida_Lateral := FALSE;   // RS flip-flop
   END_IF;
   IF #_w2 THEN "DB900_Estado_Mesas".EstadoVI[#NumeroMesaSalida].Err_Salida_Lateral := TRUE; END_IF;
   IF "DB900_Estado_Mesas".EstadoVI[#NumeroMesaSalida].Err_Salida_Lateral THEN
       "DB900_Estado_Mesas".EstadoVI[#NumeroMesaSalida].Error_Mx := TRUE;
   END_IF;
END_REGION

REGION Network 9: #En_Descarga
   RUNG wire#powerrail
      Contact( #out_AVTF_Sig )
      Contact( #PTF_Sig )
      Contact( #out_Avance_Sal )
      S_SR(operand := "DB900_Estado_Mesas".EstadoVI[#NumeroMesaSalida].Etapas_Descarga_S3, r1 := wire#w1)
   END_RUNG
   RUNG wire#powerrail
      I_Contact( #PTF_Sig )
      I_Contact( #pHs_Sal )
      Contact( #Prot_Sal )
      I_Contact( #out_Avance_Sal )
   END_RUNG wire#w1
   // the same network as SCL:
   IF #out_AVTF_Sig AND #PTF_Sig AND #out_Avance_Sal THEN
       "DB900_Estado_Mesas".EstadoVI[#NumeroMesaSalida].Etapas_Descarga_S3 := TRUE;   // SR flip-flop
   END_IF;
   IF NOT #PTF_Sig AND NOT #pHs_Sal AND #Prot_Sal AND NOT #out_Avance_Sal THEN
       "DB900_Estado_Mesas".EstadoVI[#NumeroMesaSalida].Etapas_Descarga_S3 := FALSE;
   END_IF;
END_REGION

REGION Network 10: Paro elevador por estar ocupada la salida
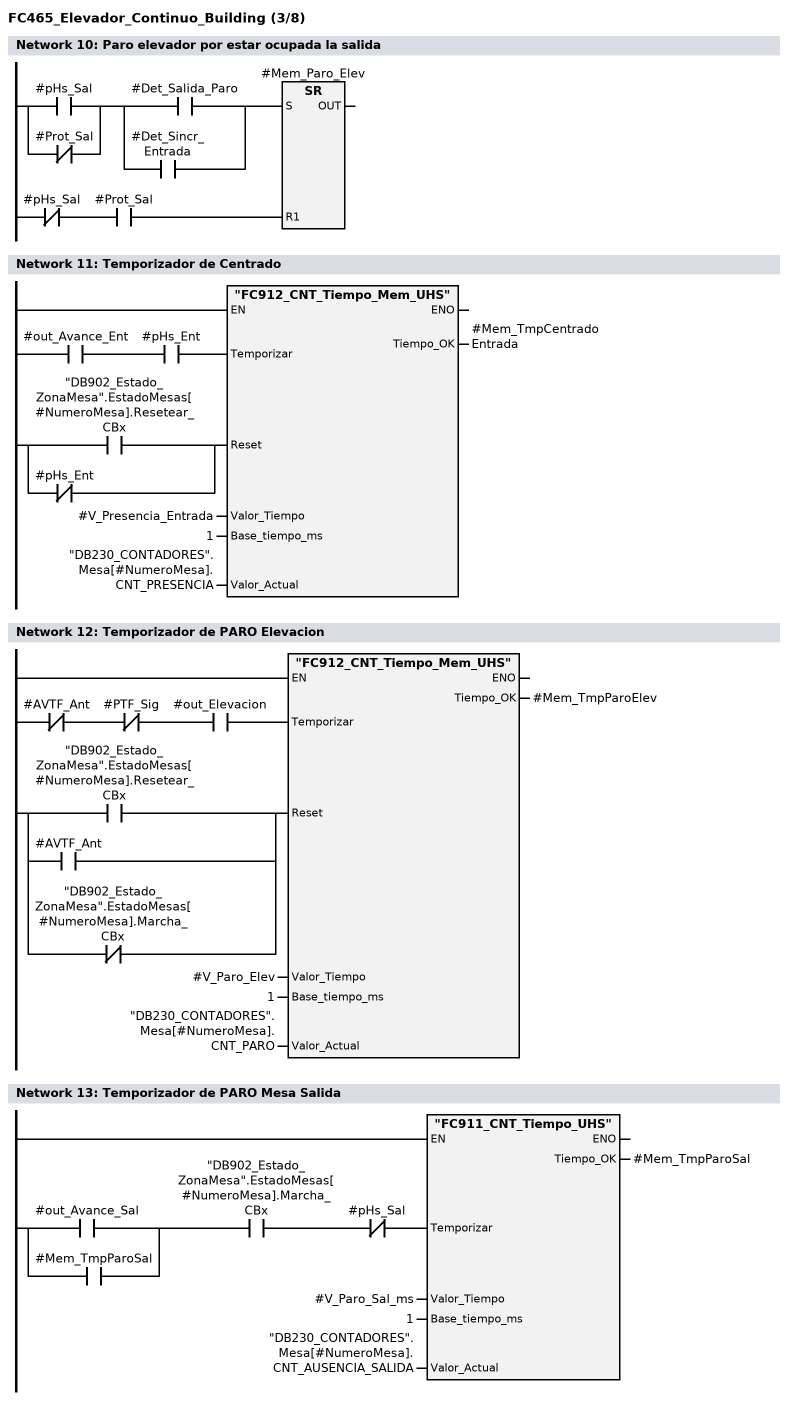
   RUNG wire#powerrail
      Contact( #pHs_Sal )
      wire#w1
      Contact( #Det_Salida_Paro )
      wire#w2
      S_SR(operand := #Mem_Paro_Elev, r1 := wire#w3)
   END_RUNG
   RUNG wire#powerrail
      I_Contact( #Prot_Sal )
   END_RUNG wire#w1
   RUNG wire#w1
      Contact( #Det_Sincr_Entrada )
   END_RUNG wire#w2
   RUNG wire#powerrail
      I_Contact( #pHs_Sal )
      Contact( #Prot_Sal )
   END_RUNG wire#w3
   // the same network as SCL:
   IF (#pHs_Sal OR NOT #Prot_Sal) AND (#Det_Salida_Paro OR #Det_Sincr_Entrada) THEN
       #Mem_Paro_Elev := TRUE;   // SR flip-flop
   END_IF;
   IF NOT #pHs_Sal AND #Prot_Sal THEN #Mem_Paro_Elev := FALSE; END_IF;
END_REGION

REGION Network 11: Temporizador de Centrado
   RUNG wire#powerrail
      "FC912_CNT_Tiempo_Mem_UHS"(Temporizar := wire#w1, Reset := wire#w2, Valor_Tiempo := #V_Presencia_Entrada, Base_tiempo_ms := 1, Valor_Actual := "DB230_CONTADORES".Mesa[#NumeroMesa].CNT_PRESENCIA, Tiempo_OK => #Mem_TmpCentradoEntrada)
   END_RUNG
   RUNG wire#powerrail
      Contact( #out_Avance_Ent )
      Contact( #pHs_Ent )
   END_RUNG wire#w1
   RUNG wire#powerrail
      Contact( "DB902_Estado_ZonaMesa".EstadoMesas[#NumeroMesa].Resetear_CBx )
   END_RUNG wire#w2
   RUNG wire#powerrail
      I_Contact( #pHs_Ent )
   END_RUNG wire#w2
   // the same network as SCL:
   "FC912_CNT_Tiempo_Mem_UHS"(Temporizar := #out_Avance_Ent AND #pHs_Ent,
                           Reset := "DB902_Estado_ZonaMesa".EstadoMesas[#NumeroMesa].Resetear_CBx OR NOT #pHs_Ent,
                           Valor_Tiempo := #V_Presencia_Entrada,
                           Base_tiempo_ms := 1,
                           Valor_Actual := "DB230_CONTADORES".Mesa[#NumeroMesa].CNT_PRESENCIA,
                           Tiempo_OK => #Mem_TmpCentradoEntrada);
END_REGION

REGION Network 12: Temporizador de PARO Elevacion
   RUNG wire#powerrail
      "FC912_CNT_Tiempo_Mem_UHS"(Temporizar := wire#w1, Reset := wire#w2, Valor_Tiempo := #V_Paro_Elev, Base_tiempo_ms := 1, Valor_Actual := "DB230_CONTADORES".Mesa[#NumeroMesa].CNT_PARO, Tiempo_OK => #Mem_TmpParoElev)
   END_RUNG
   RUNG wire#powerrail
      I_Contact( #AVTF_Ant )
      I_Contact( #PTF_Sig )
      Contact( #out_Elevacion )
   END_RUNG wire#w1
   RUNG wire#powerrail
      Contact( "DB902_Estado_ZonaMesa".EstadoMesas[#NumeroMesa].Resetear_CBx )
   END_RUNG wire#w2
   RUNG wire#powerrail
      Contact( #AVTF_Ant )
   END_RUNG wire#w2
   RUNG wire#powerrail
      I_Contact( "DB902_Estado_ZonaMesa".EstadoMesas[#NumeroMesa].Marcha_CBx )
   END_RUNG wire#w2
   // the same network as SCL:
   "FC912_CNT_Tiempo_Mem_UHS"(Temporizar := NOT #AVTF_Ant AND NOT #PTF_Sig AND #out_Elevacion,
                           Reset := "DB902_Estado_ZonaMesa".EstadoMesas[#NumeroMesa].Resetear_CBx OR #AVTF_Ant OR NOT "DB902_Estado_ZonaMesa".EstadoMesas[#NumeroMesa].Marcha_CBx,
                           Valor_Tiempo := #V_Paro_Elev,
                           Base_tiempo_ms := 1,
                           Valor_Actual := "DB230_CONTADORES".Mesa[#NumeroMesa].CNT_PARO,
                           Tiempo_OK => #Mem_TmpParoElev);
END_REGION

REGION Network 13: Temporizador de PARO Mesa Salida
   RUNG wire#powerrail
      "FC911_CNT_Tiempo_UHS"(Temporizar := wire#w2, Valor_Tiempo := #V_Paro_Sal_ms, Base_tiempo_ms := 1, Valor_Actual := "DB230_CONTADORES".Mesa[#NumeroMesa].CNT_AUSENCIA_SALIDA, Tiempo_OK => #Mem_TmpParoSal)
   END_RUNG
   RUNG wire#powerrail
      Contact( #out_Avance_Sal )
      wire#w1
      Contact( "DB902_Estado_ZonaMesa".EstadoMesas[#NumeroMesa].Marcha_CBx )
      I_Contact( #pHs_Sal )
   END_RUNG wire#w2
   RUNG wire#powerrail
      Contact( #Mem_TmpParoSal )
   END_RUNG wire#w1
   // the same network as SCL:
   "FC911_CNT_Tiempo_UHS"(Temporizar := (#out_Avance_Sal OR #Mem_TmpParoSal) AND "DB902_Estado_ZonaMesa".EstadoMesas[#NumeroMesa].Marcha_CBx AND NOT #pHs_Sal,
                          Valor_Tiempo := #V_Paro_Sal_ms,
                          Base_tiempo_ms := 1,
                          Valor_Actual := "DB230_CONTADORES".Mesa[#NumeroMesa].CNT_AUSENCIA_SALIDA,
                          Tiempo_OK => #Mem_TmpParoSal);
END_REGION

REGION Network 14: Temporizador de PARO E2
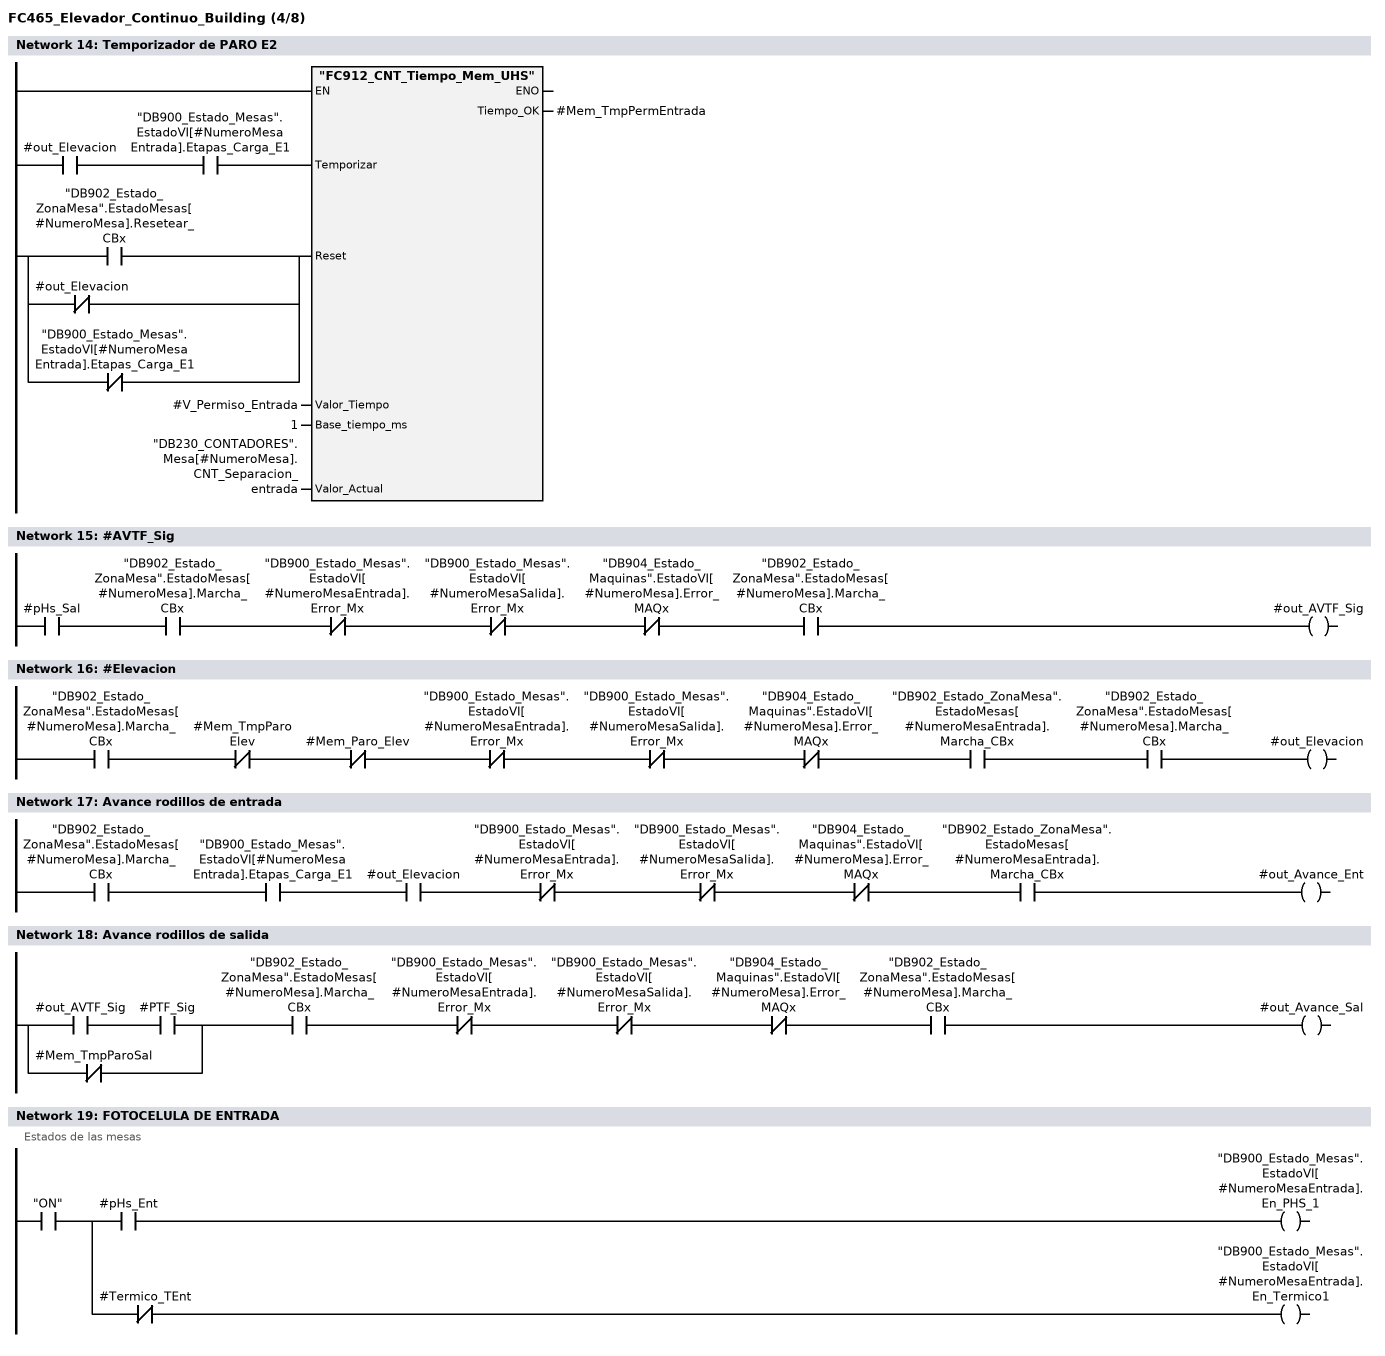
   RUNG wire#powerrail
      "FC912_CNT_Tiempo_Mem_UHS"(Temporizar := wire#w1, Reset := wire#w2, Valor_Tiempo := #V_Permiso_Entrada, Base_tiempo_ms := 1, Valor_Actual := "DB230_CONTADORES".Mesa[#NumeroMesa].CNT_Separacion_entrada, Tiempo_OK => #Mem_TmpPermEntrada)
   END_RUNG
   RUNG wire#powerrail
      Contact( #out_Elevacion )
      Contact( "DB900_Estado_Mesas".EstadoVI[#NumeroMesaEntrada].Etapas_Carga_E1 )
   END_RUNG wire#w1
   RUNG wire#powerrail
      Contact( "DB902_Estado_ZonaMesa".EstadoMesas[#NumeroMesa].Resetear_CBx )
   END_RUNG wire#w2
   RUNG wire#powerrail
      I_Contact( #out_Elevacion )
   END_RUNG wire#w2
   RUNG wire#powerrail
      I_Contact( "DB900_Estado_Mesas".EstadoVI[#NumeroMesaEntrada].Etapas_Carga_E1 )
   END_RUNG wire#w2
   // the same network as SCL:
   "FC912_CNT_Tiempo_Mem_UHS"(Temporizar := #out_Elevacion AND "DB900_Estado_Mesas".EstadoVI[#NumeroMesaEntrada].Etapas_Carga_E1,
                           Reset := "DB902_Estado_ZonaMesa".EstadoMesas[#NumeroMesa].Resetear_CBx OR NOT #out_Elevacion OR NOT "DB900_Estado_Mesas".EstadoVI[#NumeroMesaEntrada].Etapas_Carga_E1,
                           Valor_Tiempo := #V_Permiso_Entrada,
                           Base_tiempo_ms := 1,
                           Valor_Actual := "DB230_CONTADORES".Mesa[#NumeroMesa].CNT_Separacion_entrada,
                           Tiempo_OK => #Mem_TmpPermEntrada);
END_REGION

REGION Network 15: #AVTF_Sig
   RUNG wire#powerrail
      Contact( #pHs_Sal )
      Contact( "DB902_Estado_ZonaMesa".EstadoMesas[#NumeroMesa].Marcha_CBx )
      I_Contact( "DB900_Estado_Mesas".EstadoVI[#NumeroMesaEntrada].Error_Mx )
      I_Contact( "DB900_Estado_Mesas".EstadoVI[#NumeroMesaSalida].Error_Mx )
      I_Contact( "DB904_Estado_Maquinas".EstadoVI[#NumeroMesa].Error_MAQx )
      Contact( "DB902_Estado_ZonaMesa".EstadoMesas[#NumeroMesa].Marcha_CBx )
      Coil( #out_AVTF_Sig )
   END_RUNG
   // the same network as SCL:
   #out_AVTF_Sig := #pHs_Sal AND "DB902_Estado_ZonaMesa".EstadoMesas[#NumeroMesa].Marcha_CBx AND NOT "DB900_Estado_Mesas".EstadoVI[#NumeroMesaEntrada].Error_Mx AND NOT "DB900_Estado_Mesas".EstadoVI[#NumeroMesaSalida].Error_Mx AND NOT "DB904_Estado_Maquinas".EstadoVI[#NumeroMesa].Error_MAQx AND "DB902_Estado_ZonaMesa".EstadoMesas[#NumeroMesa].Marcha_CBx;
END_REGION

REGION Network 16: #Elevacion
   RUNG wire#powerrail
      Contact( "DB902_Estado_ZonaMesa".EstadoMesas[#NumeroMesa].Marcha_CBx )
      I_Contact( #Mem_TmpParoElev )
      I_Contact( #Mem_Paro_Elev )
      I_Contact( "DB900_Estado_Mesas".EstadoVI[#NumeroMesaEntrada].Error_Mx )
      I_Contact( "DB900_Estado_Mesas".EstadoVI[#NumeroMesaSalida].Error_Mx )
      I_Contact( "DB904_Estado_Maquinas".EstadoVI[#NumeroMesa].Error_MAQx )
      Contact( "DB902_Estado_ZonaMesa".EstadoMesas[#NumeroMesaEntrada].Marcha_CBx )
      Contact( "DB902_Estado_ZonaMesa".EstadoMesas[#NumeroMesa].Marcha_CBx )
      Coil( #out_Elevacion )
   END_RUNG
   // the same network as SCL:
   #out_Elevacion := "DB902_Estado_ZonaMesa".EstadoMesas[#NumeroMesa].Marcha_CBx AND NOT #Mem_TmpParoElev AND NOT #Mem_Paro_Elev AND NOT "DB900_Estado_Mesas".EstadoVI[#NumeroMesaEntrada].Error_Mx AND NOT "DB900_Estado_Mesas".EstadoVI[#NumeroMesaSalida].Error_Mx AND NOT "DB904_Estado_Maquinas".EstadoVI[#NumeroMesa].Error_MAQx AND "DB902_Estado_ZonaMesa".EstadoMesas[#NumeroMesaEntrada].Marcha_CBx AND "DB902_Estado_ZonaMesa".EstadoMesas[#NumeroMesa].Marcha_CBx;
END_REGION

REGION Network 17: Avance rodillos de entrada
   RUNG wire#powerrail
      Contact( "DB902_Estado_ZonaMesa".EstadoMesas[#NumeroMesa].Marcha_CBx )
      Contact( "DB900_Estado_Mesas".EstadoVI[#NumeroMesaEntrada].Etapas_Carga_E1 )
      Contact( #out_Elevacion )
      I_Contact( "DB900_Estado_Mesas".EstadoVI[#NumeroMesaEntrada].Error_Mx )
      I_Contact( "DB900_Estado_Mesas".EstadoVI[#NumeroMesaSalida].Error_Mx )
      I_Contact( "DB904_Estado_Maquinas".EstadoVI[#NumeroMesa].Error_MAQx )
      Contact( "DB902_Estado_ZonaMesa".EstadoMesas[#NumeroMesaEntrada].Marcha_CBx )
      Coil( #out_Avance_Ent )
   END_RUNG
   // the same network as SCL:
   #out_Avance_Ent := "DB902_Estado_ZonaMesa".EstadoMesas[#NumeroMesa].Marcha_CBx AND "DB900_Estado_Mesas".EstadoVI[#NumeroMesaEntrada].Etapas_Carga_E1 AND #out_Elevacion AND NOT "DB900_Estado_Mesas".EstadoVI[#NumeroMesaEntrada].Error_Mx AND NOT "DB900_Estado_Mesas".EstadoVI[#NumeroMesaSalida].Error_Mx AND NOT "DB904_Estado_Maquinas".EstadoVI[#NumeroMesa].Error_MAQx AND "DB902_Estado_ZonaMesa".EstadoMesas[#NumeroMesaEntrada].Marcha_CBx;
END_REGION

REGION Network 18: Avance rodillos de salida
   RUNG wire#powerrail
      Contact( #out_AVTF_Sig )
      Contact( #PTF_Sig )
      wire#w1
      Contact( "DB902_Estado_ZonaMesa".EstadoMesas[#NumeroMesa].Marcha_CBx )
      I_Contact( "DB900_Estado_Mesas".EstadoVI[#NumeroMesaEntrada].Error_Mx )
      I_Contact( "DB900_Estado_Mesas".EstadoVI[#NumeroMesaSalida].Error_Mx )
      I_Contact( "DB904_Estado_Maquinas".EstadoVI[#NumeroMesa].Error_MAQx )
      Contact( "DB902_Estado_ZonaMesa".EstadoMesas[#NumeroMesa].Marcha_CBx )
      Coil( #out_Avance_Sal )
   END_RUNG
   RUNG wire#powerrail
      I_Contact( #Mem_TmpParoSal )
   END_RUNG wire#w1
   // the same network as SCL:
   #out_Avance_Sal := ((#out_AVTF_Sig AND #PTF_Sig) OR NOT #Mem_TmpParoSal) AND "DB902_Estado_ZonaMesa".EstadoMesas[#NumeroMesa].Marcha_CBx AND NOT "DB900_Estado_Mesas".EstadoVI[#NumeroMesaEntrada].Error_Mx AND NOT "DB900_Estado_Mesas".EstadoVI[#NumeroMesaSalida].Error_Mx AND NOT "DB904_Estado_Maquinas".EstadoVI[#NumeroMesa].Error_MAQx AND "DB902_Estado_ZonaMesa".EstadoMesas[#NumeroMesa].Marcha_CBx;
END_REGION

REGION Network 19: FOTOCELULA DE ENTRADA
   // Estados de las mesas
   RUNG wire#powerrail
      Contact( "ON" )
      wire#w1
      Contact( #pHs_Ent )
      Coil( "DB900_Estado_Mesas".EstadoVI[#NumeroMesaEntrada].En_PHS_1 )
   END_RUNG
   RUNG wire#w1
      I_Contact( #Termico_TEnt )
      Coil( "DB900_Estado_Mesas".EstadoVI[#NumeroMesaEntrada].En_Termico1 )
   END_RUNG
   // the same network as SCL:
   "DB900_Estado_Mesas".EstadoVI[#NumeroMesaEntrada].En_PHS_1 := "ON" AND #pHs_Ent;
   "DB900_Estado_Mesas".EstadoVI[#NumeroMesaEntrada].En_Termico1 := "ON" AND NOT #Termico_TEnt;
END_REGION

REGION Network 20: ESTADOS MESA ENTRADA
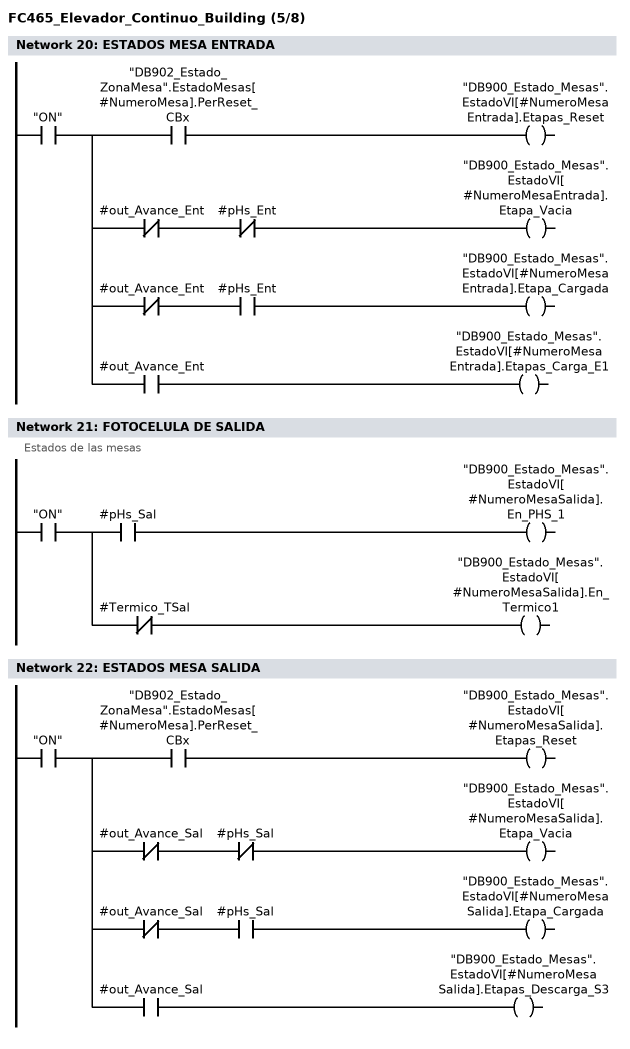
   RUNG wire#powerrail
      Contact( "ON" )
      wire#w1
      Contact( "DB902_Estado_ZonaMesa".EstadoMesas[#NumeroMesa].PerReset_CBx )
      Coil( "DB900_Estado_Mesas".EstadoVI[#NumeroMesaEntrada].Etapas_Reset )
   END_RUNG
   RUNG wire#w1
      I_Contact( #out_Avance_Ent )
      I_Contact( #pHs_Ent )
      Coil( "DB900_Estado_Mesas".EstadoVI[#NumeroMesaEntrada].Etapa_Vacia )
   END_RUNG
   RUNG wire#w1
      I_Contact( #out_Avance_Ent )
      Contact( #pHs_Ent )
      Coil( "DB900_Estado_Mesas".EstadoVI[#NumeroMesaEntrada].Etapa_Cargada )
   END_RUNG
   RUNG wire#w1
      Contact( #out_Avance_Ent )
      Coil( "DB900_Estado_Mesas".EstadoVI[#NumeroMesaEntrada].Etapas_Carga_E1 )
   END_RUNG
   // the same network as SCL:
   "DB900_Estado_Mesas".EstadoVI[#NumeroMesaEntrada].Etapas_Reset := "ON" AND "DB902_Estado_ZonaMesa".EstadoMesas[#NumeroMesa].PerReset_CBx;
   "DB900_Estado_Mesas".EstadoVI[#NumeroMesaEntrada].Etapa_Vacia := "ON" AND NOT #out_Avance_Ent AND NOT #pHs_Ent;
   "DB900_Estado_Mesas".EstadoVI[#NumeroMesaEntrada].Etapa_Cargada := "ON" AND NOT #out_Avance_Ent AND #pHs_Ent;
   "DB900_Estado_Mesas".EstadoVI[#NumeroMesaEntrada].Etapas_Carga_E1 := "ON" AND #out_Avance_Ent;
END_REGION

REGION Network 21: FOTOCELULA DE SALIDA
   // Estados de las mesas
   RUNG wire#powerrail
      Contact( "ON" )
      wire#w1
      Contact( #pHs_Sal )
      Coil( "DB900_Estado_Mesas".EstadoVI[#NumeroMesaSalida].En_PHS_1 )
   END_RUNG
   RUNG wire#w1
      I_Contact( #Termico_TSal )
      Coil( "DB900_Estado_Mesas".EstadoVI[#NumeroMesaSalida].En_Termico1 )
   END_RUNG
   // the same network as SCL:
   "DB900_Estado_Mesas".EstadoVI[#NumeroMesaSalida].En_PHS_1 := "ON" AND #pHs_Sal;
   "DB900_Estado_Mesas".EstadoVI[#NumeroMesaSalida].En_Termico1 := "ON" AND NOT #Termico_TSal;
END_REGION

REGION Network 22: ESTADOS MESA SALIDA
   RUNG wire#powerrail
      Contact( "ON" )
      wire#w1
      Contact( "DB902_Estado_ZonaMesa".EstadoMesas[#NumeroMesa].PerReset_CBx )
      Coil( "DB900_Estado_Mesas".EstadoVI[#NumeroMesaSalida].Etapas_Reset )
   END_RUNG
   RUNG wire#w1
      I_Contact( #out_Avance_Sal )
      I_Contact( #pHs_Sal )
      Coil( "DB900_Estado_Mesas".EstadoVI[#NumeroMesaSalida].Etapa_Vacia )
   END_RUNG
   RUNG wire#w1
      I_Contact( #out_Avance_Sal )
      Contact( #pHs_Sal )
      Coil( "DB900_Estado_Mesas".EstadoVI[#NumeroMesaSalida].Etapa_Cargada )
   END_RUNG
   RUNG wire#w1
      Contact( #out_Avance_Sal )
      Coil( "DB900_Estado_Mesas".EstadoVI[#NumeroMesaSalida].Etapas_Descarga_S3 )
   END_RUNG
   // the same network as SCL:
   "DB900_Estado_Mesas".EstadoVI[#NumeroMesaSalida].Etapas_Reset := "ON" AND "DB902_Estado_ZonaMesa".EstadoMesas[#NumeroMesa].PerReset_CBx;
   "DB900_Estado_Mesas".EstadoVI[#NumeroMesaSalida].Etapa_Vacia := "ON" AND NOT #out_Avance_Sal AND NOT #pHs_Sal;
   "DB900_Estado_Mesas".EstadoVI[#NumeroMesaSalida].Etapa_Cargada := "ON" AND NOT #out_Avance_Sal AND #pHs_Sal;
   "DB900_Estado_Mesas".EstadoVI[#NumeroMesaSalida].Etapas_Descarga_S3 := "ON" AND #out_Avance_Sal;
END_REGION

REGION Network 23: ESTADOS MESA SALIDA
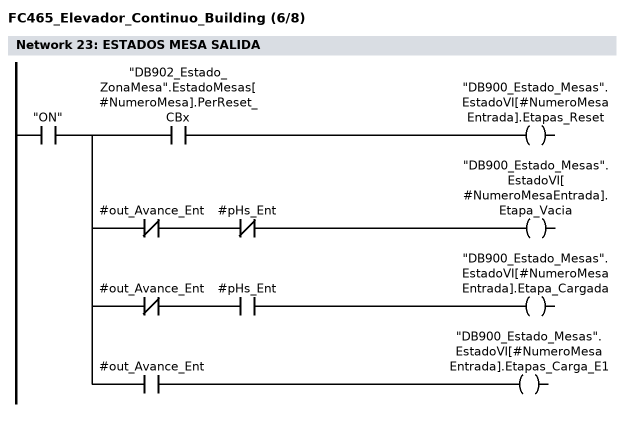
   RUNG wire#powerrail
      Contact( "ON" )
      wire#w1
      Contact( "DB902_Estado_ZonaMesa".EstadoMesas[#NumeroMesa].PerReset_CBx )
      Coil( "DB900_Estado_Mesas".EstadoVI[#NumeroMesaEntrada].Etapas_Reset )
   END_RUNG
   RUNG wire#w1
      I_Contact( #out_Avance_Ent )
      I_Contact( #pHs_Ent )
      Coil( "DB900_Estado_Mesas".EstadoVI[#NumeroMesaEntrada].Etapa_Vacia )
   END_RUNG
   RUNG wire#w1
      I_Contact( #out_Avance_Ent )
      Contact( #pHs_Ent )
      Coil( "DB900_Estado_Mesas".EstadoVI[#NumeroMesaEntrada].Etapa_Cargada )
   END_RUNG
   RUNG wire#w1
      Contact( #out_Avance_Ent )
      Coil( "DB900_Estado_Mesas".EstadoVI[#NumeroMesaEntrada].Etapas_Carga_E1 )
   END_RUNG
   // the same network as SCL:
   "DB900_Estado_Mesas".EstadoVI[#NumeroMesaEntrada].Etapas_Reset := "ON" AND "DB902_Estado_ZonaMesa".EstadoMesas[#NumeroMesa].PerReset_CBx;
   "DB900_Estado_Mesas".EstadoVI[#NumeroMesaEntrada].Etapa_Vacia := "ON" AND NOT #out_Avance_Ent AND NOT #pHs_Ent;
   "DB900_Estado_Mesas".EstadoVI[#NumeroMesaEntrada].Etapa_Cargada := "ON" AND NOT #out_Avance_Ent AND #pHs_Ent;
   "DB900_Estado_Mesas".EstadoVI[#NumeroMesaEntrada].Etapas_Carga_E1 := "ON" AND #out_Avance_Ent;
END_REGION

REGION Network 24: ESTADO MAQUINA
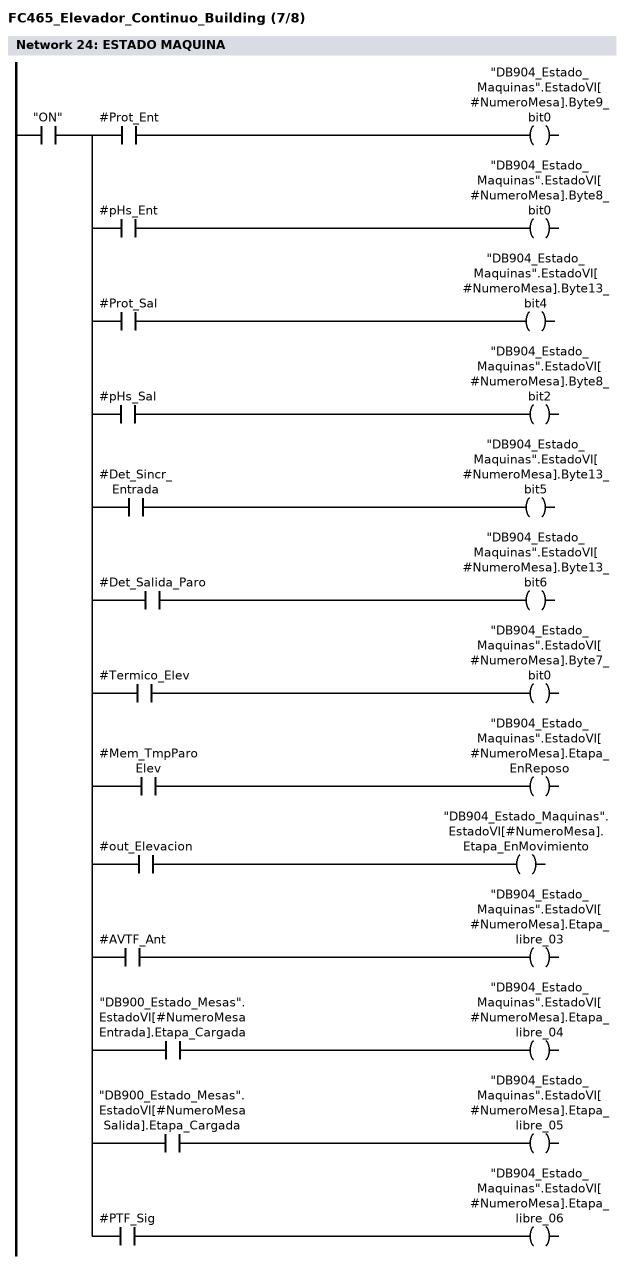
   RUNG wire#powerrail
      Contact( "ON" )
      wire#w1
      Contact( #Prot_Ent )
      Coil( "DB904_Estado_Maquinas".EstadoVI[#NumeroMesa].Byte9_bit0 )
   END_RUNG
   RUNG wire#w1
      Contact( #pHs_Ent )
      Coil( "DB904_Estado_Maquinas".EstadoVI[#NumeroMesa].Byte8_bit0 )
   END_RUNG
   RUNG wire#w1
      Contact( #Prot_Sal )
      Coil( "DB904_Estado_Maquinas".EstadoVI[#NumeroMesa].Byte13_bit4 )
   END_RUNG
   RUNG wire#w1
      Contact( #pHs_Sal )
      Coil( "DB904_Estado_Maquinas".EstadoVI[#NumeroMesa].Byte8_bit2 )
   END_RUNG
   RUNG wire#w1
      Contact( #Det_Sincr_Entrada )
      Coil( "DB904_Estado_Maquinas".EstadoVI[#NumeroMesa].Byte13_bit5 )
   END_RUNG
   RUNG wire#w1
      Contact( #Det_Salida_Paro )
      Coil( "DB904_Estado_Maquinas".EstadoVI[#NumeroMesa].Byte13_bit6 )
   END_RUNG
   RUNG wire#w1
      Contact( #Termico_Elev )
      Coil( "DB904_Estado_Maquinas".EstadoVI[#NumeroMesa].Byte7_bit0 )
   END_RUNG
   RUNG wire#w1
      Contact( #Mem_TmpParoElev )
      Coil( "DB904_Estado_Maquinas".EstadoVI[#NumeroMesa].Etapa_EnReposo )
   END_RUNG
   RUNG wire#w1
      Contact( #out_Elevacion )
      Coil( "DB904_Estado_Maquinas".EstadoVI[#NumeroMesa].Etapa_EnMovimiento )
   END_RUNG
   RUNG wire#w1
      Contact( #AVTF_Ant )
      Coil( "DB904_Estado_Maquinas".EstadoVI[#NumeroMesa].Etapa_libre_03 )
   END_RUNG
   RUNG wire#w1
      Contact( "DB900_Estado_Mesas".EstadoVI[#NumeroMesaEntrada].Etapa_Cargada )
      Coil( "DB904_Estado_Maquinas".EstadoVI[#NumeroMesa].Etapa_libre_04 )
   END_RUNG
   RUNG wire#w1
      Contact( "DB900_Estado_Mesas".EstadoVI[#NumeroMesaSalida].Etapa_Cargada )
      Coil( "DB904_Estado_Maquinas".EstadoVI[#NumeroMesa].Etapa_libre_05 )
   END_RUNG
   RUNG wire#w1
      Contact( #PTF_Sig )
      Coil( "DB904_Estado_Maquinas".EstadoVI[#NumeroMesa].Etapa_libre_06 )
   END_RUNG
   // the same network as SCL:
   "DB904_Estado_Maquinas".EstadoVI[#NumeroMesa].Byte9_bit0 := "ON" AND #Prot_Ent;
   "DB904_Estado_Maquinas".EstadoVI[#NumeroMesa].Byte8_bit0 := "ON" AND #pHs_Ent;
   "DB904_Estado_Maquinas".EstadoVI[#NumeroMesa].Byte13_bit4 := "ON" AND #Prot_Sal;
   "DB904_Estado_Maquinas".EstadoVI[#NumeroMesa].Byte8_bit2 := "ON" AND #pHs_Sal;
   "DB904_Estado_Maquinas".EstadoVI[#NumeroMesa].Byte13_bit5 := "ON" AND #Det_Sincr_Entrada;
   "DB904_Estado_Maquinas".EstadoVI[#NumeroMesa].Byte13_bit6 := "ON" AND #Det_Salida_Paro;
   "DB904_Estado_Maquinas".EstadoVI[#NumeroMesa].Byte7_bit0 := "ON" AND #Termico_Elev;
   "DB904_Estado_Maquinas".EstadoVI[#NumeroMesa].Etapa_EnReposo := "ON" AND #Mem_TmpParoElev;
   "DB904_Estado_Maquinas".EstadoVI[#NumeroMesa].Etapa_EnMovimiento := "ON" AND #out_Elevacion;
   "DB904_Estado_Maquinas".EstadoVI[#NumeroMesa].Etapa_libre_03 := "ON" AND #AVTF_Ant;
   "DB904_Estado_Maquinas".EstadoVI[#NumeroMesa].Etapa_libre_04 := "ON" AND "DB900_Estado_Mesas".EstadoVI[#NumeroMesaEntrada].Etapa_Cargada;
   "DB904_Estado_Maquinas".EstadoVI[#NumeroMesa].Etapa_libre_05 := "ON" AND "DB900_Estado_Mesas".EstadoVI[#NumeroMesaSalida].Etapa_Cargada;
   "DB904_Estado_Maquinas".EstadoVI[#NumeroMesa].Etapa_libre_06 := "ON" AND #PTF_Sig;
END_REGION

REGION Network 25: Fin de Vehiculo
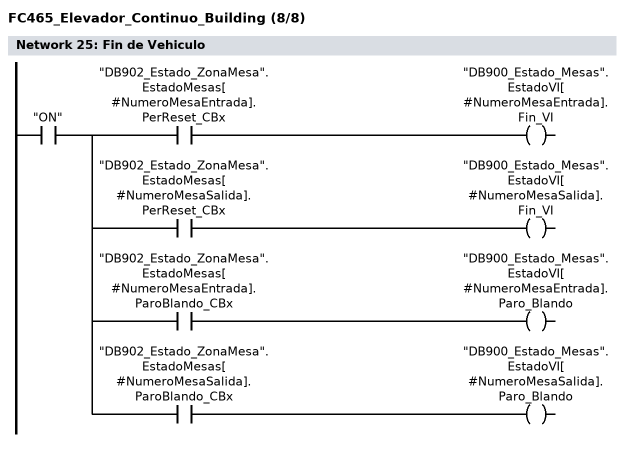
   RUNG wire#powerrail
      Contact( "ON" )
      wire#w1
      Contact( "DB902_Estado_ZonaMesa".EstadoMesas[#NumeroMesaEntrada].PerReset_CBx )
      Coil( "DB900_Estado_Mesas".EstadoVI[#NumeroMesaEntrada].Fin_VI )
   END_RUNG
   RUNG wire#w1
      Contact( "DB902_Estado_ZonaMesa".EstadoMesas[#NumeroMesaSalida].PerReset_CBx )
      Coil( "DB900_Estado_Mesas".EstadoVI[#NumeroMesaSalida].Fin_VI )
   END_RUNG
   RUNG wire#w1
      Contact( "DB902_Estado_ZonaMesa".EstadoMesas[#NumeroMesaEntrada].ParoBlando_CBx )
      Coil( "DB900_Estado_Mesas".EstadoVI[#NumeroMesaEntrada].Paro_Blando )
   END_RUNG
   RUNG wire#w1
      Contact( "DB902_Estado_ZonaMesa".EstadoMesas[#NumeroMesaSalida].ParoBlando_CBx )
      Coil( "DB900_Estado_Mesas".EstadoVI[#NumeroMesaSalida].Paro_Blando )
   END_RUNG
   // the same network as SCL:
   "DB900_Estado_Mesas".EstadoVI[#NumeroMesaEntrada].Fin_VI := "ON" AND "DB902_Estado_ZonaMesa".EstadoMesas[#NumeroMesaEntrada].PerReset_CBx;
   "DB900_Estado_Mesas".EstadoVI[#NumeroMesaSalida].Fin_VI := "ON" AND "DB902_Estado_ZonaMesa".EstadoMesas[#NumeroMesaSalida].PerReset_CBx;
   "DB900_Estado_Mesas".EstadoVI[#NumeroMesaEntrada].Paro_Blando := "ON" AND "DB902_Estado_ZonaMesa".EstadoMesas[#NumeroMesaEntrada].ParoBlando_CBx;
   "DB900_Estado_Mesas".EstadoVI[#NumeroMesaSalida].Paro_Blando := "ON" AND "DB902_Estado_ZonaMesa".EstadoMesas[#NumeroMesaSalida].ParoBlando_CBx;
END_REGION
END_FUNCTION

FUNCTION "FC505_CNT_ET_OK_NOOK" : Void   // FC505, LAD
{ S7_Optimized_Access := 'FALSE' }
AUTHOR : TLigero
NAME : 20130623
VERSION : 3.1
// stored: AutoNumber false, SetENOAutomatically false
   VAR_INPUT
      Num_Scanner : UInt;
      Evento_a_Registrar : UInt;   // 1 lectura nook, 2 lectura ok, 3 lectura no encontrada
   END_VAR
   VAR_TEMP
      Cero : Byte;
      retval : Int;
      Auxiliar : UInt;
   END_VAR
BEGIN

NETWORK
TITLE = inicializacion
//============================================================

      L     0;
      T     #Cero;


//============================================================

NETWORK
TITLE = Sacamos los datos previamente guardados para actualizarlos
//============================================================
// -- revisamos si hay algún dato que se va a desbordar

      SET;
      L     "DB216_Cnt_Estadisticas_Scanners".CNT_LectSCR[#Num_Scanner].Lect_Good;
      L     65535;
      ==I;
      JC    inicializa;


      SET;
      L     "DB216_Cnt_Estadisticas_Scanners".CNT_LectSCR[#Num_Scanner].Lect_NoGood;
      L     65535;
      ==I;
      JC    inicializa;

      JU    registra_datos;

//============================================================
// -- Ponemos a cero todos los datos salvo el contador
// -- de lecturas malas consecutivas
inicializa:NOP   0;

      L     "DB216_Cnt_Estadisticas_Scanners".CNT_LectSCR[#Num_Scanner].Lect_NoGood_consecutivas;
      T     #Auxiliar;
      CALL  FILL
      ( BVAL    := #Cero,
        RET_VAL := #retval,
        BLK     := "DB216_Cnt_Estadisticas_Scanners".CNT_LectSCR[#Num_Scanner]
      );

      L     #Auxiliar;
      T     "DB216_Cnt_Estadisticas_Scanners".CNT_LectSCR[#Num_Scanner].Lect_NoGood_consecutivas;
//============================================================


NETWORK
TITLE = Registrar los datos
//============================================================
registra_datos:NOP   0;

      L     #Evento_a_Registrar;

      JL    valor_no_valido;

      JU    valor_no_valido;  // --- Con dato 0
      JU    contar_lectura_nook;  // --- Con dato 1
      JU    contar_lectura_ok;  // --- Con dato 2
      JU    contar_no_encontradas;  // --- Con dato 2

valor_no_valido:JU    guardar_datos;  // --- Motivo INEXISTENTE


//============================================================
// -- Contar lectura ok

contar_lectura_nook:NOP   0;
      L     "DB216_Cnt_Estadisticas_Scanners".CNT_LectSCR[#Num_Scanner].Lect_NoGood;
      L     1;
      +I;
      T     "DB216_Cnt_Estadisticas_Scanners".CNT_LectSCR[#Num_Scanner].Lect_NoGood;

//-- incrementamos también el contador
// -- de lecturas malas consecutivas
      L     "DB216_Cnt_Estadisticas_Scanners".CNT_LectSCR[#Num_Scanner].Lect_NoGood_consecutivas;
      L     1;
      +I;
      T     "DB216_Cnt_Estadisticas_Scanners".CNT_LectSCR[#Num_Scanner].Lect_NoGood_consecutivas;

      JU    guardar_datos;

//============================================================
// -- Contar lectura ok

contar_lectura_ok:NOP   0;
      L     "DB216_Cnt_Estadisticas_Scanners".CNT_LectSCR[#Num_Scanner].Lect_Good;
      L     1;
      +I;
      T     "DB216_Cnt_Estadisticas_Scanners".CNT_LectSCR[#Num_Scanner].Lect_Good;

//-- como hemos tenido lectura ok
//-- reseteamos el contador de errores consecutivos
      L     0;
      T     "DB216_Cnt_Estadisticas_Scanners".CNT_LectSCR[#Num_Scanner].Lect_NoGood_consecutivas;

      JU    guardar_datos;
//============================================================
// -- Contar no encontrada
// -- Suma 1 también a lectura ok
contar_no_encontradas:NOP   0;

      L     "DB216_Cnt_Estadisticas_Scanners".CNT_LectSCR[#Num_Scanner].Lect_NoFound;
      L     1;
      +I;
      T     "DB216_Cnt_Estadisticas_Scanners".CNT_LectSCR[#Num_Scanner].Lect_NoFound;

      L     "DB216_Cnt_Estadisticas_Scanners".CNT_LectSCR[#Num_Scanner].Lect_Good;
      L     1;
      +I;
      T     "DB216_Cnt_Estadisticas_Scanners".CNT_LectSCR[#Num_Scanner].Lect_Good;

//-- como hemos tenido lectura ok
//-- reseteamos el contador de errores consecutivos
      L     0;
      T     "DB216_Cnt_Estadisticas_Scanners".CNT_LectSCR[#Num_Scanner].Lect_NoGood_consecutivas;

      JU    guardar_datos;

//============================================================

NETWORK
TITLE = Guardar los datos actualizados
//============================================================
guardar_datos:NOP   0;


//============================================================

END_FUNCTION

